REGION Network 6: LECTURA ESCANER SIDE LH
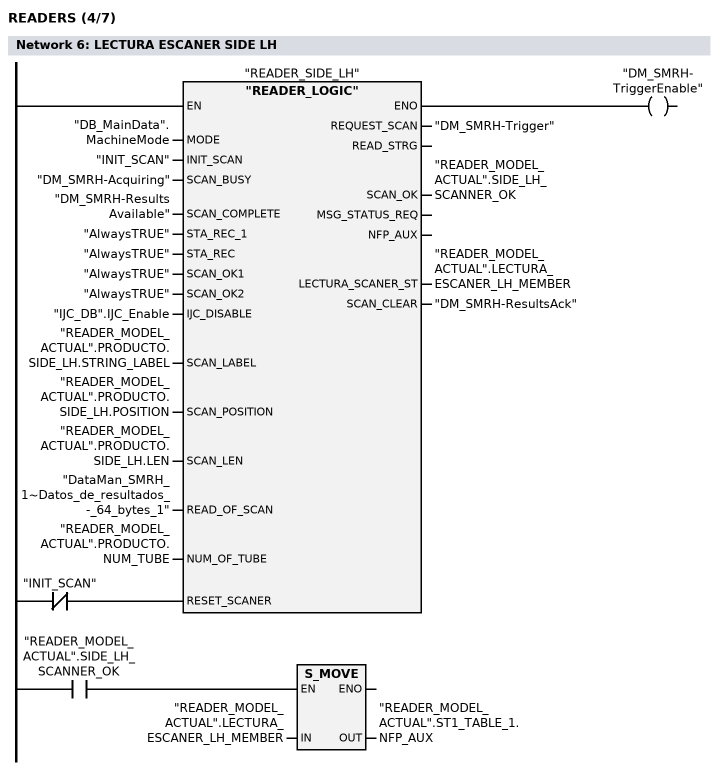
   RUNG wire#powerrail
      "READER_SIDE_LH"(RESET_SCANER := wire#w1, MODE := "DB_MainData".MachineMode, INIT_SCAN := "INIT_SCAN", SCAN_BUSY := "DM_SMRH-Acquiring", SCAN_COMPLETE := "DM_SMRH-Results Available", STA_REC_1 := "AlwaysTRUE", STA_REC := "AlwaysTRUE", SCAN_OK1 := "AlwaysTRUE", SCAN_OK2 := "AlwaysTRUE", IJC_DISABLE := "IJC_DB".IJC_Enable, SCAN_LABEL := "READER_MODEL_ACTUAL".PRODUCTO.SIDE_LH.STRING_LABEL, SCAN_POSITION := "READER_MODEL_ACTUAL".PRODUCTO.SIDE_LH.POSITION, SCAN_LEN := "READER_MODEL_ACTUAL".PRODUCTO.SIDE_LH.LEN, READ_OF_SCAN := "DataMan_SMRH_1~Datos_de_resultados_-_64_bytes_1", NUM_OF_TUBE := "READER_MODEL_ACTUAL".PRODUCTO.NUM_TUBE, REQUEST_SCAN => "DM_SMRH-Trigger", READ_STRG =>, SCAN_OK => "READER_MODEL_ACTUAL".SIDE_LH_SCANNER_OK, MSG_STATUS_REQ =>, NFP_AUX =>, LECTURA_SCANER_ST => "READER_MODEL_ACTUAL".LECTURA_ESCANER_LH_MEMBER, SCAN_CLEAR => "DM_SMRH-ResultsAck")
      Coil( "DM_SMRH-TriggerEnable" )
   END_RUNG
   RUNG wire#powerrail
      I_Contact( "INIT_SCAN" )
   END_RUNG wire#w1
   RUNG wire#powerrail
      Contact( "READER_MODEL_ACTUAL".SIDE_LH_SCANNER_OK )
      S_Move(in := "READER_MODEL_ACTUAL".LECTURA_ESCANER_LH_MEMBER, out => "READER_MODEL_ACTUAL".ST1_TABLE_1.NFP_AUX)
   END_RUNG
   // the same network as SCL:
   "READER_SIDE_LH"(MODE := "DB_MainData".MachineMode,   // "READER_LOGIC"
                    INIT_SCAN := "INIT_SCAN",
                    SCAN_BUSY := "DM_SMRH-Acquiring",
                    SCAN_COMPLETE := "DM_SMRH-Results Available",
                    STA_REC_1 := "AlwaysTRUE",
                    STA_REC := "AlwaysTRUE",
                    SCAN_OK1 := "AlwaysTRUE",
                    SCAN_OK2 := "AlwaysTRUE",
                    IJC_DISABLE := "IJC_DB".IJC_Enable,
                    SCAN_LABEL := "READER_MODEL_ACTUAL".PRODUCTO.SIDE_LH.STRING_LABEL,
                    SCAN_POSITION := "READER_MODEL_ACTUAL".PRODUCTO.SIDE_LH.POSITION,
                    SCAN_LEN := "READER_MODEL_ACTUAL".PRODUCTO.SIDE_LH.LEN,
                    READ_OF_SCAN := "DataMan_SMRH_1~Datos_de_resultados_-_64_bytes_1",
                    NUM_OF_TUBE := "READER_MODEL_ACTUAL".PRODUCTO.NUM_TUBE,
                    RESET_SCANER := NOT "INIT_SCAN",
                    REQUEST_SCAN => "DM_SMRH-Trigger",
                    SCAN_OK => "READER_MODEL_ACTUAL".SIDE_LH_SCANNER_OK,
                    LECTURA_SCANER_ST => "READER_MODEL_ACTUAL".LECTURA_ESCANER_LH_MEMBER,
                    SCAN_CLEAR => "DM_SMRH-ResultsAck",
                    ENO => #_w1);
   "DM_SMRH-TriggerEnable" := #_w1;
   IF "READER_MODEL_ACTUAL".SIDE_LH_SCANNER_OK THEN
       "READER_MODEL_ACTUAL".ST1_TABLE_1.NFP_AUX := "READER_MODEL_ACTUAL".LECTURA_ESCANER_LH_MEMBER;
   END_IF;
END_REGION

REGION Network 7: LECTURA ESCANER SIDE RH
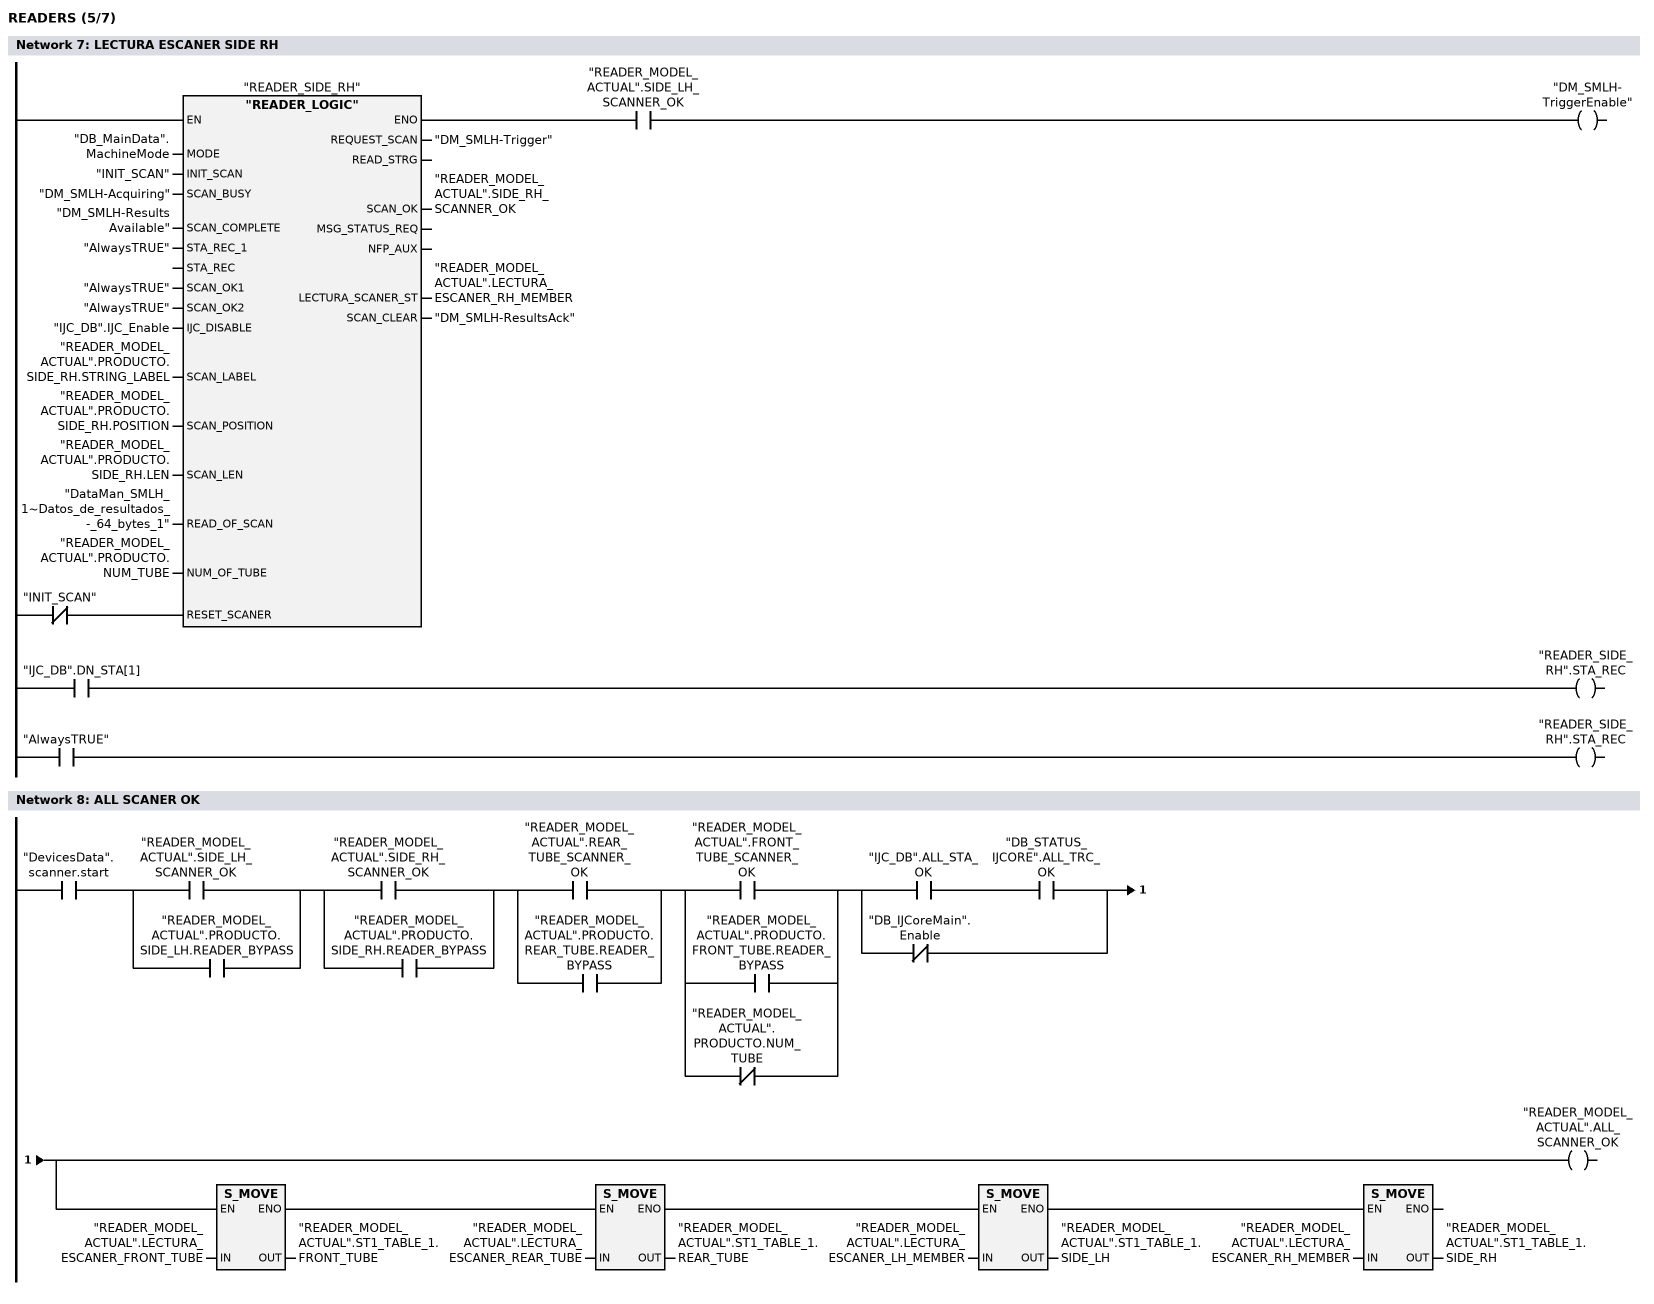
   RUNG wire#powerrail
      "READER_SIDE_RH"(RESET_SCANER := wire#w1, MODE := "DB_MainData".MachineMode, INIT_SCAN := "INIT_SCAN", SCAN_BUSY := "DM_SMLH-Acquiring", SCAN_COMPLETE := "DM_SMLH-Results Available", STA_REC_1 := "AlwaysTRUE", STA_REC :=, SCAN_OK1 := "AlwaysTRUE", SCAN_OK2 := "AlwaysTRUE", IJC_DISABLE := "IJC_DB".IJC_Enable, SCAN_LABEL := "READER_MODEL_ACTUAL".PRODUCTO.SIDE_RH.STRING_LABEL, SCAN_POSITION := "READER_MODEL_ACTUAL".PRODUCTO.SIDE_RH.POSITION, SCAN_LEN := "READER_MODEL_ACTUAL".PRODUCTO.SIDE_RH.LEN, READ_OF_SCAN := "DataMan_SMLH_1~Datos_de_resultados_-_64_bytes_1", NUM_OF_TUBE := "READER_MODEL_ACTUAL".PRODUCTO.NUM_TUBE, REQUEST_SCAN => "DM_SMLH-Trigger", READ_STRG =>, SCAN_OK => "READER_MODEL_ACTUAL".SIDE_RH_SCANNER_OK, MSG_STATUS_REQ =>, NFP_AUX =>, LECTURA_SCANER_ST => "READER_MODEL_ACTUAL".LECTURA_ESCANER_RH_MEMBER, SCAN_CLEAR => "DM_SMLH-ResultsAck")
      Contact( "READER_MODEL_ACTUAL".SIDE_LH_SCANNER_OK )
      Coil( "DM_SMLH-TriggerEnable" )
   END_RUNG
   RUNG wire#powerrail
      I_Contact( "INIT_SCAN" )
   END_RUNG wire#w1
   RUNG wire#powerrail
      Contact( "IJC_DB".DN_STA[1] )
      Coil( "READER_SIDE_RH".STA_REC )
   END_RUNG
   RUNG wire#powerrail
      Contact( "AlwaysTRUE" )
      Coil( "READER_SIDE_RH".STA_REC )
   END_RUNG
   // the same network as SCL:
   "READER_SIDE_RH"(MODE := "DB_MainData".MachineMode,   // "READER_LOGIC"
                    INIT_SCAN := "INIT_SCAN",
                    SCAN_BUSY := "DM_SMLH-Acquiring",
                    SCAN_COMPLETE := "DM_SMLH-Results Available",
                    STA_REC_1 := "AlwaysTRUE",
                    SCAN_OK1 := "AlwaysTRUE",
                    SCAN_OK2 := "AlwaysTRUE",
                    IJC_DISABLE := "IJC_DB".IJC_Enable,
                    SCAN_LABEL := "READER_MODEL_ACTUAL".PRODUCTO.SIDE_RH.STRING_LABEL,
                    SCAN_POSITION := "READER_MODEL_ACTUAL".PRODUCTO.SIDE_RH.POSITION,
                    SCAN_LEN := "READER_MODEL_ACTUAL".PRODUCTO.SIDE_RH.LEN,
                    READ_OF_SCAN := "DataMan_SMLH_1~Datos_de_resultados_-_64_bytes_1",
                    NUM_OF_TUBE := "READER_MODEL_ACTUAL".PRODUCTO.NUM_TUBE,
                    RESET_SCANER := NOT "INIT_SCAN",
                    REQUEST_SCAN => "DM_SMLH-Trigger",
                    SCAN_OK => "READER_MODEL_ACTUAL".SIDE_RH_SCANNER_OK,
                    LECTURA_SCANER_ST => "READER_MODEL_ACTUAL".LECTURA_ESCANER_RH_MEMBER,
                    SCAN_CLEAR => "DM_SMLH-ResultsAck",
                    ENO => #_w1);
   "DM_SMLH-TriggerEnable" := #_w1 AND "READER_MODEL_ACTUAL".SIDE_LH_SCANNER_OK;
   "READER_SIDE_RH".STA_REC := "IJC_DB".DN_STA[1];
   "READER_SIDE_RH".STA_REC := "AlwaysTRUE";
END_REGION

REGION Network 8: ALL SCANER OK
   RUNG wire#powerrail
      Contact( "DevicesData".scanner.start )
      wire#w1
      Contact( "READER_MODEL_ACTUAL".SIDE_LH_SCANNER_OK )
      wire#w2
      Contact( "READER_MODEL_ACTUAL".SIDE_RH_SCANNER_OK )
      wire#w3
      Contact( "READER_MODEL_ACTUAL".REAR_TUBE_SCANNER_OK )
      wire#w4
      Contact( "READER_MODEL_ACTUAL".FRONT_TUBE_SCANNER_OK )
      wire#w5
      Contact( "IJC_DB".ALL_STA_OK )
      Contact( "DB_STATUS_IJCORE".ALL_TRC_OK )
      wire#w6
      Coil( "READER_MODEL_ACTUAL".ALL_SCANNER_OK )
   END_RUNG
   RUNG wire#w1
      Contact( "READER_MODEL_ACTUAL".PRODUCTO.SIDE_LH.READER_BYPASS )
   END_RUNG wire#w2
   RUNG wire#w2
      Contact( "READER_MODEL_ACTUAL".PRODUCTO.SIDE_RH.READER_BYPASS )
   END_RUNG wire#w3
   RUNG wire#w3
      Contact( "READER_MODEL_ACTUAL".PRODUCTO.REAR_TUBE.READER_BYPASS )
   END_RUNG wire#w4
   RUNG wire#w4
      Contact( "READER_MODEL_ACTUAL".PRODUCTO.FRONT_TUBE.READER_BYPASS )
   END_RUNG wire#w5
   RUNG wire#w4
      I_Contact( "READER_MODEL_ACTUAL".PRODUCTO.NUM_TUBE )
   END_RUNG wire#w5
   RUNG wire#w5
      I_Contact( "DB_IJCoreMain".Enable )
   END_RUNG wire#w6
   RUNG wire#w6
      S_Move(in := "READER_MODEL_ACTUAL".LECTURA_ESCANER_FRONT_TUBE, out => "READER_MODEL_ACTUAL".ST1_TABLE_1.FRONT_TUBE)
      S_Move(in := "READER_MODEL_ACTUAL".LECTURA_ESCANER_REAR_TUBE, out => "READER_MODEL_ACTUAL".ST1_TABLE_1.REAR_TUBE)
      S_Move(in := "READER_MODEL_ACTUAL".LECTURA_ESCANER_LH_MEMBER, out => "READER_MODEL_ACTUAL".ST1_TABLE_1.SIDE_LH)
      S_Move(in := "READER_MODEL_ACTUAL".LECTURA_ESCANER_RH_MEMBER, out => "READER_MODEL_ACTUAL".ST1_TABLE_1.SIDE_RH)
   END_RUNG
   // the same network as SCL:
   "READER_MODEL_ACTUAL".ALL_SCANNER_OK := "DevicesData".scanner.start AND ("READER_MODEL_ACTUAL".SIDE_LH_SCANNER_OK OR "READER_MODEL_ACTUAL".PRODUCTO.SIDE_LH.READER_BYPASS) AND ("READER_MODEL_ACTUAL".SIDE_RH_SCANNER_OK OR "READER_MODEL_ACTUAL".PRODUCTO.SIDE_RH.READER_BYPASS) AND ("READER_MODEL_ACTUAL".REAR_TUBE_SCANNER_OK OR "READER_MODEL_ACTUAL".PRODUCTO.REAR_TUBE.READER_BYPASS) AND ("READER_MODEL_ACTUAL".FRONT_TUBE_SCANNER_OK OR "READER_MODEL_ACTUAL".PRODUCTO.FRONT_TUBE.READER_BYPASS OR NOT "READER_MODEL_ACTUAL".PRODUCTO.NUM_TUBE) AND (("IJC_DB".ALL_STA_OK AND "DB_STATUS_IJCORE".ALL_TRC_OK) OR NOT "DB_IJCoreMain".Enable);
   IF "READER_MODEL_ACTUAL".ALL_SCANNER_OK THEN
       "READER_MODEL_ACTUAL".ST1_TABLE_1.FRONT_TUBE := "READER_MODEL_ACTUAL".LECTURA_ESCANER_FRONT_TUBE;
       "READER_MODEL_ACTUAL".ST1_TABLE_1.REAR_TUBE := "READER_MODEL_ACTUAL".LECTURA_ESCANER_REAR_TUBE;
       "READER_MODEL_ACTUAL".ST1_TABLE_1.SIDE_LH := "READER_MODEL_ACTUAL".LECTURA_ESCANER_LH_MEMBER;
       "READER_MODEL_ACTUAL".ST1_TABLE_1.SIDE_RH := "READER_MODEL_ACTUAL".LECTURA_ESCANER_RH_MEMBER;
   END_IF;
END_REGION

REGION Network 9
   // "DB_ProductionProgramActual".Program.MechanicalType:
   // 0 - LH
   // 1 - RH
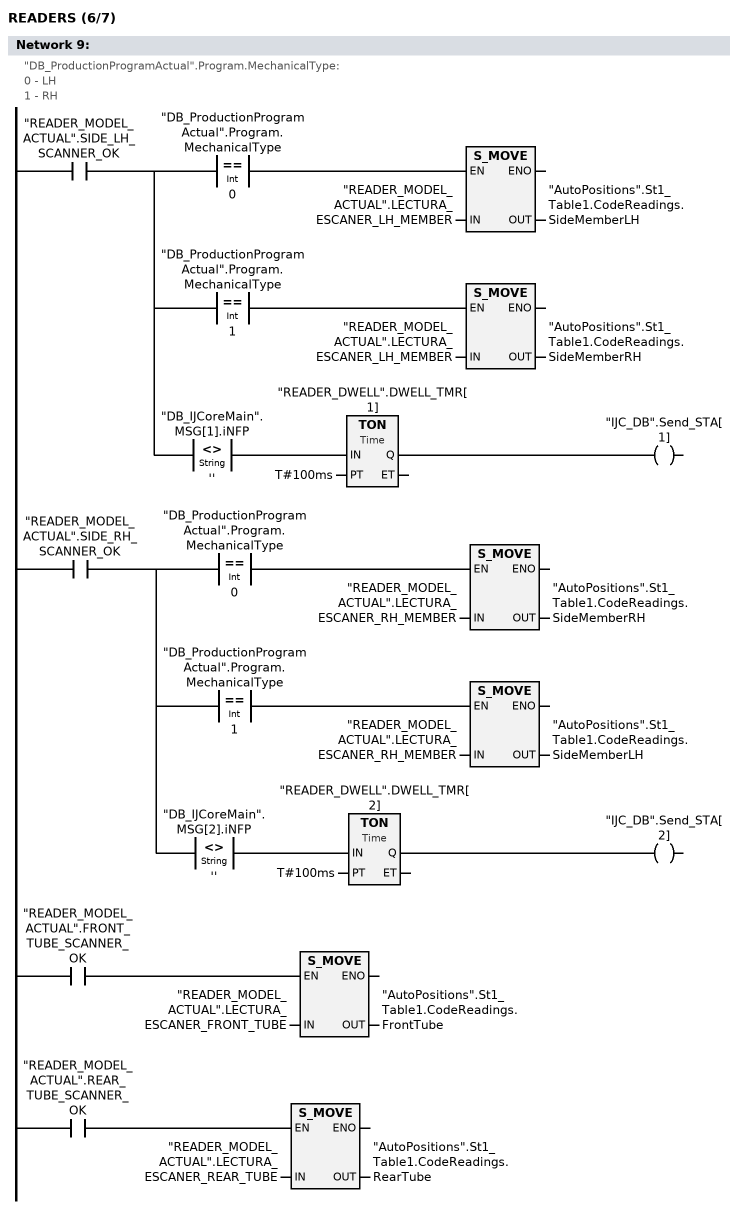
   RUNG wire#powerrail
      Contact( "READER_MODEL_ACTUAL".SIDE_LH_SCANNER_OK )
      wire#w1
      { S7_Templates := "SrcType := Int" } EQ_Contact(in1 := "DB_ProductionProgramActual".Program.MechanicalType, in2 := 0)
      S_Move(in := "READER_MODEL_ACTUAL".LECTURA_ESCANER_LH_MEMBER, out => "AutoPositions".St1_Table1.CodeReadings.SideMemberLH)
   END_RUNG
   RUNG wire#w1
      { S7_Templates := "SrcType := Int" } EQ_Contact(in1 := "DB_ProductionProgramActual".Program.MechanicalType, in2 := 1)
      S_Move(in := "READER_MODEL_ACTUAL".LECTURA_ESCANER_LH_MEMBER, out => "AutoPositions".St1_Table1.CodeReadings.SideMemberRH)
   END_RUNG
   RUNG wire#w1
      { S7_Templates := "SrcType := String" } NE_Contact(in1 := "DB_IJCoreMain".MSG[1].iNFP, in2 := '')
      { S7_Templates := "time_type := Time" } "READER_DWELL".DWELL_TMR[1].TON(pt := T#100ms, et =>)
      Coil( "IJC_DB".Send_STA[1] )
   END_RUNG
   RUNG wire#powerrail
      Contact( "READER_MODEL_ACTUAL".SIDE_RH_SCANNER_OK )
      wire#w2
      { S7_Templates := "SrcType := Int" } EQ_Contact(in1 := "DB_ProductionProgramActual".Program.MechanicalType, in2 := 0)
      S_Move(in := "READER_MODEL_ACTUAL".LECTURA_ESCANER_RH_MEMBER, out => "AutoPositions".St1_Table1.CodeReadings.SideMemberRH)
   END_RUNG
   RUNG wire#w2
      { S7_Templates := "SrcType := Int" } EQ_Contact(in1 := "DB_ProductionProgramActual".Program.MechanicalType, in2 := 1)
      S_Move(in := "READER_MODEL_ACTUAL".LECTURA_ESCANER_RH_MEMBER, out => "AutoPositions".St1_Table1.CodeReadings.SideMemberLH)
   END_RUNG
   RUNG wire#w2
      { S7_Templates := "SrcType := String" } NE_Contact(in1 := "DB_IJCoreMain".MSG[2].iNFP, in2 := '')
      { S7_Templates := "time_type := Time" } "READER_DWELL".DWELL_TMR[2].TON(pt := T#100ms, et =>)
      Coil( "IJC_DB".Send_STA[2] )
   END_RUNG
   RUNG wire#powerrail
      Contact( "READER_MODEL_ACTUAL".FRONT_TUBE_SCANNER_OK )
      S_Move(in := "READER_MODEL_ACTUAL".LECTURA_ESCANER_FRONT_TUBE, out => "AutoPositions".St1_Table1.CodeReadings.FrontTube)
   END_RUNG
   RUNG wire#powerrail
      Contact( "READER_MODEL_ACTUAL".REAR_TUBE_SCANNER_OK )
      S_Move(in := "READER_MODEL_ACTUAL".LECTURA_ESCANER_REAR_TUBE, out => "AutoPositions".St1_Table1.CodeReadings.RearTube)
   END_RUNG
   // the same network as SCL:
   IF "READER_MODEL_ACTUAL".SIDE_LH_SCANNER_OK AND ("DB_ProductionProgramActual".Program.MechanicalType = 0) THEN
       "AutoPositions".St1_Table1.CodeReadings.SideMemberLH := "READER_MODEL_ACTUAL".LECTURA_ESCANER_LH_MEMBER;
   END_IF;
   IF "READER_MODEL_ACTUAL".SIDE_LH_SCANNER_OK AND ("DB_ProductionProgramActual".Program.MechanicalType = 1) THEN
       "AutoPositions".St1_Table1.CodeReadings.SideMemberRH := "READER_MODEL_ACTUAL".LECTURA_ESCANER_LH_MEMBER;
   END_IF;
   "READER_DWELL".DWELL_TMR[1].TON(IN := "READER_MODEL_ACTUAL".SIDE_LH_SCANNER_OK AND ("DB_IJCoreMain".MSG[1].iNFP <> ''),
                           PT := T#100ms);
   "IJC_DB".Send_STA[1] := "READER_DWELL".DWELL_TMR[1].Q;
   IF "READER_MODEL_ACTUAL".SIDE_RH_SCANNER_OK AND ("DB_ProductionProgramActual".Program.MechanicalType = 0) THEN
       "AutoPositions".St1_Table1.CodeReadings.SideMemberRH := "READER_MODEL_ACTUAL".LECTURA_ESCANER_RH_MEMBER;
   END_IF;
   IF "READER_MODEL_ACTUAL".SIDE_RH_SCANNER_OK AND ("DB_ProductionProgramActual".Program.MechanicalType = 1) THEN
       "AutoPositions".St1_Table1.CodeReadings.SideMemberLH := "READER_MODEL_ACTUAL".LECTURA_ESCANER_RH_MEMBER;
   END_IF;
   "READER_DWELL".DWELL_TMR[2].TON(IN := "READER_MODEL_ACTUAL".SIDE_RH_SCANNER_OK AND ("DB_IJCoreMain".MSG[2].iNFP <> ''),
                           PT := T#100ms);
   "IJC_DB".Send_STA[2] := "READER_DWELL".DWELL_TMR[2].Q;
   IF "READER_MODEL_ACTUAL".FRONT_TUBE_SCANNER_OK THEN
       "AutoPositions".St1_Table1.CodeReadings.FrontTube := "READER_MODEL_ACTUAL".LECTURA_ESCANER_FRONT_TUBE;
   END_IF;
   IF "READER_MODEL_ACTUAL".REAR_TUBE_SCANNER_OK THEN
       "AutoPositions".St1_Table1.CodeReadings.RearTube := "READER_MODEL_ACTUAL".LECTURA_ESCANER_REAR_TUBE;
   END_IF;
END_REGION

REGION Network 10: SENSORES LASER
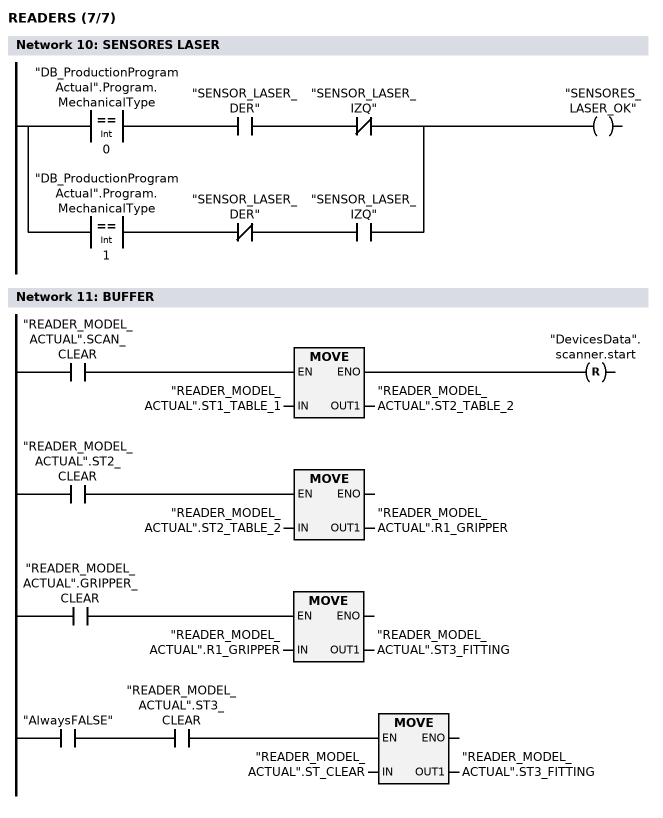
   RUNG wire#powerrail
      { S7_Templates := "SrcType := Int" } EQ_Contact(in1 := "DB_ProductionProgramActual".Program.MechanicalType, in2 := 0)
      Contact( "SENSOR_LASER_DER" )
      I_Contact( "SENSOR_LASER_IZQ" )
      wire#w1
      Coil( "SENSORES_LASER_OK" )
   END_RUNG
   RUNG wire#powerrail
      { S7_Templates := "SrcType := Int" } EQ_Contact(in1 := "DB_ProductionProgramActual".Program.MechanicalType, in2 := 1)
      I_Contact( "SENSOR_LASER_DER" )
      Contact( "SENSOR_LASER_IZQ" )
   END_RUNG wire#w1
   // the same network as SCL:
   "SENSORES_LASER_OK" := (("DB_ProductionProgramActual".Program.MechanicalType = 0) AND "SENSOR_LASER_DER" AND NOT "SENSOR_LASER_IZQ") OR (("DB_ProductionProgramActual".Program.MechanicalType = 1) AND NOT "SENSOR_LASER_DER" AND "SENSOR_LASER_IZQ");
END_REGION

REGION Network 11: BUFFER
   RUNG wire#powerrail
      Contact( "READER_MODEL_ACTUAL".SCAN_CLEAR )
      Move(in := "READER_MODEL_ACTUAL".ST1_TABLE_1, out1 => "READER_MODEL_ACTUAL".ST2_TABLE_2)
      R_Coil( "DevicesData".scanner.start )
   END_RUNG
   RUNG wire#powerrail
      Contact( "READER_MODEL_ACTUAL".ST2_CLEAR )
      Move(in := "READER_MODEL_ACTUAL".ST2_TABLE_2, out1 => "READER_MODEL_ACTUAL".R1_GRIPPER)
   END_RUNG
   RUNG wire#powerrail
      Contact( "READER_MODEL_ACTUAL".GRIPPER_CLEAR )
      Move(in := "READER_MODEL_ACTUAL".R1_GRIPPER, out1 => "READER_MODEL_ACTUAL".ST3_FITTING)
   END_RUNG
   RUNG wire#powerrail
      Contact( "AlwaysFALSE" )
      Contact( "READER_MODEL_ACTUAL".ST3_CLEAR )
      Move(in := "READER_MODEL_ACTUAL".ST_CLEAR, out1 => "READER_MODEL_ACTUAL".ST3_FITTING)
   END_RUNG
   // the same network as SCL:
   IF "READER_MODEL_ACTUAL".SCAN_CLEAR THEN
       "READER_MODEL_ACTUAL".ST2_TABLE_2 := "READER_MODEL_ACTUAL".ST1_TABLE_1;
       "DevicesData".scanner.start := FALSE;
   END_IF;
   IF "READER_MODEL_ACTUAL".ST2_CLEAR THEN
       "READER_MODEL_ACTUAL".R1_GRIPPER := "READER_MODEL_ACTUAL".ST2_TABLE_2;
   END_IF;
   IF "READER_MODEL_ACTUAL".GRIPPER_CLEAR THEN
       "READER_MODEL_ACTUAL".ST3_FITTING := "READER_MODEL_ACTUAL".R1_GRIPPER;
   END_IF;
   IF "AlwaysFALSE" AND "READER_MODEL_ACTUAL".ST3_CLEAR THEN
       "READER_MODEL_ACTUAL".ST3_FITTING := "READER_MODEL_ACTUAL".ST_CLEAR;
   END_IF;
END_REGION
END_FUNCTION

FUNCTION_BLOCK "READER_LOGIC"   // FB24, LAD
{ S7_Optimized_Access := 'TRUE' }
VERSION : 0.1
// stored: AutoNumber true, IsIECCheckEnabled false, IsRetainMemResEnabled false, MemoryReserve 100, SetENOAutomatically false, UDAEnableTagReadback false
   VAR_INPUT
      MODE : UInt;
      INIT_SCAN : Bool;
      SCAN_BUSY : Bool;
      SCAN_COMPLETE : Bool;
      STA_REC_1 : Bool;
      STA_REC : Bool;
      SCAN_OK1 : Bool;
      SCAN_OK2 : Bool;
      IJC_DISABLE : Bool;
      SCAN_LABEL : String;
      SCAN_POSITION : Int;
      SCAN_LEN : Int;
      READ_OF_SCAN : HW_SUBMODULE;
      NUM_OF_TUBE : Bool;
      RESET_SCANER : Bool;
   END_VAR
   VAR_OUTPUT
      REQUEST_SCAN : Bool;
      READ_STRG : String;
      SCAN_OK : Bool;
      MSG_STATUS_REQ : Bool;
      NFP_AUX : String;
      LECTURA_SCANER_ST : String;
      SCAN_CLEAR : Bool;
   END_VAR
   VAR
      RET_TRIG : IEC_TIMER;
   END_VAR
   VAR_TEMP
      ERROR_RECIBIDO_ESCANER : Int;
      RECIBIDO_SCANER : Array[0..254] of Char;
      RECIBIDO_SCANER_STRG : String;
      LECTURA_SCANER : String;
      done : Bool;
   END_VAR
   VAR_TEMP   // added for the SCL form of the ladder/FBD networks
      _w1 : Bool;
      _w2 : Bool;
      _w3 : Bool;
      _w4 : Bool;
      _w5 : Bool;
   END_VAR
BEGIN

REGION Network 1
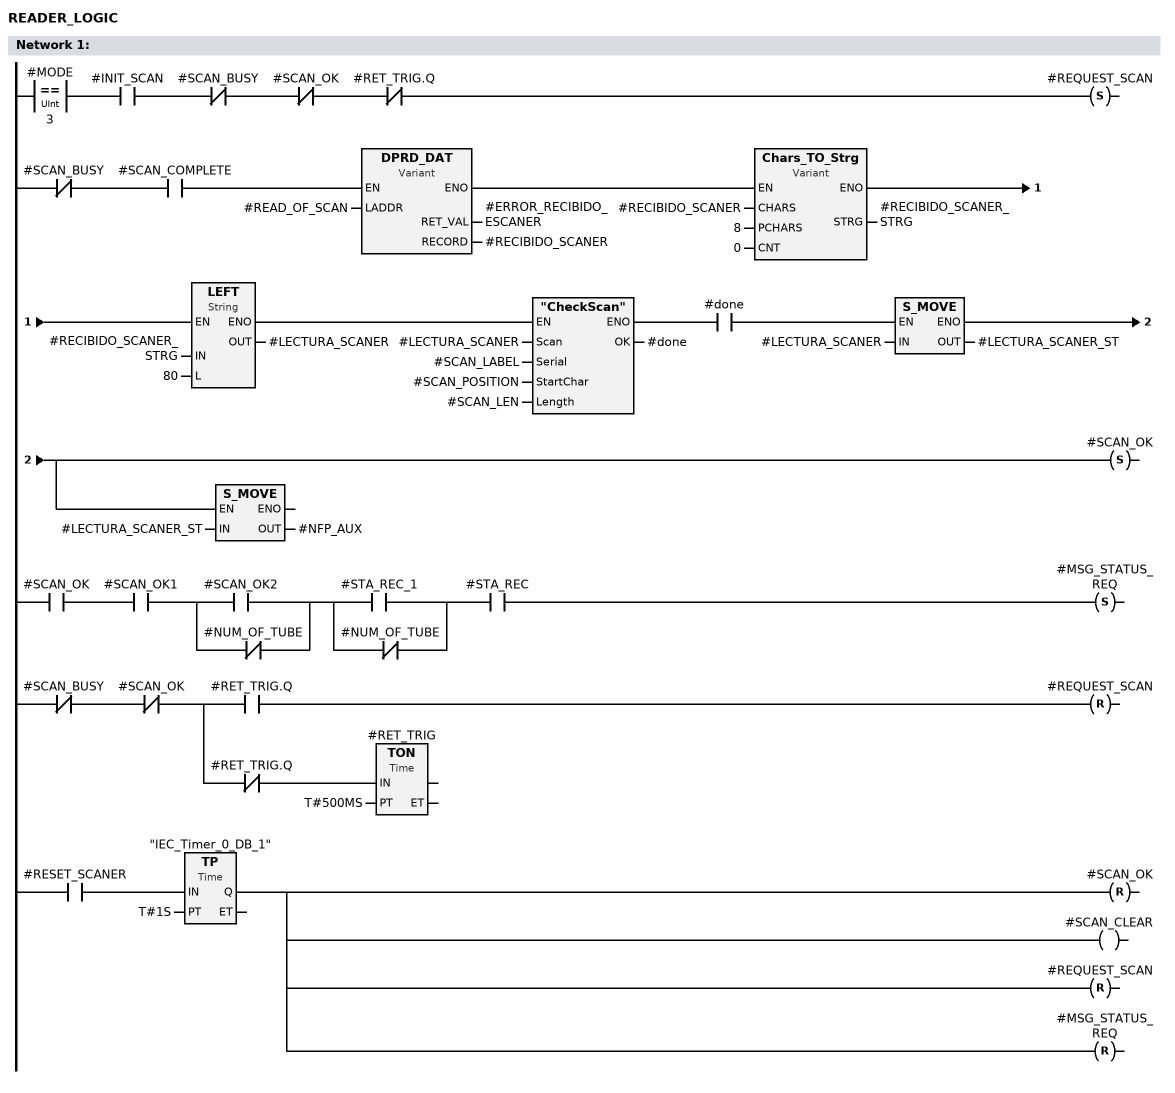
   RUNG wire#powerrail
      { S7_Templates := "SrcType := UInt" } EQ_Contact(in1 := #MODE, in2 := 3)
      Contact( #INIT_SCAN )
      I_Contact( #SCAN_BUSY )
      I_Contact( #SCAN_OK )
      I_Contact( #RET_TRIG.Q )
      S_Coil( #REQUEST_SCAN )
   END_RUNG
   RUNG wire#powerrail
      I_Contact( #SCAN_BUSY )
      Contact( #SCAN_COMPLETE )
      { S7_Templates := "[ptr_type := Variant, laddr_type := HW_IO]" } DPRD_DAT(LADDR := #READ_OF_SCAN, RET_VAL => #ERROR_RECIBIDO_ESCANER, RECORD => #RECIBIDO_SCANER)
      { S7_Templates := "[ptr_type := Variant, str_type := String]" } Chars_TO_Strg(Chars := #RECIBIDO_SCANER, pChars := 8, Cnt := 0, Strg => #RECIBIDO_SCANER_STRG)
      { S7_Templates := "str_type := String" } LEFT(IN := #RECIBIDO_SCANER_STRG, L := 80, OUT => #LECTURA_SCANER)
      "CheckScan"(Scan := #LECTURA_SCANER, Serial := #SCAN_LABEL, StartChar := #SCAN_POSITION, Length := #SCAN_LEN, OK => #done)
      Contact( #done )
      S_Move(in := #LECTURA_SCANER, out => #LECTURA_SCANER_ST)
      wire#w1
      S_Coil( #SCAN_OK )
   END_RUNG
   RUNG wire#w1
      S_Move(in := #LECTURA_SCANER_ST, out => #NFP_AUX)
   END_RUNG
   RUNG wire#powerrail
      Contact( #SCAN_OK )
      Contact( #SCAN_OK1 )
      wire#w2
      Contact( #SCAN_OK2 )
      wire#w3
      Contact( #STA_REC_1 )
      wire#w4
      Contact( #STA_REC )
      S_Coil( #MSG_STATUS_REQ )
   END_RUNG
   RUNG wire#w2
      I_Contact( #NUM_OF_TUBE )
   END_RUNG wire#w3
   RUNG wire#w3
      I_Contact( #NUM_OF_TUBE )
   END_RUNG wire#w4
   RUNG wire#powerrail
      I_Contact( #SCAN_BUSY )
      I_Contact( #SCAN_OK )
      wire#w5
      Contact( #RET_TRIG.Q )
      R_Coil( #REQUEST_SCAN )
   END_RUNG
   RUNG wire#w5
      I_Contact( #RET_TRIG.Q )
      { S7_Templates := "time_type := Time" } #RET_TRIG.TON(pt := T#500MS, et =>)
   END_RUNG
   RUNG wire#powerrail
      Contact( #RESET_SCANER )
      { S7_Templates := "time_type := Time" } "IEC_Timer_0_DB_1".TP(pt := T#1S, et =>)
      wire#w6
      R_Coil( #SCAN_OK )
   END_RUNG
   RUNG wire#w6
      Coil( #SCAN_CLEAR )
   END_RUNG
   RUNG wire#w6
      R_Coil( #REQUEST_SCAN )
   END_RUNG
   RUNG wire#w6
      R_Coil( #MSG_STATUS_REQ )
   END_RUNG
   // the same network as SCL:
   IF (#MODE = 3) AND #INIT_SCAN AND NOT #SCAN_BUSY AND NOT #SCAN_OK AND NOT #RET_TRIG.Q THEN
       #REQUEST_SCAN := TRUE;
   END_IF;
   #ERROR_RECIBIDO_ESCANER := DPRD_DAT(EN := NOT #SCAN_BUSY AND #SCAN_COMPLETE,
                           LADDR := #READ_OF_SCAN,
                           RECORD => #RECIBIDO_SCANER,
                           ENO => #_w1);
   Chars_TO_Strg(EN := #_w1,
                 Chars := #RECIBIDO_SCANER,
                 pChars := 8,
                 Cnt := 0,
                 Strg => #RECIBIDO_SCANER_STRG,
                 ENO => #_w2);
   LEFT(EN := #_w2, IN := #RECIBIDO_SCANER_STRG, L := 80, OUT => #LECTURA_SCANER, ENO => #_w3);
   "CheckScan"(EN := #_w3,
               Scan := #LECTURA_SCANER,
               Serial := #SCAN_LABEL,
               StartChar := #SCAN_POSITION,
               Length := #SCAN_LEN,
               OK => #done,
               ENO => #_w4);
   IF #_w4 AND #done THEN
       #LECTURA_SCANER_ST := #LECTURA_SCANER;
       #SCAN_OK := TRUE;
       #NFP_AUX := #LECTURA_SCANER_ST;
   END_IF;
   IF #SCAN_OK AND #SCAN_OK1 AND (#SCAN_OK2 OR NOT #NUM_OF_TUBE) AND (#STA_REC_1 OR NOT #NUM_OF_TUBE) AND #STA_REC THEN
       #MSG_STATUS_REQ := TRUE;
   END_IF;
   #_w5 := NOT #SCAN_BUSY AND NOT #SCAN_OK;
   IF #_w5 AND #RET_TRIG.Q THEN #REQUEST_SCAN := FALSE; END_IF;
   #RET_TRIG.TON(IN := #_w5 AND NOT #RET_TRIG.Q, PT := T#500MS);
   "IEC_Timer_0_DB_1".TP(IN := #RESET_SCANER, PT := T#1S);
   IF "IEC_Timer_0_DB_1".Q THEN #SCAN_OK := FALSE; END_IF;
   #SCAN_CLEAR := "IEC_Timer_0_DB_1".Q;
   IF "IEC_Timer_0_DB_1".Q THEN
       #REQUEST_SCAN := FALSE;
       #MSG_STATUS_REQ := FALSE;
   END_IF;
END_REGION
END_FUNCTION_BLOCK

FUNCTION_BLOCK "FB_IJC"   // FB800, LAD
{ S7_Optimized_Access := 'TRUE' }
VERSION : 0.1
// stored: AutoNumber false, IsIECCheckEnabled false, IsRetainMemResEnabled false, MemoryReserve 100, SetENOAutomatically false, UDAEnableTagReadback false
   VAR
      MSG { S7_SetPoint := 'True'} : Array[0..30] of "IJC PROTOCOL";
      NFP_1 { S7_SetPoint := 'True'} : String[8];
      Component_1 : String[30];
      NFP_2 : String[8];
      Component_2 : String[30];
      Send_STA : Array[0..5] of Bool;
      Send_TRC : Array[0..5] of Bool;
      Send_TRR : Array[0..5] of Bool;
      Send_CNF : Array[0..5] of Bool;
      IJC_STA_1_Ans_OK : Bool;
      IJC_STA_1_Ans_NOK : Bool;
      IJC_TRC_1_Ans_OK : Bool;
      IJC_TRC_1_Ans_NOK : Bool;
      IJC_STA_2_Ans_NOK : Bool;
      IJC_STA_2_Ans_OK : Bool;
      IJC_TRC_2_Ans_OK : Bool;
      IJC_TRC_2_Ans_NOK : Bool;
      FP1 : Bool;
      FP2 : Bool;
      FP3 : Bool;
      FP4 : Bool;
      FP5 : Bool;
      FP6 : Bool;
      Reset : Bool;
      IJC_Enable : Bool;
      DN_STA : Array[0..5] of Bool;
      DN_TRC : Array[0..5] of Bool;
      DN_TRR : Array[0..5] of Bool;
      DN_CNF : Array[0..5] of Bool;
      INDEX : Int;
      ALL_STA_OK : Bool;
      AWAKE_SIGNAL_INSTANCE : "AWAKE_SIGNAL";
   END_VAR
   VAR_TEMP
      i : USInt;
      res : SInt;
      INDEX_NFP : Int;
   END_VAR
BEGIN

REGION Network 1
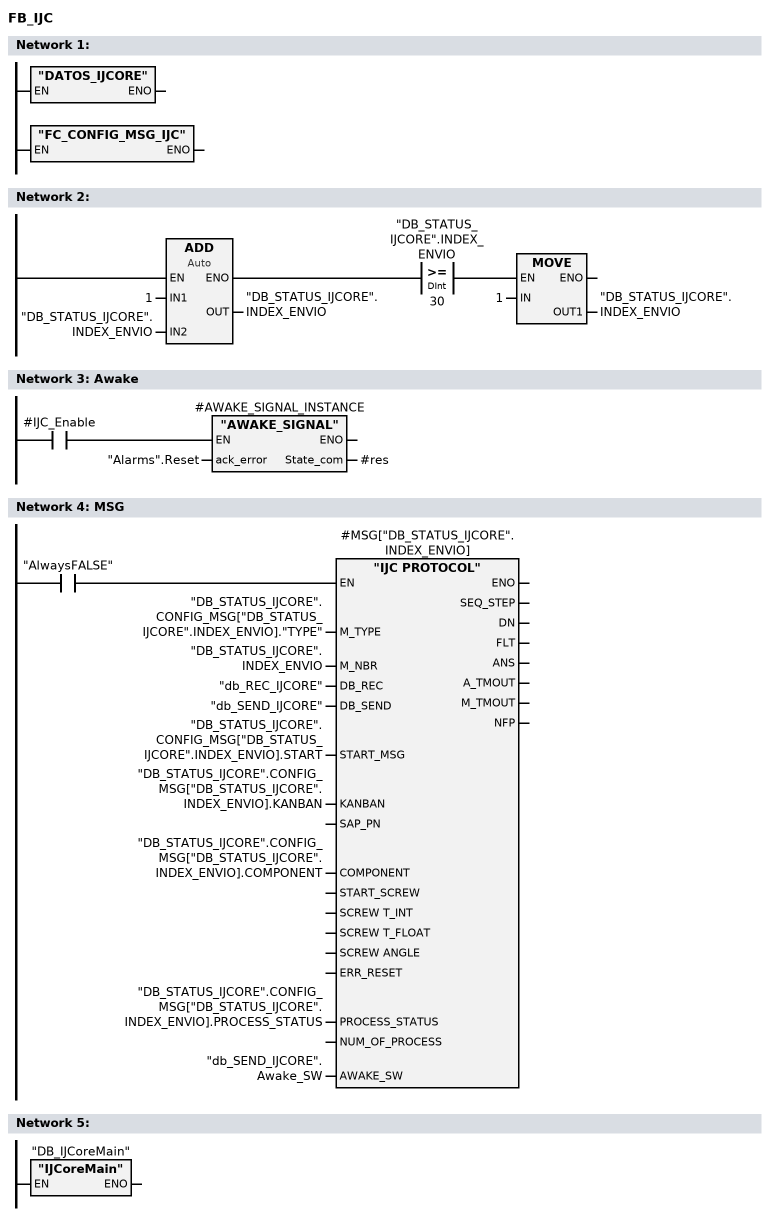
   RUNG wire#powerrail
      "DATOS_IJCORE"()
   END_RUNG
   RUNG wire#powerrail
      "FC_CONFIG_MSG_IJC"()
   END_RUNG
   // the same network as SCL:
   "DATOS_IJCORE"();
   "FC_CONFIG_MSG_IJC"();
END_REGION

REGION Network 2
   RUNG wire#powerrail
      Add(in1 := 1, in2 := "DB_STATUS_IJCORE".INDEX_ENVIO, out => "DB_STATUS_IJCORE".INDEX_ENVIO)
      { S7_Templates := "SrcType := DInt" } GE_Contact(in1 := "DB_STATUS_IJCORE".INDEX_ENVIO, in2 := 30)
      Move(in := 1, out1 => "DB_STATUS_IJCORE".INDEX_ENVIO)
   END_RUNG
   // the same network as SCL:
   "DB_STATUS_IJCORE".INDEX_ENVIO := 1 + "DB_STATUS_IJCORE".INDEX_ENVIO;
   IF "DB_STATUS_IJCORE".INDEX_ENVIO >= 30 THEN "DB_STATUS_IJCORE".INDEX_ENVIO := 1; END_IF;
END_REGION

REGION Network 3: Awake
   RUNG wire#powerrail
      Contact( #IJC_Enable )
      #AWAKE_SIGNAL_INSTANCE(ack_error := "Alarms".Reset, State_com => #res)
   END_RUNG
   // the same network as SCL:
   IF #IJC_Enable THEN
       #AWAKE_SIGNAL_INSTANCE(ack_error := "Alarms".Reset, State_com => #res);   // "AWAKE_SIGNAL"
   END_IF;
END_REGION

REGION Network 4: MSG
   RUNG wire#powerrail
      Contact( "AlwaysFALSE" )
      #MSG["DB_STATUS_IJCORE".INDEX_ENVIO](M_TYPE := "DB_STATUS_IJCORE".CONFIG_MSG["DB_STATUS_IJCORE".INDEX_ENVIO]."TYPE", M_NBR := "DB_STATUS_IJCORE".INDEX_ENVIO, DB_REC := "db_REC_IJCORE", DB_SEND := "db_SEND_IJCORE", START_MSG := "DB_STATUS_IJCORE".CONFIG_MSG["DB_STATUS_IJCORE".INDEX_ENVIO].START, KANBAN := "DB_STATUS_IJCORE".CONFIG_MSG["DB_STATUS_IJCORE".INDEX_ENVIO].KANBAN, SAP_PN :=, COMPONENT := "DB_STATUS_IJCORE".CONFIG_MSG["DB_STATUS_IJCORE".INDEX_ENVIO].COMPONENT, START_SCREW :=, "SCREW T_INT" :=, "SCREW T_FLOAT" :=, "SCREW ANGLE" :=, ERR_RESET :=, PROCESS_STATUS := "DB_STATUS_IJCORE".CONFIG_MSG["DB_STATUS_IJCORE".INDEX_ENVIO].PROCESS_STATUS, NUM_OF_PROCESS :=, AWAKE_SW := "db_SEND_IJCORE".Awake_SW, SEQ_STEP =>, DN =>, FLT =>, ANS =>, A_TMOUT =>, M_TMOUT =>, NFP =>)
   END_RUNG
   // the same network as SCL:
   IF "AlwaysFALSE" THEN
       #MSG["DB_STATUS_IJCORE".INDEX_ENVIO](M_TYPE := "DB_STATUS_IJCORE".CONFIG_MSG["DB_STATUS_IJCORE".INDEX_ENVIO]."TYPE",   // "IJC PROTOCOL"
                               M_NBR := "DB_STATUS_IJCORE".INDEX_ENVIO,
                               DB_REC := "db_REC_IJCORE",
                               DB_SEND := "db_SEND_IJCORE",
                               START_MSG := "DB_STATUS_IJCORE".CONFIG_MSG["DB_STATUS_IJCORE".INDEX_ENVIO].START,
                               KANBAN := "DB_STATUS_IJCORE".CONFIG_MSG["DB_STATUS_IJCORE".INDEX_ENVIO].KANBAN,
                               COMPONENT := "DB_STATUS_IJCORE".CONFIG_MSG["DB_STATUS_IJCORE".INDEX_ENVIO].COMPONENT,
                               PROCESS_STATUS := "DB_STATUS_IJCORE".CONFIG_MSG["DB_STATUS_IJCORE".INDEX_ENVIO].PROCESS_STATUS,
                               AWAKE_SW := "db_SEND_IJCORE".Awake_SW);
   END_IF;
END_REGION

REGION Network 5
   RUNG wire#powerrail
      "DB_IJCoreMain"()
   END_RUNG
   // the same network as SCL:
   "DB_IJCoreMain"();   // "IJCoreMain"
END_REGION
END_FUNCTION_BLOCK

FUNCTION "DATOS_IJCORE" : Void   // FC1, LAD
{ S7_Optimized_Access := 'TRUE' }
VERSION : 0.1
// stored: AutoNumber true, IsIECCheckEnabled false, SetENOAutomatically false, UDAEnableTagReadback false
   VAR_TEMP
      ijc_off : Bool;
      PV_HMI : Int;
      INDEX_HMI2 : Int;
      INDEX_HMI3 : Int;
   END_VAR
   VAR_TEMP   // added for the SCL form of the ladder/FBD networks
      _w1 : Bool;
   END_VAR
BEGIN

REGION Network 2: ALARMA ACTIVA
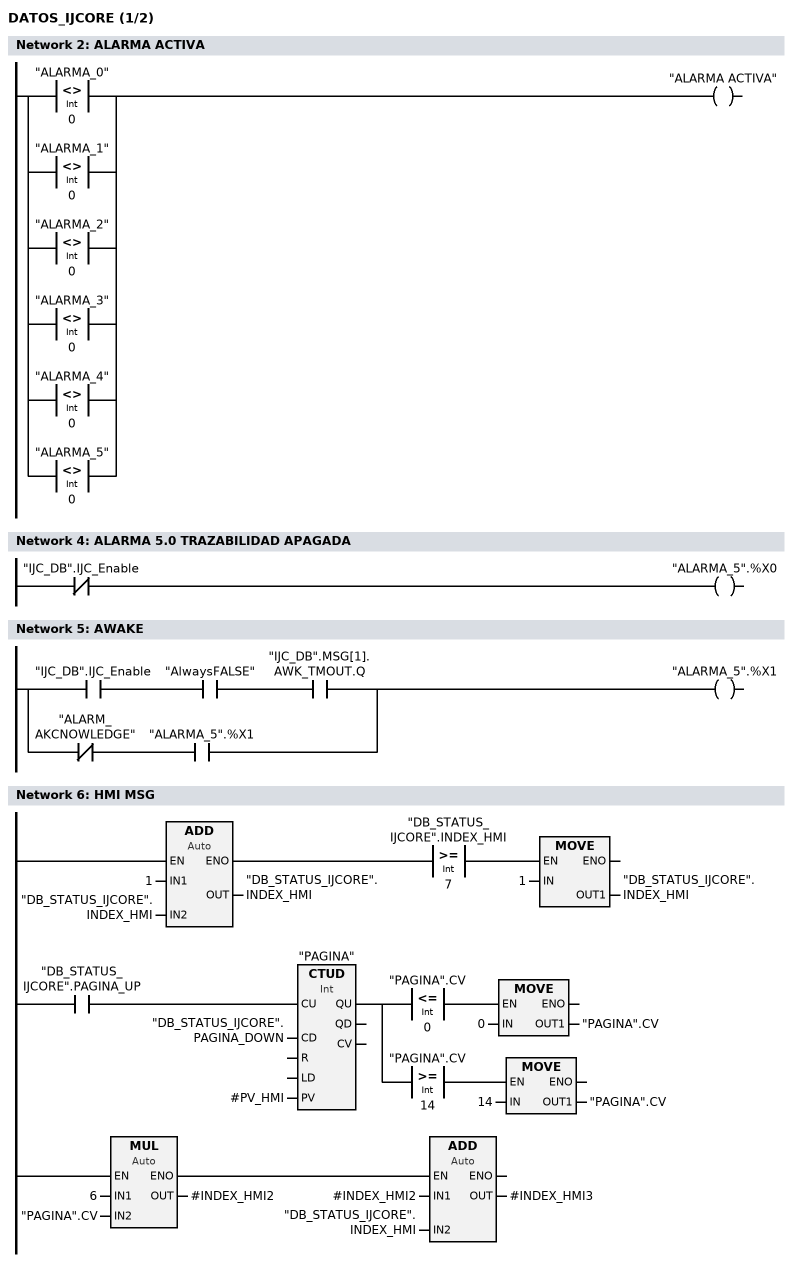
   RUNG wire#powerrail
      { S7_Templates := "SrcType := Int" } NE_Contact(in1 := "ALARMA_0", in2 := 0)
      wire#w1
      Coil( "ALARMA ACTIVA" )
   END_RUNG
   RUNG wire#powerrail
      { S7_Templates := "SrcType := Int" } NE_Contact(in1 := "ALARMA_1", in2 := 0)
   END_RUNG wire#w1
   RUNG wire#powerrail
      { S7_Templates := "SrcType := Int" } NE_Contact(in1 := "ALARMA_2", in2 := 0)
   END_RUNG wire#w1
   RUNG wire#powerrail
      { S7_Templates := "SrcType := Int" } NE_Contact(in1 := "ALARMA_3", in2 := 0)
   END_RUNG wire#w1
   RUNG wire#powerrail
      { S7_Templates := "SrcType := Int" } NE_Contact(in1 := "ALARMA_4", in2 := 0)
   END_RUNG wire#w1
   RUNG wire#powerrail
      { S7_Templates := "SrcType := Int" } NE_Contact(in1 := "ALARMA_5", in2 := 0)
   END_RUNG wire#w1
   // the same network as SCL:
   "ALARMA ACTIVA" := ("ALARMA_0" <> 0) OR ("ALARMA_1" <> 0) OR ("ALARMA_2" <> 0) OR ("ALARMA_3" <> 0) OR ("ALARMA_4" <> 0) OR ("ALARMA_5" <> 0);
END_REGION

REGION Network 3 (SCL): ALARMAS IJCORE

   //////// MESAGE ALARMS /////////
   //
   //Alarm AWAKE  error
   //
   IF "IJC_DB".AWAKE_SIGNAL_INSTANCE.AwSignalTimeOutFault AND"IJC_DB".IJC_Enable THEN
       "Alarms".Alarm[127] := true;
   ELSE
       "Alarms".Alarm[127] := FALSE;
   END_IF;

   CASE "DB_ProductionProgramActual".Program.MechanicalType OF
       1:

           //Alarm IJC STA SIDE MEMBER LH  error
           //
           IF "IJC_DB".MSG[1].DN AND "DB_STATUS_IJCORE".ANSWER_STA[1] = -2
               AND "IJC_DB".IJC_Enable AND "DB_ProductionProgramActual".Program.MechanicalType = 1 THEN
               "Alarms".Alarm[130] := true;
           ELSE
               "Alarms".Alarm[130] := FALSE;
           END_IF;

           IF "IJC_DB".MSG[1].DN AND "DB_STATUS_IJCORE".ANSWER_STA[1] = -10
               AND "IJC_DB".IJC_Enable AND "DB_ProductionProgramActual".Program.MechanicalType = 1 THEN
               "Alarms".Alarm[150] := true;
           ELSE
               "Alarms".Alarm[150] := FALSE;
           END_IF;

           IF "IJC_DB".MSG[1].DN AND "DB_STATUS_IJCORE".ANSWER_STA[1] = -16
               AND "IJC_DB".IJC_Enable AND "DB_ProductionProgramActual".Program.MechanicalType = 1 THEN
               "Alarms".Alarm[151] := true;
           ELSE
               "Alarms".Alarm[151] := FALSE;
           END_IF;

           IF "IJC_DB".MSG[1].DN AND "DB_STATUS_IJCORE".ANSWER_STA[1] = 8224
               AND "IJC_DB".IJC_Enable AND "DB_ProductionProgramActual".Program.MechanicalType = 1 THEN
               "Alarms".Alarm[152] := true;
           ELSE
               "Alarms".Alarm[152] := FALSE;
           END_IF;

           //Alarm IJC STA SIDE MEMBER RH  error
           //
           IF "IJC_DB".MSG[2].DN AND "DB_STATUS_IJCORE".ANSWER_STA[2] = -2
               AND "IJC_DB".IJC_Enable THEN
               "Alarms".Alarm[131] := true;
           ELSE
               "Alarms".Alarm[131] := FALSE;
           END_IF;

           IF "IJC_DB".MSG[2].DN AND "DB_STATUS_IJCORE".ANSWER_STA[2] = -10
               AND "IJC_DB".IJC_Enable THEN
               "Alarms".Alarm[153] := true;
           ELSE
               "Alarms".Alarm[153] := FALSE;
           END_IF;

           IF "IJC_DB".MSG[2].DN AND "DB_STATUS_IJCORE".ANSWER_STA[2] = -16
               AND "IJC_DB".IJC_Enable THEN
               "Alarms".Alarm[154] := true;
           ELSE
               "Alarms".Alarm[154] := FALSE;
           END_IF;

           IF "IJC_DB".MSG[2].DN AND "DB_STATUS_IJCORE".ANSWER_STA[2] = 8224
               AND "IJC_DB".IJC_Enable THEN
               "Alarms".Alarm[155] := true;
           ELSE
               "Alarms".Alarm[155] := FALSE;
           END_IF;
       0:

           //Alarm IJC STA SIDE MEMBER LH  error
           //
           IF "IJC_DB".MSG[1].DN AND "DB_STATUS_IJCORE".ANSWER_STA[1] = -2
               AND "IJC_DB".IJC_Enable AND "DB_ProductionProgramActual".Program.MechanicalType = 1 THEN
               "Alarms".Alarm[131] := true;
           ELSE
               "Alarms".Alarm[131] := FALSE;
           END_IF;

           IF "IJC_DB".MSG[1].DN AND "DB_STATUS_IJCORE".ANSWER_STA[1] = -10
               AND "IJC_DB".IJC_Enable AND "DB_ProductionProgramActual".Program.MechanicalType = 1 THEN
               "Alarms".Alarm[153] := true;
           ELSE
               "Alarms".Alarm[153] := FALSE;
           END_IF;

           IF "IJC_DB".MSG[1].DN AND "DB_STATUS_IJCORE".ANSWER_STA[1] = -16
               AND "IJC_DB".IJC_Enable AND "DB_ProductionProgramActual".Program.MechanicalType = 1 THEN
               "Alarms".Alarm[154] := true;
           ELSE
               "Alarms".Alarm[154] := FALSE;
           END_IF;

           IF "IJC_DB".MSG[1].DN AND "DB_STATUS_IJCORE".ANSWER_STA[1] = 8224
               AND "IJC_DB".IJC_Enable AND "DB_ProductionProgramActual".Program.MechanicalType = 1 THEN
               "Alarms".Alarm[155] := true;
           ELSE
               "Alarms".Alarm[155] := FALSE;
           END_IF;

           //Alarm IJC STA SIDE MEMBER RH  error
           //
           IF "IJC_DB".MSG[2].DN AND "DB_STATUS_IJCORE".ANSWER_STA[2] = -2
               AND "IJC_DB".IJC_Enable THEN
               "Alarms".Alarm[130] := true;
           ELSE
               "Alarms".Alarm[130] := FALSE;
           END_IF;

           IF "IJC_DB".MSG[2].DN AND "DB_STATUS_IJCORE".ANSWER_STA[2] = -10
               AND "IJC_DB".IJC_Enable THEN
               "Alarms".Alarm[150] := true;
           ELSE
               "Alarms".Alarm[150] := FALSE;
           END_IF;

           IF "IJC_DB".MSG[2].DN AND "DB_STATUS_IJCORE".ANSWER_STA[2] = -16
               AND "IJC_DB".IJC_Enable THEN
               "Alarms".Alarm[151] := true;
           ELSE
               "Alarms".Alarm[151] := FALSE;
           END_IF;

           IF "IJC_DB".MSG[2].DN AND "DB_STATUS_IJCORE".ANSWER_STA[2] = 8224
               AND "IJC_DB".IJC_Enable THEN
               "Alarms".Alarm[152] := true;
           ELSE
               "Alarms".Alarm[152] := FALSE;
           END_IF;
   END_CASE;

   //Alarm IJC STA FRONT TUBE  error
   //
   IF "IJC_DB".MSG[3].DN AND "DB_STATUS_IJCORE".ANSWER_STA[3] = -2
       AND "IJC_DB".IJC_Enable THEN
       "Alarms".Alarm[132] := true;
   ELSE
       "Alarms".Alarm[132] := FALSE;
   END_IF;

   IF "IJC_DB".MSG[3].DN AND "DB_STATUS_IJCORE".ANSWER_STA[3] = -10
       AND "IJC_DB".IJC_Enable THEN
       "Alarms".Alarm[156] := true;
   ELSE
       "Alarms".Alarm[156] := FALSE;
   END_IF;

   IF "IJC_DB".MSG[3].DN AND "DB_STATUS_IJCORE".ANSWER_STA[3] = -16
       AND "IJC_DB".IJC_Enable THEN
       "Alarms".Alarm[157] := true;
   ELSE
       "Alarms".Alarm[157] := FALSE;
   END_IF;

   IF "IJC_DB".MSG[3].DN AND "DB_STATUS_IJCORE".ANSWER_STA[3] = 8224
       AND "IJC_DB".IJC_Enable THEN
       "Alarms".Alarm[158] := true;
   ELSE
       "Alarms".Alarm[158] := FALSE;
   END_IF;
   //Alarm IJC STA REAR TUBE  error
   //
   IF "IJC_DB".MSG[4].DN AND "DB_STATUS_IJCORE".ANSWER_STA[4] = -2
       AND "IJC_DB".IJC_Enable THEN
       "Alarms".Alarm[133] := true;
   ELSE
       "Alarms".Alarm[133] := FALSE;
   END_IF;

   IF "IJC_DB".MSG[4].DN AND "DB_STATUS_IJCORE".ANSWER_STA[4] = -10
       AND "IJC_DB".IJC_Enable THEN
       "Alarms".Alarm[159] := true;
   ELSE
       "Alarms".Alarm[159] := FALSE;
   END_IF;

   IF "IJC_DB".MSG[4].DN AND "DB_STATUS_IJCORE".ANSWER_STA[4] = -16
       AND "IJC_DB".IJC_Enable THEN
       "Alarms".Alarm[160] := true;
   ELSE
       "Alarms".Alarm[160] := FALSE;
   END_IF;

   IF "IJC_DB".MSG[4].DN AND "DB_STATUS_IJCORE".ANSWER_STA[4] = 8224
       AND "IJC_DB".IJC_Enable THEN
       "Alarms".Alarm[161] := true;
   ELSE
       "Alarms".Alarm[161] := FALSE;
   END_IF;

   //Alarm IJC TRC SIDE MEMBER LH  error
   //
   IF "IJC_DB".MSG[5].DN AND "DB_STATUS_IJCORE".ANSWER_TRC[1] = -2
       AND "IJC_DB".IJC_Enable AND NOT "M_TRC1_OK" THEN
       "Alarms".Alarm[134] := true;
   ELSE
       "Alarms".Alarm[134] := FALSE;
   END_IF;

   IF "IJC_DB".MSG[5].DN AND "DB_STATUS_IJCORE".ANSWER_TRC[1] = -4
       AND "IJC_DB".IJC_Enable AND NOT "M_TRC1_OK" THEN
       "Alarms".Alarm[162] := true;
   ELSE
       "Alarms".Alarm[162] := FALSE;
   END_IF;

   IF "IJC_DB".MSG[5].DN AND "DB_STATUS_IJCORE".ANSWER_TRC[1] = -16
       AND "IJC_DB".IJC_Enable AND NOT "M_TRC1_OK" THEN
       "Alarms".Alarm[163] := true;
   ELSE
       "Alarms".Alarm[163] := FALSE;
   END_IF;

   IF "IJC_DB".MSG[5].DN AND "DB_STATUS_IJCORE".ANSWER_TRC[1] = 8224
       AND "IJC_DB".IJC_Enable AND NOT "M_TRC1_OK" THEN
       "Alarms".Alarm[146] := true;
   ELSE
       "Alarms".Alarm[146] := FALSE;
   END_IF;

   //Alarm IJC TRC SIDE MEMBER RH  error
   //
   IF "IJC_DB".MSG[6].DN AND "DB_STATUS_IJCORE".ANSWER_TRC[2] = -2
       AND "IJC_DB".IJC_Enable AND NOT "M_TRC2_OK" THEN
       "Alarms".Alarm[135] := true;
   ELSE
       "Alarms".Alarm[135] := FALSE;
   END_IF;

   IF "IJC_DB".MSG[6].DN AND "DB_STATUS_IJCORE".ANSWER_TRC[2] = -4
       AND "IJC_DB".IJC_Enable AND NOT "M_TRC2_OK" THEN
       "Alarms".Alarm[164] := true;
   ELSE
       "Alarms".Alarm[164] := FALSE;
   END_IF;

   IF "IJC_DB".MSG[6].DN AND "DB_STATUS_IJCORE".ANSWER_TRC[2] = -16
       AND "IJC_DB".IJC_Enable AND NOT "M_TRC2_OK" THEN
       "Alarms".Alarm[165] := true;
   ELSE
       "Alarms".Alarm[165] := FALSE;
   END_IF;

   IF "IJC_DB".MSG[6].DN AND "DB_STATUS_IJCORE".ANSWER_TRC[2] = 8224
       AND "IJC_DB".IJC_Enable AND NOT "M_TRC2_OK" THEN
       "Alarms".Alarm[147] := true;
   ELSE
       "Alarms".Alarm[147] := FALSE;
   END_IF;

   //Alarm IJC TRC FRONT TUBE  error
   //
   IF "IJC_DB".MSG[7].DN AND "DB_STATUS_IJCORE".ANSWER_TRC[3] = -2
       AND "IJC_DB".IJC_Enable AND NOT "M_TRC3_OK" THEN
       "Alarms".Alarm[136] := true;
   ELSE
       "Alarms".Alarm[136] := FALSE;
   END_IF;

   IF "IJC_DB".MSG[7].DN AND "DB_STATUS_IJCORE".ANSWER_TRC[3] = -4
       AND "IJC_DB".IJC_Enable AND NOT "M_TRC3_OK" THEN
       "Alarms".Alarm[166] := true;
   ELSE
       "Alarms".Alarm[166] := FALSE;
   END_IF;

   IF "IJC_DB".MSG[7].DN AND "DB_STATUS_IJCORE".ANSWER_TRC[3] = -16
       AND "IJC_DB".IJC_Enable AND NOT "M_TRC3_OK" THEN
       "Alarms".Alarm[167] := true;
   ELSE
       "Alarms".Alarm[167] := FALSE;
   END_IF;

   IF "IJC_DB".MSG[7].DN AND "DB_STATUS_IJCORE".ANSWER_TRC[3] = 8224
       AND "IJC_DB".IJC_Enable AND NOT "M_TRC3_OK" THEN
       "Alarms".Alarm[148] := true;
   ELSE
       "Alarms".Alarm[148] := FALSE;
   END_IF;
   //Alarm IJC TRC REAR TUBE  error
   //
   IF "IJC_DB".MSG[8].DN AND "DB_STATUS_IJCORE".ANSWER_TRC[4] = -2
       AND "IJC_DB".IJC_Enable AND NOT "M_TRC4_OK" THEN
       "Alarms".Alarm[137] := true;
   ELSE
       "Alarms".Alarm[137] := FALSE;
   END_IF;

   IF "IJC_DB".MSG[8].DN AND "DB_STATUS_IJCORE".ANSWER_TRC[4] = -4
       AND "IJC_DB".IJC_Enable AND NOT "M_TRC4_OK" THEN
       "Alarms".Alarm[168] := true;
   ELSE
       "Alarms".Alarm[168] := FALSE;
   END_IF;

   IF "IJC_DB".MSG[8].DN AND "DB_STATUS_IJCORE".ANSWER_TRC[4] = -16
       AND "IJC_DB".IJC_Enable AND NOT "M_TRC4_OK" THEN
       "Alarms".Alarm[169] := true;
   ELSE
       "Alarms".Alarm[169] := FALSE;
   END_IF;

   IF "IJC_DB".MSG[8].DN AND "DB_STATUS_IJCORE".ANSWER_TRC[4] <> 8224
       AND "IJC_DB".IJC_Enable AND NOT "M_TRC4_OK" THEN
       "Alarms".Alarm[149] := true;
   ELSE
       "Alarms".Alarm[149] := FALSE;
   END_IF;
   //Alarm IJC TRR 1 CUPFORMIG error
   //
   //IF "IJC_DB".MSG[9].DN AND "DB_STATUS_IJCORE".ANSWER_RECIB[9] = -2
      // AND "IJC_DB".IJC_Enable THEN
       //"Alarms".Alarm[122] := true;
   //ELSE
     //  "Alarms".Alarm[122] := FALSE;
   //END_IF;
   //
   ////IF "IJC_DB".MSG[9].DN AND "DB_STATUS_IJCORE".ANSWER_RECIB[9] = -16
   // AND "IJC_DB".IJC_Enable THEN
   //"Alarms".Alarm[122] := true;
   //ELSE
   //  "Alarms".Alarm[122] := FALSE;
   //END_IF;
   //
   //IF "IJC_DB".MSG[9].DN AND "DB_STATUS_IJCORE".ANSWER_RECIB[9] = 8224
   // AND "IJC_DB".IJC_Enable THEN
   //"Alarms".Alarm[122] := true;
   //ELSE
   //  "Alarms".Alarm[122] := FALSE;
   //END_IF;

   //Alarm IJC TRR 2 RIVETS error
   //
   //IF "IJC_DB".MSG[10].DN AND "DB_STATUS_IJCORE".ANSWER_RECIB[10] = -2
       //AND "IJC_DB".IJC_Enable THEN
       //"Alarms".Alarm[123] := true;
   //ELSE
     //  "Alarms".Alarm[123] := FALSE;
   //END_IF;
   //
   //IF "IJC_DB".MSG[10].DN AND "DB_STATUS_IJCORE".ANSWER_RECIB[10] = -16
   //AND "IJC_DB".IJC_Enable THEN
   //"Alarms".Alarm[123] := true;
   //ELSE
   //  "Alarms".Alarm[123] := FALSE;
   //END_IF;
   //
   //IF "IJC_DB".MSG[10].DN AND "DB_STATUS_IJCORE".ANSWER_RECIB[10] = 8224
   //AND "IJC_DB".IJC_Enable THEN
   //"Alarms".Alarm[123] := true;
   //ELSE
   //  "Alarms".Alarm[123] := FALSE;
   //END_IF;

   //Alarm IJC CNF SIDE MEMBER LH  error
   //
   //IF "IJC_DB".MSG[11].DN AND "DB_STATUS_IJCORE".ANSWER_RECIB[11] <> 1
     //  AND "IJC_DB".IJC_Enable THEN
     //  "Alarms".Alarm[124] := true;
   //END_IF;
   //

   //
   //IF "IJC_DB".MSG[11].DN AND "DB_STATUS_IJCORE".ANSWER_RECIB[11] = 8224
   //  AND "IJC_DB".IJC_Enable THEN
   //  "Alarms".Alarm[124] := true;
   //END_IF;

   //Alarm IJC CNF SIDE MEMBER RH  error
   //
   //IF "IJC_DB".MSG[12].DN AND "DB_STATUS_IJCORE".ANSWER_RECIB[12] <> 1
     //  AND "IJC_DB".IJC_Enable THEN
       //"Alarms".Alarm[124] := true;
   //END_IF;

   //Alarm IJC CNF REAR TUBE  error
   //
   //IF "IJC_DB".MSG[13].DN AND "DB_STATUS_IJCORE".ANSWER_RECIB[13] <> 1
     //  AND "IJC_DB".IJC_Enable THEN
       //"Alarms".Alarm[125] := true;
   //ELSE
     //  "Alarms".Alarm[125] := FALSE;
   //END_IF;

   //Alarm IJC CNF SIDE MEMBER LH  error
   //
   //IF "IJC_DB".MSG[15].DN AND "DB_STATUS_IJCORE".ANSWER_RECIB[15] <> 1
     //  AND "IJC_DB".IJC_Enable THEN
       //"Alarms".Alarm[126] := true;
   //ELSE
     //  "Alarms".Alarm[126] := FALSE;
   //END_IF;
   //
   //Alarm IJC PFC SIDE MEMBER LH  error
   //
   IF "IJC_DB".MSG[14].DN AND "DB_STATUS_IJCORE".ANSWER_RECIB[14] = -2
       AND "IJC_DB".IJC_Enable AND NOT "M_PFC_OK" THEN
       "Alarms".Alarm[170] := true;
   ELSE
       "Alarms".Alarm[170] := FALSE;
   END_IF;

   IF "IJC_DB".MSG[14].DN AND "DB_STATUS_IJCORE".ANSWER_RECIB[14] = -4
       AND "IJC_DB".IJC_Enable AND NOT "M_PFC_OK" THEN
       "Alarms".Alarm[143] := true;
   ELSE
       "Alarms".Alarm[143] := FALSE;
   END_IF;

   IF "IJC_DB".MSG[14].DN AND "DB_STATUS_IJCORE".ANSWER_RECIB[14] = -10
       AND "IJC_DB".IJC_Enable AND NOT "M_PFC_OK" THEN
      "Alarms".Alarm[171] := true;
   ELSE
     "Alarms".Alarm[171] := FALSE;
   END_IF;


   IF "IJC_DB".MSG[14].DN AND "DB_STATUS_IJCORE".ANSWER_RECIB[14] = -16
       AND "IJC_DB".IJC_Enable AND NOT "M_PFC_OK" THEN
     "Alarms".Alarm[172] := true;
   ELSE
       "Alarms".Alarm[172] := FALSE;
   END_IF;

   IF "IJC_DB".MSG[14].DN AND "DB_STATUS_IJCORE".ANSWER_RECIB[14] = 8224
       AND "IJC_DB".IJC_Enable AND NOT "M_PFC_OK" THEN
       "Alarms".Alarm[145] := true;
   ELSE
       "Alarms".Alarm[145] := FALSE;
   END_IF;
END_REGION

REGION Network 4: ALARMA 5.0 TRAZABILIDAD APAGADA
   RUNG wire#powerrail
      I_Contact( "IJC_DB".IJC_Enable )
      Coil( "ALARMA_5".%X0 )
   END_RUNG
   // the same network as SCL:
   "ALARMA_5".%X0 := NOT "IJC_DB".IJC_Enable;
END_REGION

REGION Network 5: AWAKE
   RUNG wire#powerrail
      Contact( "IJC_DB".IJC_Enable )
      Contact( "AlwaysFALSE" )
      Contact( "IJC_DB".MSG[1].AWK_TMOUT.Q )
      wire#w1
      Coil( "ALARMA_5".%X1 )
   END_RUNG
   RUNG wire#powerrail
      I_Contact( "ALARM_AKCNOWLEDGE" )
      Contact( "ALARMA_5".%X1 )
   END_RUNG wire#w1
   // the same network as SCL:
   "ALARMA_5".%X1 := ("IJC_DB".IJC_Enable AND "AlwaysFALSE" AND "IJC_DB".MSG[1].AWK_TMOUT.Q) OR (NOT "ALARM_AKCNOWLEDGE" AND "ALARMA_5".%X1);
END_REGION

REGION Network 6: HMI MSG
   RUNG wire#powerrail
      Add(in1 := 1, in2 := "DB_STATUS_IJCORE".INDEX_HMI, out => "DB_STATUS_IJCORE".INDEX_HMI)
      { S7_Templates := "SrcType := Int" } GE_Contact(in1 := "DB_STATUS_IJCORE".INDEX_HMI, in2 := 7)
      Move(in := 1, out1 => "DB_STATUS_IJCORE".INDEX_HMI)
   END_RUNG
   RUNG wire#powerrail
      Contact( "DB_STATUS_IJCORE".PAGINA_UP )
      { S7_Templates := "value_type := Int" } "PAGINA".CTUD(cd := "DB_STATUS_IJCORE".PAGINA_DOWN, r :=, ld :=, pv := #PV_HMI, qd =>, cv =>)
      wire#w1
      { S7_Templates := "SrcType := Int" } LE_Contact(in1 := "PAGINA".CV, in2 := 0)
      Move(in := 0, out1 => "PAGINA".CV)
   END_RUNG
   RUNG wire#w1
      { S7_Templates := "SrcType := Int" } GE_Contact(in1 := "PAGINA".CV, in2 := 14)
      Move(in := 14, out1 => "PAGINA".CV)
   END_RUNG
   RUNG wire#powerrail
      Mul(in1 := 6, in2 := "PAGINA".CV, out => #INDEX_HMI2)
      Add(in1 := #INDEX_HMI2, in2 := "DB_STATUS_IJCORE".INDEX_HMI, out => #INDEX_HMI3)
   END_RUNG
   // the same network as SCL:
   "DB_STATUS_IJCORE".INDEX_HMI := 1 + "DB_STATUS_IJCORE".INDEX_HMI;
   IF "DB_STATUS_IJCORE".INDEX_HMI >= 7 THEN "DB_STATUS_IJCORE".INDEX_HMI := 1; END_IF;
   "PAGINA".CTUD(CU := "DB_STATUS_IJCORE".PAGINA_UP, CD := "DB_STATUS_IJCORE".PAGINA_DOWN, PV := #PV_HMI);
   #_w1 := "PAGINA".QU;
   IF "PAGINA".QU AND ("PAGINA".CV <= 0) THEN "PAGINA".CV := 0; END_IF;
   IF #_w1 AND ("PAGINA".CV >= 14) THEN "PAGINA".CV := 14; END_IF;
   #INDEX_HMI2 := 6 * "PAGINA".CV;
   #INDEX_HMI3 := #INDEX_HMI2 + "DB_STATUS_IJCORE".INDEX_HMI;
END_REGION

REGION Network 7: VARIABLES HMI
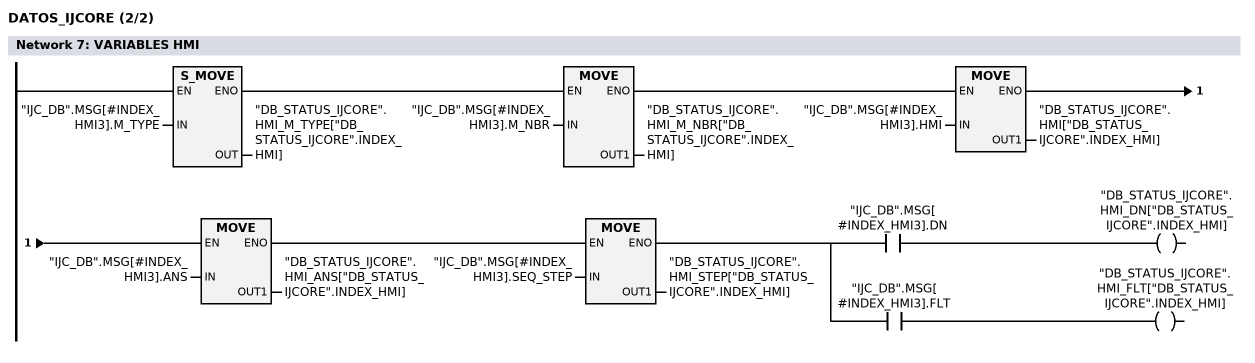
   RUNG wire#powerrail
      S_Move(in := "IJC_DB".MSG[#INDEX_HMI3].M_TYPE, out => "DB_STATUS_IJCORE".HMI_M_TYPE["DB_STATUS_IJCORE".INDEX_HMI])
      Move(in := "IJC_DB".MSG[#INDEX_HMI3].M_NBR, out1 => "DB_STATUS_IJCORE".HMI_M_NBR["DB_STATUS_IJCORE".INDEX_HMI])
      Move(in := "IJC_DB".MSG[#INDEX_HMI3].HMI, out1 => "DB_STATUS_IJCORE".HMI["DB_STATUS_IJCORE".INDEX_HMI])
      Move(in := "IJC_DB".MSG[#INDEX_HMI3].ANS, out1 => "DB_STATUS_IJCORE".HMI_ANS["DB_STATUS_IJCORE".INDEX_HMI])
      Move(in := "IJC_DB".MSG[#INDEX_HMI3].SEQ_STEP, out1 => "DB_STATUS_IJCORE".HMI_STEP["DB_STATUS_IJCORE".INDEX_HMI])
      wire#w1
      Contact( "IJC_DB".MSG[#INDEX_HMI3].DN )
      Coil( "DB_STATUS_IJCORE".HMI_DN["DB_STATUS_IJCORE".INDEX_HMI] )
   END_RUNG
   RUNG wire#w1
      Contact( "IJC_DB".MSG[#INDEX_HMI3].FLT )
      Coil( "DB_STATUS_IJCORE".HMI_FLT["DB_STATUS_IJCORE".INDEX_HMI] )
   END_RUNG
   // the same network as SCL:
   "DB_STATUS_IJCORE".HMI_M_TYPE["DB_STATUS_IJCORE".INDEX_HMI] := "IJC_DB".MSG[#INDEX_HMI3].M_TYPE;
   "DB_STATUS_IJCORE".HMI_M_NBR["DB_STATUS_IJCORE".INDEX_HMI] := "IJC_DB".MSG[#INDEX_HMI3].M_NBR;
   "DB_STATUS_IJCORE".HMI["DB_STATUS_IJCORE".INDEX_HMI] := "IJC_DB".MSG[#INDEX_HMI3].HMI;
   "DB_STATUS_IJCORE".HMI_ANS["DB_STATUS_IJCORE".INDEX_HMI] := "IJC_DB".MSG[#INDEX_HMI3].ANS;
   "DB_STATUS_IJCORE".HMI_STEP["DB_STATUS_IJCORE".INDEX_HMI] := "IJC_DB".MSG[#INDEX_HMI3].SEQ_STEP;
   "DB_STATUS_IJCORE".HMI_DN["DB_STATUS_IJCORE".INDEX_HMI] := "IJC_DB".MSG[#INDEX_HMI3].DN;
   "DB_STATUS_IJCORE".HMI_FLT["DB_STATUS_IJCORE".INDEX_HMI] := "IJC_DB".MSG[#INDEX_HMI3].FLT;
END_REGION
END_FUNCTION

FUNCTION "FC_CONFIG_MSG_IJC" : Void   // FC2, LAD
{ S7_Optimized_Access := 'TRUE' }
VERSION : 0.1
// stored: AutoNumber true, IsIECCheckEnabled false, SetENOAutomatically false, UDAEnableTagReadback false
   VAR_TEMP
      STRING_USER1 : String;
      STRING_USER2 : String;
      STRING_CORDON_1 : String;
      INDEX_IJC_CORDON : Int;
      STRING_CORDONES : Array[0..13] of String;
   END_VAR
   VAR_TEMP   // added for the SCL form of the ladder/FBD networks
      _w1 : Bool;
      _w2 : Bool;
   END_VAR
BEGIN

REGION Network 1: INDEX MSG CONFIG
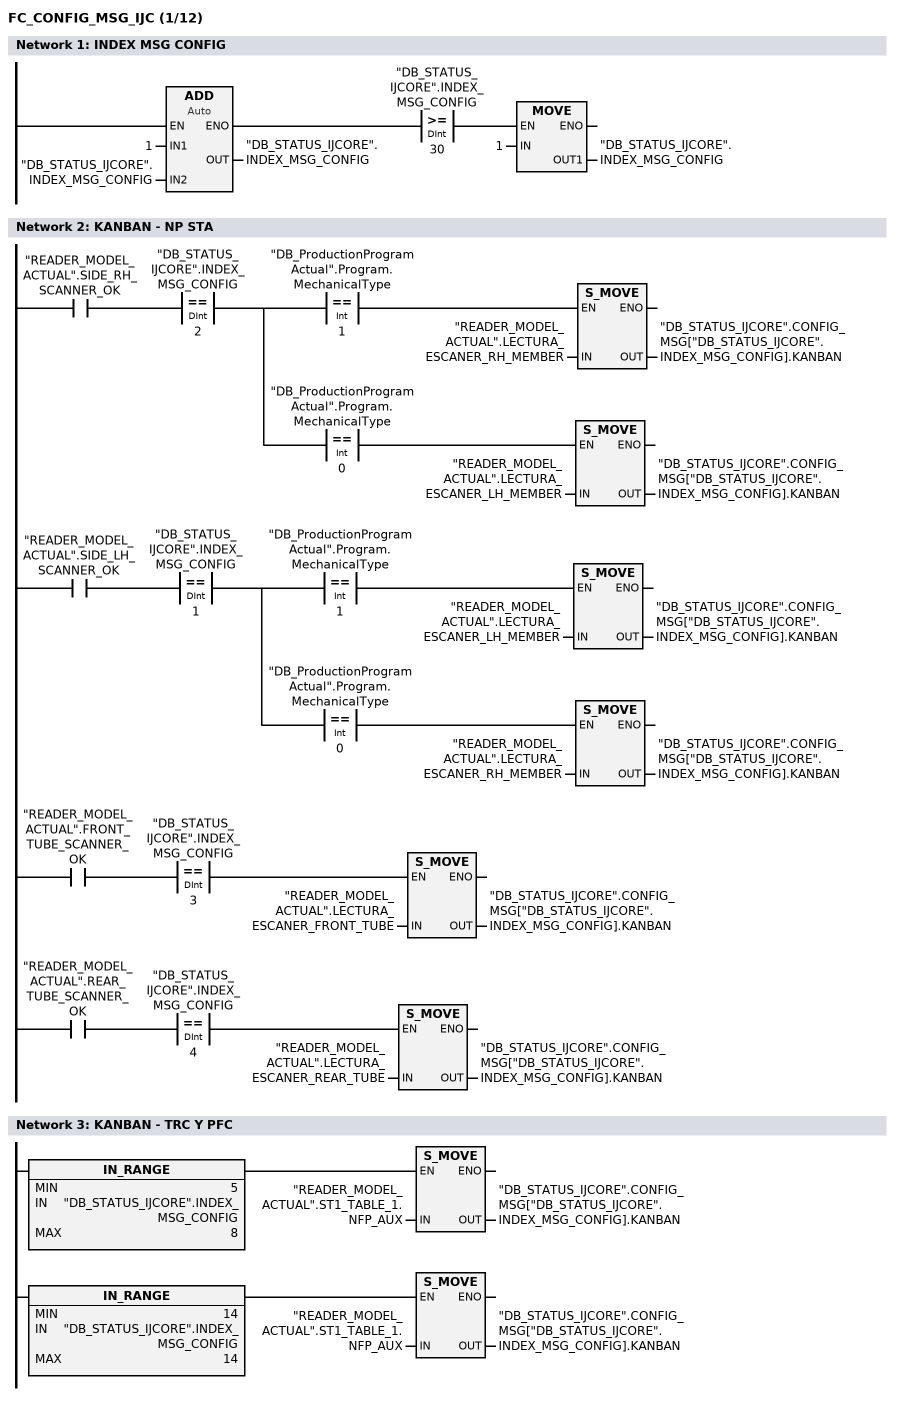
   RUNG wire#powerrail
      Add(in1 := 1, in2 := "DB_STATUS_IJCORE".INDEX_MSG_CONFIG, out => "DB_STATUS_IJCORE".INDEX_MSG_CONFIG)
      { S7_Templates := "SrcType := DInt" } GE_Contact(in1 := "DB_STATUS_IJCORE".INDEX_MSG_CONFIG, in2 := 30)
      Move(in := 1, out1 => "DB_STATUS_IJCORE".INDEX_MSG_CONFIG)
   END_RUNG
   // the same network as SCL:
   "DB_STATUS_IJCORE".INDEX_MSG_CONFIG := 1 + "DB_STATUS_IJCORE".INDEX_MSG_CONFIG;
   IF "DB_STATUS_IJCORE".INDEX_MSG_CONFIG >= 30 THEN "DB_STATUS_IJCORE".INDEX_MSG_CONFIG := 1; END_IF;
END_REGION

REGION Network 2: KANBAN - NP STA
   RUNG wire#powerrail
      Contact( "READER_MODEL_ACTUAL".SIDE_RH_SCANNER_OK )
      { S7_Templates := "SrcType := DInt" } EQ_Contact(in1 := "DB_STATUS_IJCORE".INDEX_MSG_CONFIG, in2 := 2)
      wire#w1
      { S7_Templates := "SrcType := Int" } EQ_Contact(in1 := "DB_ProductionProgramActual".Program.MechanicalType, in2 := 1)
      S_Move(in := "READER_MODEL_ACTUAL".LECTURA_ESCANER_RH_MEMBER, out => "DB_STATUS_IJCORE".CONFIG_MSG["DB_STATUS_IJCORE".INDEX_MSG_CONFIG].KANBAN)
   END_RUNG
   RUNG wire#w1
      { S7_Templates := "SrcType := Int" } EQ_Contact(in1 := "DB_ProductionProgramActual".Program.MechanicalType, in2 := 0)
      S_Move(in := "READER_MODEL_ACTUAL".LECTURA_ESCANER_LH_MEMBER, out => "DB_STATUS_IJCORE".CONFIG_MSG["DB_STATUS_IJCORE".INDEX_MSG_CONFIG].KANBAN)
   END_RUNG
   RUNG wire#powerrail
      Contact( "READER_MODEL_ACTUAL".SIDE_LH_SCANNER_OK )
      { S7_Templates := "SrcType := DInt" } EQ_Contact(in1 := "DB_STATUS_IJCORE".INDEX_MSG_CONFIG, in2 := 1)
      wire#w2
      { S7_Templates := "SrcType := Int" } EQ_Contact(in1 := "DB_ProductionProgramActual".Program.MechanicalType, in2 := 1)
      S_Move(in := "READER_MODEL_ACTUAL".LECTURA_ESCANER_LH_MEMBER, out => "DB_STATUS_IJCORE".CONFIG_MSG["DB_STATUS_IJCORE".INDEX_MSG_CONFIG].KANBAN)
   END_RUNG
   RUNG wire#w2
      { S7_Templates := "SrcType := Int" } EQ_Contact(in1 := "DB_ProductionProgramActual".Program.MechanicalType, in2 := 0)
      S_Move(in := "READER_MODEL_ACTUAL".LECTURA_ESCANER_RH_MEMBER, out => "DB_STATUS_IJCORE".CONFIG_MSG["DB_STATUS_IJCORE".INDEX_MSG_CONFIG].KANBAN)
   END_RUNG
   RUNG wire#powerrail
      Contact( "READER_MODEL_ACTUAL".FRONT_TUBE_SCANNER_OK )
      { S7_Templates := "SrcType := DInt" } EQ_Contact(in1 := "DB_STATUS_IJCORE".INDEX_MSG_CONFIG, in2 := 3)
      S_Move(in := "READER_MODEL_ACTUAL".LECTURA_ESCANER_FRONT_TUBE, out => "DB_STATUS_IJCORE".CONFIG_MSG["DB_STATUS_IJCORE".INDEX_MSG_CONFIG].KANBAN)
   END_RUNG
   RUNG wire#powerrail
      Contact( "READER_MODEL_ACTUAL".REAR_TUBE_SCANNER_OK )
      { S7_Templates := "SrcType := DInt" } EQ_Contact(in1 := "DB_STATUS_IJCORE".INDEX_MSG_CONFIG, in2 := 4)
      S_Move(in := "READER_MODEL_ACTUAL".LECTURA_ESCANER_REAR_TUBE, out => "DB_STATUS_IJCORE".CONFIG_MSG["DB_STATUS_IJCORE".INDEX_MSG_CONFIG].KANBAN)
   END_RUNG
   // the same network as SCL:
   #_w1 := "READER_MODEL_ACTUAL".SIDE_RH_SCANNER_OK AND ("DB_STATUS_IJCORE".INDEX_MSG_CONFIG = 2);
   IF #_w1 AND ("DB_ProductionProgramActual".Program.MechanicalType = 1) THEN
       "DB_STATUS_IJCORE".CONFIG_MSG["DB_STATUS_IJCORE".INDEX_MSG_CONFIG].KANBAN := "READER_MODEL_ACTUAL".LECTURA_ESCANER_RH_MEMBER;
   END_IF;
   IF #_w1 AND ("DB_ProductionProgramActual".Program.MechanicalType = 0) THEN
       "DB_STATUS_IJCORE".CONFIG_MSG["DB_STATUS_IJCORE".INDEX_MSG_CONFIG].KANBAN := "READER_MODEL_ACTUAL".LECTURA_ESCANER_LH_MEMBER;
   END_IF;
   #_w2 := "READER_MODEL_ACTUAL".SIDE_LH_SCANNER_OK AND ("DB_STATUS_IJCORE".INDEX_MSG_CONFIG = 1);
   IF #_w2 AND ("DB_ProductionProgramActual".Program.MechanicalType = 1) THEN
       "DB_STATUS_IJCORE".CONFIG_MSG["DB_STATUS_IJCORE".INDEX_MSG_CONFIG].KANBAN := "READER_MODEL_ACTUAL".LECTURA_ESCANER_LH_MEMBER;
   END_IF;
   IF #_w2 AND ("DB_ProductionProgramActual".Program.MechanicalType = 0) THEN
       "DB_STATUS_IJCORE".CONFIG_MSG["DB_STATUS_IJCORE".INDEX_MSG_CONFIG].KANBAN := "READER_MODEL_ACTUAL".LECTURA_ESCANER_RH_MEMBER;
   END_IF;
   IF "READER_MODEL_ACTUAL".FRONT_TUBE_SCANNER_OK AND ("DB_STATUS_IJCORE".INDEX_MSG_CONFIG = 3) THEN
       "DB_STATUS_IJCORE".CONFIG_MSG["DB_STATUS_IJCORE".INDEX_MSG_CONFIG].KANBAN := "READER_MODEL_ACTUAL".LECTURA_ESCANER_FRONT_TUBE;
   END_IF;
   IF "READER_MODEL_ACTUAL".REAR_TUBE_SCANNER_OK AND ("DB_STATUS_IJCORE".INDEX_MSG_CONFIG = 4) THEN
       "DB_STATUS_IJCORE".CONFIG_MSG["DB_STATUS_IJCORE".INDEX_MSG_CONFIG].KANBAN := "READER_MODEL_ACTUAL".LECTURA_ESCANER_REAR_TUBE;
   END_IF;
END_REGION

REGION Network 3: KANBAN - TRC Y PFC
   RUNG wire#powerrail
      { S7_Templates := "SrcType := DInt" } InRange(min := 5, in := "DB_STATUS_IJCORE".INDEX_MSG_CONFIG, max := 8)
      S_Move(in := "READER_MODEL_ACTUAL".ST1_TABLE_1.NFP_AUX, out => "DB_STATUS_IJCORE".CONFIG_MSG["DB_STATUS_IJCORE".INDEX_MSG_CONFIG].KANBAN)
   END_RUNG
   RUNG wire#powerrail
      { S7_Templates := "SrcType := DInt" } InRange(min := 14, in := "DB_STATUS_IJCORE".INDEX_MSG_CONFIG, max := 14)
      S_Move(in := "READER_MODEL_ACTUAL".ST1_TABLE_1.NFP_AUX, out => "DB_STATUS_IJCORE".CONFIG_MSG["DB_STATUS_IJCORE".INDEX_MSG_CONFIG].KANBAN)
   END_RUNG
   // the same network as SCL:
   IF (5 <= "DB_STATUS_IJCORE".INDEX_MSG_CONFIG) AND ("DB_STATUS_IJCORE".INDEX_MSG_CONFIG <= 8) THEN
       "DB_STATUS_IJCORE".CONFIG_MSG["DB_STATUS_IJCORE".INDEX_MSG_CONFIG].KANBAN := "READER_MODEL_ACTUAL".ST1_TABLE_1.NFP_AUX;
   END_IF;
   IF (14 <= "DB_STATUS_IJCORE".INDEX_MSG_CONFIG) AND ("DB_STATUS_IJCORE".INDEX_MSG_CONFIG <= 14) THEN
       "DB_STATUS_IJCORE".CONFIG_MSG["DB_STATUS_IJCORE".INDEX_MSG_CONFIG].KANBAN := "READER_MODEL_ACTUAL".ST1_TABLE_1.NFP_AUX;
   END_IF;
END_REGION

REGION Network 4: KANBAN - TRR Y CNF
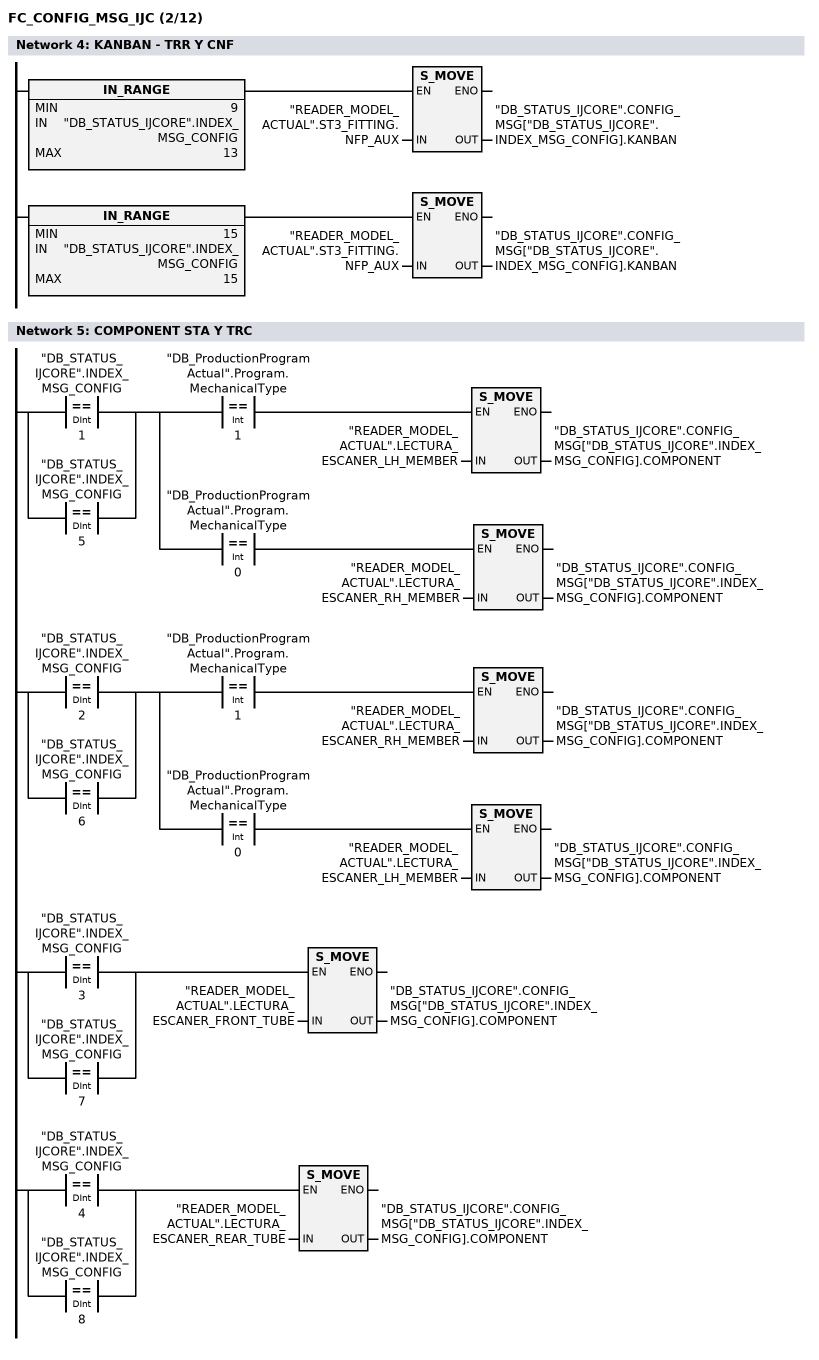
   RUNG wire#powerrail
      { S7_Templates := "SrcType := DInt" } InRange(min := 9, in := "DB_STATUS_IJCORE".INDEX_MSG_CONFIG, max := 13)
      S_Move(in := "READER_MODEL_ACTUAL".ST3_FITTING.NFP_AUX, out => "DB_STATUS_IJCORE".CONFIG_MSG["DB_STATUS_IJCORE".INDEX_MSG_CONFIG].KANBAN)
   END_RUNG
   RUNG wire#powerrail
      { S7_Templates := "SrcType := DInt" } InRange(min := 15, in := "DB_STATUS_IJCORE".INDEX_MSG_CONFIG, max := 15)
      S_Move(in := "READER_MODEL_ACTUAL".ST3_FITTING.NFP_AUX, out => "DB_STATUS_IJCORE".CONFIG_MSG["DB_STATUS_IJCORE".INDEX_MSG_CONFIG].KANBAN)
   END_RUNG
   // the same network as SCL:
   IF (9 <= "DB_STATUS_IJCORE".INDEX_MSG_CONFIG) AND ("DB_STATUS_IJCORE".INDEX_MSG_CONFIG <= 13) THEN
       "DB_STATUS_IJCORE".CONFIG_MSG["DB_STATUS_IJCORE".INDEX_MSG_CONFIG].KANBAN := "READER_MODEL_ACTUAL".ST3_FITTING.NFP_AUX;
   END_IF;
   IF (15 <= "DB_STATUS_IJCORE".INDEX_MSG_CONFIG) AND ("DB_STATUS_IJCORE".INDEX_MSG_CONFIG <= 15) THEN
       "DB_STATUS_IJCORE".CONFIG_MSG["DB_STATUS_IJCORE".INDEX_MSG_CONFIG].KANBAN := "READER_MODEL_ACTUAL".ST3_FITTING.NFP_AUX;
   END_IF;
END_REGION

REGION Network 5: COMPONENT STA Y TRC
   RUNG wire#powerrail
      { S7_Templates := "SrcType := DInt" } EQ_Contact(in1 := "DB_STATUS_IJCORE".INDEX_MSG_CONFIG, in2 := 1)
      wire#w1
      { S7_Templates := "SrcType := Int" } EQ_Contact(in1 := "DB_ProductionProgramActual".Program.MechanicalType, in2 := 1)
      S_Move(in := "READER_MODEL_ACTUAL".LECTURA_ESCANER_LH_MEMBER, out => "DB_STATUS_IJCORE".CONFIG_MSG["DB_STATUS_IJCORE".INDEX_MSG_CONFIG].COMPONENT)
   END_RUNG
   RUNG wire#powerrail
      { S7_Templates := "SrcType := DInt" } EQ_Contact(in1 := "DB_STATUS_IJCORE".INDEX_MSG_CONFIG, in2 := 5)
   END_RUNG wire#w1
   RUNG wire#w1
      { S7_Templates := "SrcType := Int" } EQ_Contact(in1 := "DB_ProductionProgramActual".Program.MechanicalType, in2 := 0)
      S_Move(in := "READER_MODEL_ACTUAL".LECTURA_ESCANER_RH_MEMBER, out => "DB_STATUS_IJCORE".CONFIG_MSG["DB_STATUS_IJCORE".INDEX_MSG_CONFIG].COMPONENT)
   END_RUNG
   RUNG wire#powerrail
      { S7_Templates := "SrcType := DInt" } EQ_Contact(in1 := "DB_STATUS_IJCORE".INDEX_MSG_CONFIG, in2 := 2)
      wire#w2
      { S7_Templates := "SrcType := Int" } EQ_Contact(in1 := "DB_ProductionProgramActual".Program.MechanicalType, in2 := 1)
      S_Move(in := "READER_MODEL_ACTUAL".LECTURA_ESCANER_RH_MEMBER, out => "DB_STATUS_IJCORE".CONFIG_MSG["DB_STATUS_IJCORE".INDEX_MSG_CONFIG].COMPONENT)
   END_RUNG
   RUNG wire#powerrail
      { S7_Templates := "SrcType := DInt" } EQ_Contact(in1 := "DB_STATUS_IJCORE".INDEX_MSG_CONFIG, in2 := 6)
   END_RUNG wire#w2
   RUNG wire#w2
      { S7_Templates := "SrcType := Int" } EQ_Contact(in1 := "DB_ProductionProgramActual".Program.MechanicalType, in2 := 0)
      S_Move(in := "READER_MODEL_ACTUAL".LECTURA_ESCANER_LH_MEMBER, out => "DB_STATUS_IJCORE".CONFIG_MSG["DB_STATUS_IJCORE".INDEX_MSG_CONFIG].COMPONENT)
   END_RUNG
   RUNG wire#powerrail
      { S7_Templates := "SrcType := DInt" } EQ_Contact(in1 := "DB_STATUS_IJCORE".INDEX_MSG_CONFIG, in2 := 3)
      wire#w3
      S_Move(in := "READER_MODEL_ACTUAL".LECTURA_ESCANER_FRONT_TUBE, out => "DB_STATUS_IJCORE".CONFIG_MSG["DB_STATUS_IJCORE".INDEX_MSG_CONFIG].COMPONENT)
   END_RUNG
   RUNG wire#powerrail
      { S7_Templates := "SrcType := DInt" } EQ_Contact(in1 := "DB_STATUS_IJCORE".INDEX_MSG_CONFIG, in2 := 7)
   END_RUNG wire#w3
   RUNG wire#powerrail
      { S7_Templates := "SrcType := DInt" } EQ_Contact(in1 := "DB_STATUS_IJCORE".INDEX_MSG_CONFIG, in2 := 4)
      wire#w4
      S_Move(in := "READER_MODEL_ACTUAL".LECTURA_ESCANER_REAR_TUBE, out => "DB_STATUS_IJCORE".CONFIG_MSG["DB_STATUS_IJCORE".INDEX_MSG_CONFIG].COMPONENT)
   END_RUNG
   RUNG wire#powerrail
      { S7_Templates := "SrcType := DInt" } EQ_Contact(in1 := "DB_STATUS_IJCORE".INDEX_MSG_CONFIG, in2 := 8)
   END_RUNG wire#w4
   // the same network as SCL:
   #_w1 := ("DB_STATUS_IJCORE".INDEX_MSG_CONFIG = 1) OR ("DB_STATUS_IJCORE".INDEX_MSG_CONFIG = 5);
   IF #_w1 AND ("DB_ProductionProgramActual".Program.MechanicalType = 1) THEN
       "DB_STATUS_IJCORE".CONFIG_MSG["DB_STATUS_IJCORE".INDEX_MSG_CONFIG].COMPONENT := "READER_MODEL_ACTUAL".LECTURA_ESCANER_LH_MEMBER;
   END_IF;
   IF #_w1 AND ("DB_ProductionProgramActual".Program.MechanicalType = 0) THEN
       "DB_STATUS_IJCORE".CONFIG_MSG["DB_STATUS_IJCORE".INDEX_MSG_CONFIG].COMPONENT := "READER_MODEL_ACTUAL".LECTURA_ESCANER_RH_MEMBER;
   END_IF;
   #_w2 := ("DB_STATUS_IJCORE".INDEX_MSG_CONFIG = 2) OR ("DB_STATUS_IJCORE".INDEX_MSG_CONFIG = 6);
   IF #_w2 AND ("DB_ProductionProgramActual".Program.MechanicalType = 1) THEN
       "DB_STATUS_IJCORE".CONFIG_MSG["DB_STATUS_IJCORE".INDEX_MSG_CONFIG].COMPONENT := "READER_MODEL_ACTUAL".LECTURA_ESCANER_RH_MEMBER;
   END_IF;
   IF #_w2 AND ("DB_ProductionProgramActual".Program.MechanicalType = 0) THEN
       "DB_STATUS_IJCORE".CONFIG_MSG["DB_STATUS_IJCORE".INDEX_MSG_CONFIG].COMPONENT := "READER_MODEL_ACTUAL".LECTURA_ESCANER_LH_MEMBER;
   END_IF;
   IF ("DB_STATUS_IJCORE".INDEX_MSG_CONFIG = 3) OR ("DB_STATUS_IJCORE".INDEX_MSG_CONFIG = 7) THEN
       "DB_STATUS_IJCORE".CONFIG_MSG["DB_STATUS_IJCORE".INDEX_MSG_CONFIG].COMPONENT := "READER_MODEL_ACTUAL".LECTURA_ESCANER_FRONT_TUBE;
   END_IF;
   IF ("DB_STATUS_IJCORE".INDEX_MSG_CONFIG = 4) OR ("DB_STATUS_IJCORE".INDEX_MSG_CONFIG = 8) THEN
       "DB_STATUS_IJCORE".CONFIG_MSG["DB_STATUS_IJCORE".INDEX_MSG_CONFIG].COMPONENT := "READER_MODEL_ACTUAL".LECTURA_ESCANER_REAR_TUBE;
   END_IF;
END_REGION

REGION Network 6: COMPONENT PFC
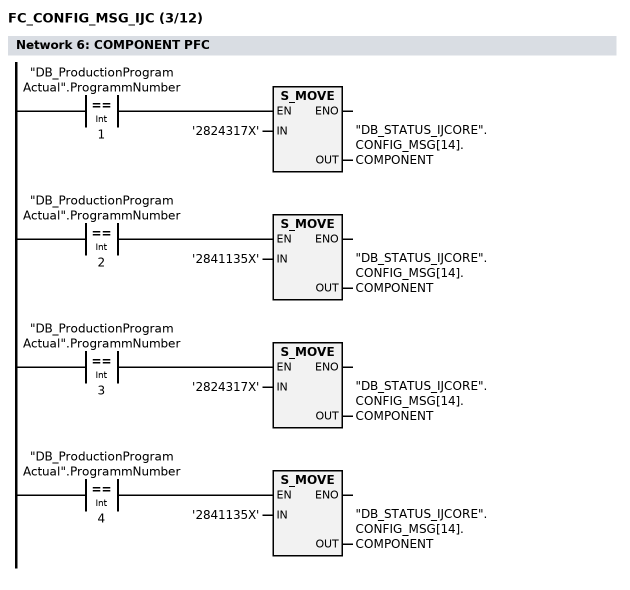
   RUNG wire#powerrail
      { S7_Templates := "SrcType := Int" } EQ_Contact(in1 := "DB_ProductionProgramActual".ProgrammNumber, in2 := 1)
      S_Move(in := '2824317X', out => "DB_STATUS_IJCORE".CONFIG_MSG[14].COMPONENT)
   END_RUNG
   RUNG wire#powerrail
      { S7_Templates := "SrcType := Int" } EQ_Contact(in1 := "DB_ProductionProgramActual".ProgrammNumber, in2 := 2)
      S_Move(in := '2841135X', out => "DB_STATUS_IJCORE".CONFIG_MSG[14].COMPONENT)
   END_RUNG
   RUNG wire#powerrail
      { S7_Templates := "SrcType := Int" } EQ_Contact(in1 := "DB_ProductionProgramActual".ProgrammNumber, in2 := 3)
      S_Move(in := '2824317X', out => "DB_STATUS_IJCORE".CONFIG_MSG[14].COMPONENT)
   END_RUNG
   RUNG wire#powerrail
      { S7_Templates := "SrcType := Int" } EQ_Contact(in1 := "DB_ProductionProgramActual".ProgrammNumber, in2 := 4)
      S_Move(in := '2841135X', out => "DB_STATUS_IJCORE".CONFIG_MSG[14].COMPONENT)
   END_RUNG
   // the same network as SCL:
   IF "DB_ProductionProgramActual".ProgrammNumber = 1 THEN
       "DB_STATUS_IJCORE".CONFIG_MSG[14].COMPONENT := '2824317X';
   END_IF;
   IF "DB_ProductionProgramActual".ProgrammNumber = 2 THEN
       "DB_STATUS_IJCORE".CONFIG_MSG[14].COMPONENT := '2841135X';
   END_IF;
   IF "DB_ProductionProgramActual".ProgrammNumber = 3 THEN
       "DB_STATUS_IJCORE".CONFIG_MSG[14].COMPONENT := '2824317X';
   END_IF;
   IF "DB_ProductionProgramActual".ProgrammNumber = 4 THEN
       "DB_STATUS_IJCORE".CONFIG_MSG[14].COMPONENT := '2841135X';
   END_IF;
END_REGION

REGION Network 7: COMPONENT CNF
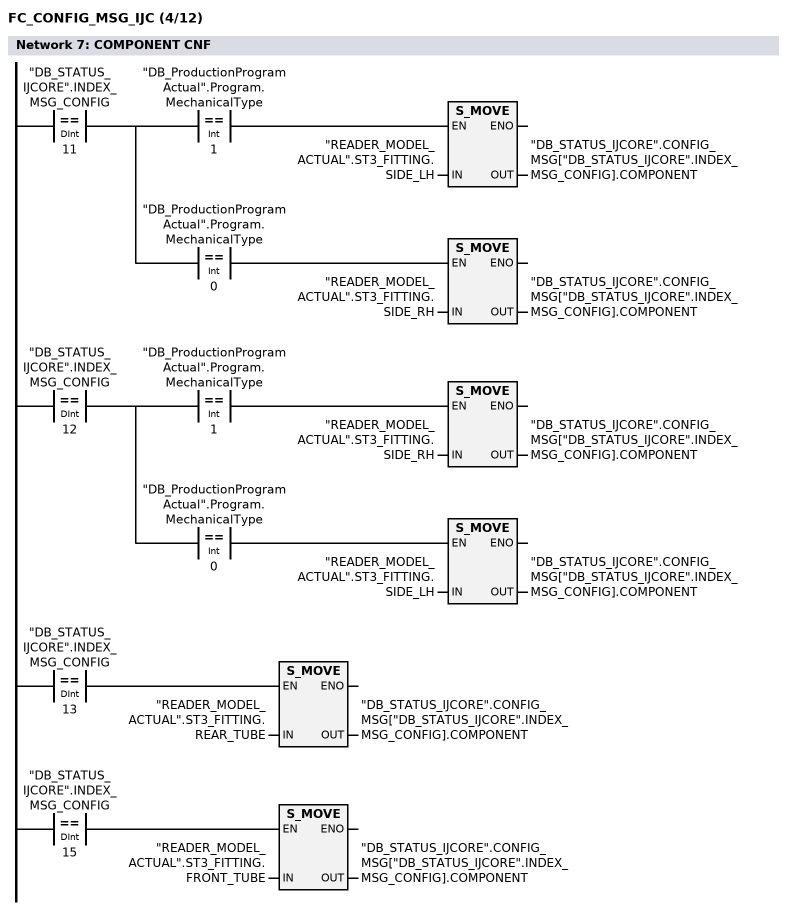
   RUNG wire#powerrail
      { S7_Templates := "SrcType := DInt" } EQ_Contact(in1 := "DB_STATUS_IJCORE".INDEX_MSG_CONFIG, in2 := 11)
      wire#w1
      { S7_Templates := "SrcType := Int" } EQ_Contact(in1 := "DB_ProductionProgramActual".Program.MechanicalType, in2 := 1)
      S_Move(in := "READER_MODEL_ACTUAL".ST3_FITTING.SIDE_LH, out => "DB_STATUS_IJCORE".CONFIG_MSG["DB_STATUS_IJCORE".INDEX_MSG_CONFIG].COMPONENT)
   END_RUNG
   RUNG wire#w1
      { S7_Templates := "SrcType := Int" } EQ_Contact(in1 := "DB_ProductionProgramActual".Program.MechanicalType, in2 := 0)
      S_Move(in := "READER_MODEL_ACTUAL".ST3_FITTING.SIDE_RH, out => "DB_STATUS_IJCORE".CONFIG_MSG["DB_STATUS_IJCORE".INDEX_MSG_CONFIG].COMPONENT)
   END_RUNG
   RUNG wire#powerrail
      { S7_Templates := "SrcType := DInt" } EQ_Contact(in1 := "DB_STATUS_IJCORE".INDEX_MSG_CONFIG, in2 := 12)
      wire#w2
      { S7_Templates := "SrcType := Int" } EQ_Contact(in1 := "DB_ProductionProgramActual".Program.MechanicalType, in2 := 1)
      S_Move(in := "READER_MODEL_ACTUAL".ST3_FITTING.SIDE_RH, out => "DB_STATUS_IJCORE".CONFIG_MSG["DB_STATUS_IJCORE".INDEX_MSG_CONFIG].COMPONENT)
   END_RUNG
   RUNG wire#w2
      { S7_Templates := "SrcType := Int" } EQ_Contact(in1 := "DB_ProductionProgramActual".Program.MechanicalType, in2 := 0)
      S_Move(in := "READER_MODEL_ACTUAL".ST3_FITTING.SIDE_LH, out => "DB_STATUS_IJCORE".CONFIG_MSG["DB_STATUS_IJCORE".INDEX_MSG_CONFIG].COMPONENT)
   END_RUNG
   RUNG wire#powerrail
      { S7_Templates := "SrcType := DInt" } EQ_Contact(in1 := "DB_STATUS_IJCORE".INDEX_MSG_CONFIG, in2 := 13)
      S_Move(in := "READER_MODEL_ACTUAL".ST3_FITTING.REAR_TUBE, out => "DB_STATUS_IJCORE".CONFIG_MSG["DB_STATUS_IJCORE".INDEX_MSG_CONFIG].COMPONENT)
   END_RUNG
   RUNG wire#powerrail
      { S7_Templates := "SrcType := DInt" } EQ_Contact(in1 := "DB_STATUS_IJCORE".INDEX_MSG_CONFIG, in2 := 15)
      S_Move(in := "READER_MODEL_ACTUAL".ST3_FITTING.FRONT_TUBE, out => "DB_STATUS_IJCORE".CONFIG_MSG["DB_STATUS_IJCORE".INDEX_MSG_CONFIG].COMPONENT)
   END_RUNG
   // the same network as SCL:
   #_w1 := "DB_STATUS_IJCORE".INDEX_MSG_CONFIG = 11;
   IF #_w1 AND ("DB_ProductionProgramActual".Program.MechanicalType = 1) THEN
       "DB_STATUS_IJCORE".CONFIG_MSG["DB_STATUS_IJCORE".INDEX_MSG_CONFIG].COMPONENT := "READER_MODEL_ACTUAL".ST3_FITTING.SIDE_LH;
   END_IF;
   IF #_w1 AND ("DB_ProductionProgramActual".Program.MechanicalType = 0) THEN
       "DB_STATUS_IJCORE".CONFIG_MSG["DB_STATUS_IJCORE".INDEX_MSG_CONFIG].COMPONENT := "READER_MODEL_ACTUAL".ST3_FITTING.SIDE_RH;
   END_IF;
   #_w2 := "DB_STATUS_IJCORE".INDEX_MSG_CONFIG = 12;
   IF #_w2 AND ("DB_ProductionProgramActual".Program.MechanicalType = 1) THEN
       "DB_STATUS_IJCORE".CONFIG_MSG["DB_STATUS_IJCORE".INDEX_MSG_CONFIG].COMPONENT := "READER_MODEL_ACTUAL".ST3_FITTING.SIDE_RH;
   END_IF;
   IF #_w2 AND ("DB_ProductionProgramActual".Program.MechanicalType = 0) THEN
       "DB_STATUS_IJCORE".CONFIG_MSG["DB_STATUS_IJCORE".INDEX_MSG_CONFIG].COMPONENT := "READER_MODEL_ACTUAL".ST3_FITTING.SIDE_LH;
   END_IF;
   IF "DB_STATUS_IJCORE".INDEX_MSG_CONFIG = 13 THEN
       "DB_STATUS_IJCORE".CONFIG_MSG["DB_STATUS_IJCORE".INDEX_MSG_CONFIG].COMPONENT := "READER_MODEL_ACTUAL".ST3_FITTING.REAR_TUBE;
   END_IF;
   IF "DB_STATUS_IJCORE".INDEX_MSG_CONFIG = 15 THEN
       "DB_STATUS_IJCORE".CONFIG_MSG["DB_STATUS_IJCORE".INDEX_MSG_CONFIG].COMPONENT := "READER_MODEL_ACTUAL".ST3_FITTING.FRONT_TUBE;
   END_IF;
END_REGION

REGION Network 8: STATUS TRR
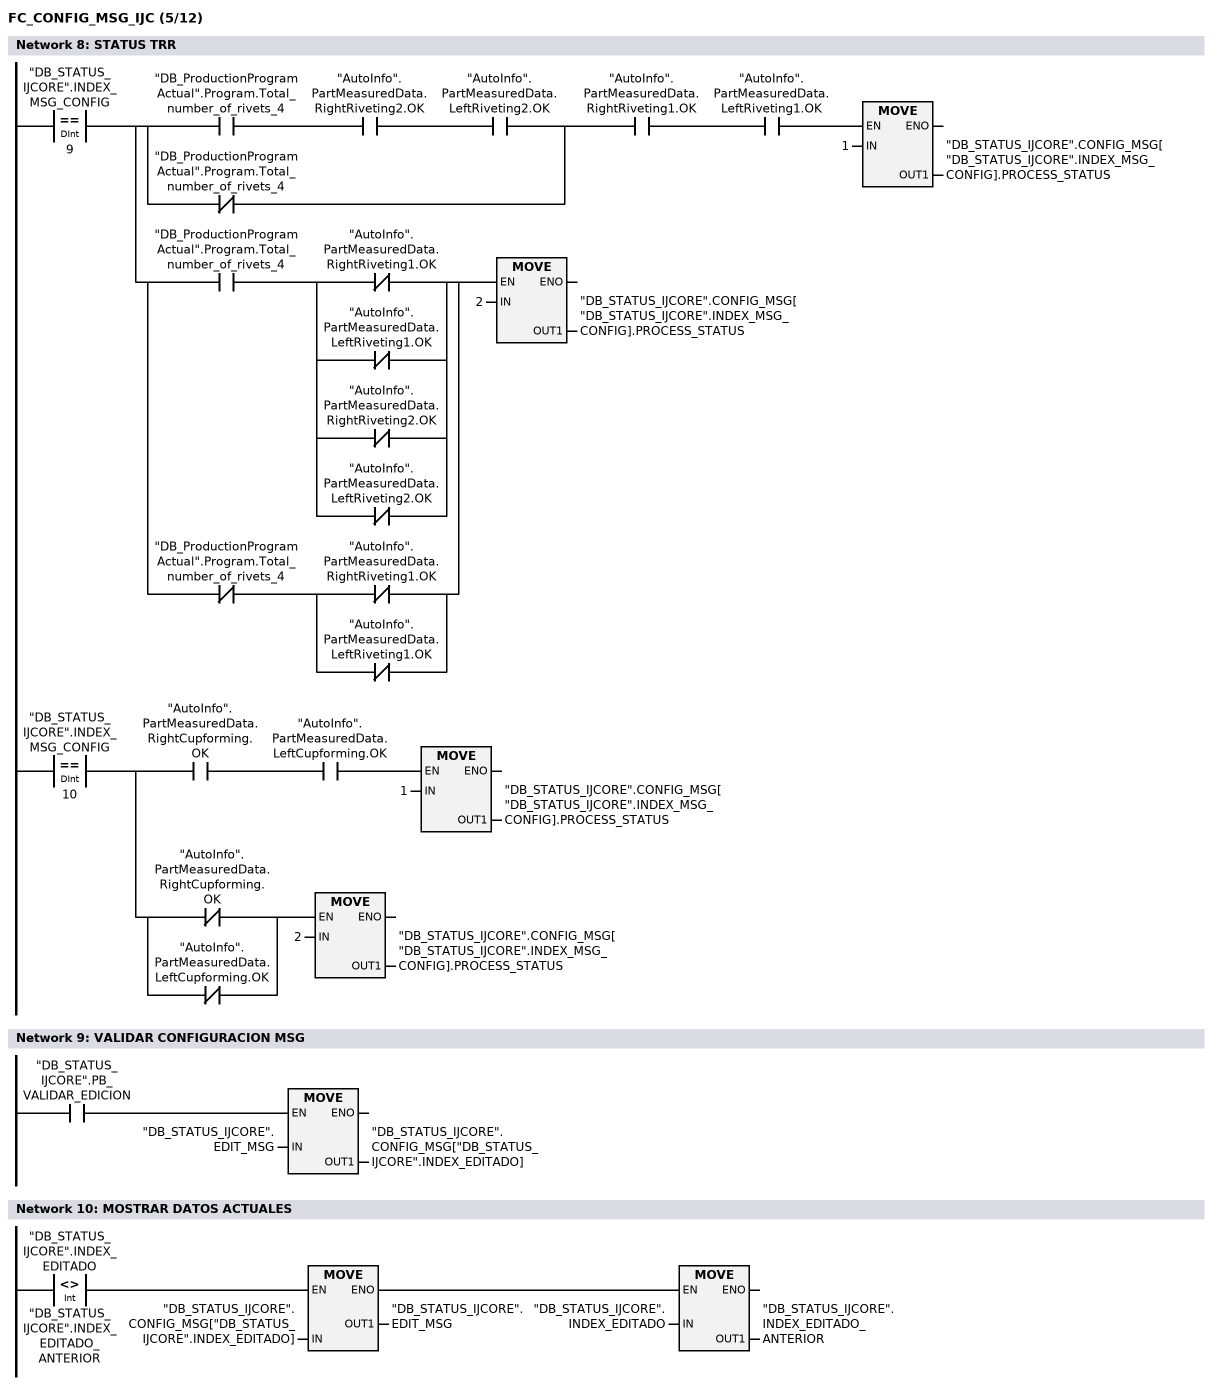
   RUNG wire#powerrail
      { S7_Templates := "SrcType := DInt" } EQ_Contact(in1 := "DB_STATUS_IJCORE".INDEX_MSG_CONFIG, in2 := 9)
      wire#w1
      Contact( "DB_ProductionProgramActual".Program.Total_number_of_rivets_4 )
      Contact( "AutoInfo".PartMeasuredData.RightRiveting2.OK )
      Contact( "AutoInfo".PartMeasuredData.LeftRiveting2.OK )
      wire#w2
      Contact( "AutoInfo".PartMeasuredData.RightRiveting1.OK )
      Contact( "AutoInfo".PartMeasuredData.LeftRiveting1.OK )
      Move(in := 1, out1 => "DB_STATUS_IJCORE".CONFIG_MSG["DB_STATUS_IJCORE".INDEX_MSG_CONFIG].PROCESS_STATUS)
   END_RUNG
   RUNG wire#w1
      I_Contact( "DB_ProductionProgramActual".Program.Total_number_of_rivets_4 )
   END_RUNG wire#w2
   RUNG wire#w1
      Contact( "DB_ProductionProgramActual".Program.Total_number_of_rivets_4 )
      wire#w3
      I_Contact( "AutoInfo".PartMeasuredData.RightRiveting1.OK )
      wire#w4
      Move(in := 2, out1 => "DB_STATUS_IJCORE".CONFIG_MSG["DB_STATUS_IJCORE".INDEX_MSG_CONFIG].PROCESS_STATUS)
   END_RUNG
   RUNG wire#w3
      I_Contact( "AutoInfo".PartMeasuredData.LeftRiveting1.OK )
   END_RUNG wire#w4
   RUNG wire#w3
      I_Contact( "AutoInfo".PartMeasuredData.RightRiveting2.OK )
   END_RUNG wire#w4
   RUNG wire#w3
      I_Contact( "AutoInfo".PartMeasuredData.LeftRiveting2.OK )
   END_RUNG wire#w4
   RUNG wire#w1
      I_Contact( "DB_ProductionProgramActual".Program.Total_number_of_rivets_4 )
      wire#w5
      I_Contact( "AutoInfo".PartMeasuredData.RightRiveting1.OK )
   END_RUNG wire#w4
   RUNG wire#w5
      I_Contact( "AutoInfo".PartMeasuredData.LeftRiveting1.OK )
   END_RUNG wire#w4
   RUNG wire#powerrail
      { S7_Templates := "SrcType := DInt" } EQ_Contact(in1 := "DB_STATUS_IJCORE".INDEX_MSG_CONFIG, in2 := 10)
      wire#w6
      Contact( "AutoInfo".PartMeasuredData.RightCupforming.OK )
      Contact( "AutoInfo".PartMeasuredData.LeftCupforming.OK )
      Move(in := 1, out1 => "DB_STATUS_IJCORE".CONFIG_MSG["DB_STATUS_IJCORE".INDEX_MSG_CONFIG].PROCESS_STATUS)
   END_RUNG
   RUNG wire#w6
      I_Contact( "AutoInfo".PartMeasuredData.RightCupforming.OK )
      wire#w7
      Move(in := 2, out1 => "DB_STATUS_IJCORE".CONFIG_MSG["DB_STATUS_IJCORE".INDEX_MSG_CONFIG].PROCESS_STATUS)
   END_RUNG
   RUNG wire#w6
      I_Contact( "AutoInfo".PartMeasuredData.LeftCupforming.OK )
   END_RUNG wire#w7
   // the same network as SCL:
   #_w1 := "DB_STATUS_IJCORE".INDEX_MSG_CONFIG = 9;
   IF #_w1 AND (("DB_ProductionProgramActual".Program.Total_number_of_rivets_4 AND "AutoInfo".PartMeasuredData.RightRiveting2.OK AND "AutoInfo".PartMeasuredData.LeftRiveting2.OK) OR NOT "DB_ProductionProgramActual".Program.Total_number_of_rivets_4) AND "AutoInfo".PartMeasuredData.RightRiveting1.OK AND "AutoInfo".PartMeasuredData.LeftRiveting1.OK THEN
       "DB_STATUS_IJCORE".CONFIG_MSG["DB_STATUS_IJCORE".INDEX_MSG_CONFIG].PROCESS_STATUS := 1;
   END_IF;
   IF #_w1 AND (("DB_ProductionProgramActual".Program.Total_number_of_rivets_4 AND (NOT "AutoInfo".PartMeasuredData.RightRiveting1.OK OR NOT "AutoInfo".PartMeasuredData.LeftRiveting1.OK OR NOT "AutoInfo".PartMeasuredData.RightRiveting2.OK OR NOT "AutoInfo".PartMeasuredData.LeftRiveting2.OK)) OR (NOT "DB_ProductionProgramActual".Program.Total_number_of_rivets_4 AND (NOT "AutoInfo".PartMeasuredData.RightRiveting1.OK OR NOT "AutoInfo".PartMeasuredData.LeftRiveting1.OK))) THEN
       "DB_STATUS_IJCORE".CONFIG_MSG["DB_STATUS_IJCORE".INDEX_MSG_CONFIG].PROCESS_STATUS := 2;
   END_IF;
   #_w2 := "DB_STATUS_IJCORE".INDEX_MSG_CONFIG = 10;
   IF #_w2 AND "AutoInfo".PartMeasuredData.RightCupforming.OK AND "AutoInfo".PartMeasuredData.LeftCupforming.OK THEN
       "DB_STATUS_IJCORE".CONFIG_MSG["DB_STATUS_IJCORE".INDEX_MSG_CONFIG].PROCESS_STATUS := 1;
   END_IF;
   IF #_w2 AND (NOT "AutoInfo".PartMeasuredData.RightCupforming.OK OR NOT "AutoInfo".PartMeasuredData.LeftCupforming.OK) THEN
       "DB_STATUS_IJCORE".CONFIG_MSG["DB_STATUS_IJCORE".INDEX_MSG_CONFIG].PROCESS_STATUS := 2;
   END_IF;
END_REGION

REGION Network 9: VALIDAR CONFIGURACION MSG
   RUNG wire#powerrail
      Contact( "DB_STATUS_IJCORE".PB_VALIDAR_EDICION )
      Move(in := "DB_STATUS_IJCORE".EDIT_MSG, out1 => "DB_STATUS_IJCORE".CONFIG_MSG["DB_STATUS_IJCORE".INDEX_EDITADO])
   END_RUNG
   // the same network as SCL:
   IF "DB_STATUS_IJCORE".PB_VALIDAR_EDICION THEN
       "DB_STATUS_IJCORE".CONFIG_MSG["DB_STATUS_IJCORE".INDEX_EDITADO] := "DB_STATUS_IJCORE".EDIT_MSG;
   END_IF;
END_REGION

REGION Network 10: MOSTRAR DATOS ACTUALES
   RUNG wire#powerrail
      { S7_Templates := "SrcType := Int" } NE_Contact(in1 := "DB_STATUS_IJCORE".INDEX_EDITADO, in2 := "DB_STATUS_IJCORE".INDEX_EDITADO_ANTERIOR)
      Move(in := "DB_STATUS_IJCORE".CONFIG_MSG["DB_STATUS_IJCORE".INDEX_EDITADO], out1 => "DB_STATUS_IJCORE".EDIT_MSG)
      Move(in := "DB_STATUS_IJCORE".INDEX_EDITADO, out1 => "DB_STATUS_IJCORE".INDEX_EDITADO_ANTERIOR)
   END_RUNG
   // the same network as SCL:
   IF "DB_STATUS_IJCORE".INDEX_EDITADO <> "DB_STATUS_IJCORE".INDEX_EDITADO_ANTERIOR THEN
       "DB_STATUS_IJCORE".EDIT_MSG := "DB_STATUS_IJCORE".CONFIG_MSG["DB_STATUS_IJCORE".INDEX_EDITADO];
       "DB_STATUS_IJCORE".INDEX_EDITADO_ANTERIOR := "DB_STATUS_IJCORE".INDEX_EDITADO;
   END_IF;
END_REGION

REGION Network 11: SEND STA
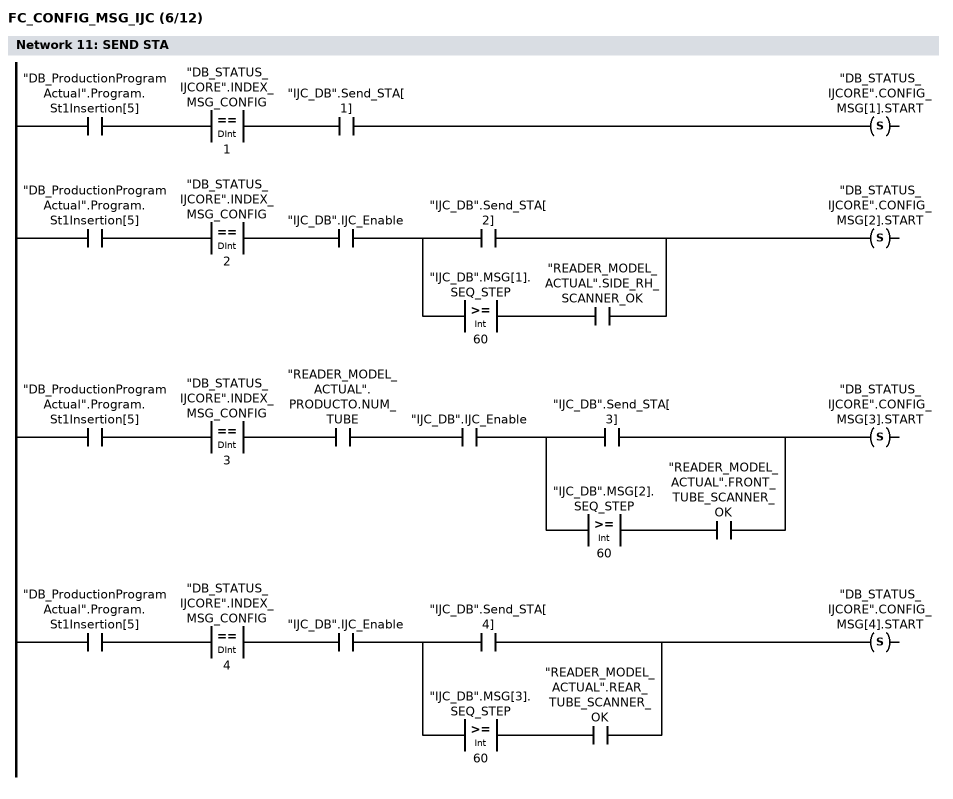
   RUNG wire#powerrail
      Contact( "DB_ProductionProgramActual".Program.St1Insertion[5] )
      { S7_Templates := "SrcType := DInt" } EQ_Contact(in1 := "DB_STATUS_IJCORE".INDEX_MSG_CONFIG, in2 := 1)
      Contact( "IJC_DB".Send_STA[1] )
      S_Coil( "DB_STATUS_IJCORE".CONFIG_MSG[1].START )
   END_RUNG
   RUNG wire#powerrail
      Contact( "DB_ProductionProgramActual".Program.St1Insertion[5] )
      { S7_Templates := "SrcType := DInt" } EQ_Contact(in1 := "DB_STATUS_IJCORE".INDEX_MSG_CONFIG, in2 := 2)
      Contact( "IJC_DB".IJC_Enable )
      wire#w1
      Contact( "IJC_DB".Send_STA[2] )
      wire#w2
      S_Coil( "DB_STATUS_IJCORE".CONFIG_MSG[2].START )
   END_RUNG
   RUNG wire#w1
      { S7_Templates := "SrcType := Int" } GE_Contact(in1 := "IJC_DB".MSG[1].SEQ_STEP, in2 := 60)
      Contact( "READER_MODEL_ACTUAL".SIDE_RH_SCANNER_OK )
   END_RUNG wire#w2
   RUNG wire#powerrail
      Contact( "DB_ProductionProgramActual".Program.St1Insertion[5] )
      { S7_Templates := "SrcType := DInt" } EQ_Contact(in1 := "DB_STATUS_IJCORE".INDEX_MSG_CONFIG, in2 := 3)
      Contact( "READER_MODEL_ACTUAL".PRODUCTO.NUM_TUBE )
      Contact( "IJC_DB".IJC_Enable )
      wire#w3
      Contact( "IJC_DB".Send_STA[3] )
      wire#w4
      S_Coil( "DB_STATUS_IJCORE".CONFIG_MSG[3].START )
   END_RUNG
   RUNG wire#w3
      { S7_Templates := "SrcType := Int" } GE_Contact(in1 := "IJC_DB".MSG[2].SEQ_STEP, in2 := 60)
      Contact( "READER_MODEL_ACTUAL".FRONT_TUBE_SCANNER_OK )
   END_RUNG wire#w4
   RUNG wire#powerrail
      Contact( "DB_ProductionProgramActual".Program.St1Insertion[5] )
      { S7_Templates := "SrcType := DInt" } EQ_Contact(in1 := "DB_STATUS_IJCORE".INDEX_MSG_CONFIG, in2 := 4)
      Contact( "IJC_DB".IJC_Enable )
      wire#w5
      Contact( "IJC_DB".Send_STA[4] )
      wire#w6
      S_Coil( "DB_STATUS_IJCORE".CONFIG_MSG[4].START )
   END_RUNG
   RUNG wire#w5
      { S7_Templates := "SrcType := Int" } GE_Contact(in1 := "IJC_DB".MSG[3].SEQ_STEP, in2 := 60)
      Contact( "READER_MODEL_ACTUAL".REAR_TUBE_SCANNER_OK )
   END_RUNG wire#w6
   // the same network as SCL:
   IF "DB_ProductionProgramActual".Program.St1Insertion[5] AND ("DB_STATUS_IJCORE".INDEX_MSG_CONFIG = 1) AND "IJC_DB".Send_STA[1] THEN
       "DB_STATUS_IJCORE".CONFIG_MSG[1].START := TRUE;
   END_IF;
   IF "DB_ProductionProgramActual".Program.St1Insertion[5] AND ("DB_STATUS_IJCORE".INDEX_MSG_CONFIG = 2) AND "IJC_DB".IJC_Enable AND ("IJC_DB".Send_STA[2] OR (("IJC_DB".MSG[1].SEQ_STEP >= 60) AND "READER_MODEL_ACTUAL".SIDE_RH_SCANNER_OK)) THEN
       "DB_STATUS_IJCORE".CONFIG_MSG[2].START := TRUE;
   END_IF;
   IF "DB_ProductionProgramActual".Program.St1Insertion[5] AND ("DB_STATUS_IJCORE".INDEX_MSG_CONFIG = 3) AND "READER_MODEL_ACTUAL".PRODUCTO.NUM_TUBE AND "IJC_DB".IJC_Enable AND ("IJC_DB".Send_STA[3] OR (("IJC_DB".MSG[2].SEQ_STEP >= 60) AND "READER_MODEL_ACTUAL".FRONT_TUBE_SCANNER_OK)) THEN
       "DB_STATUS_IJCORE".CONFIG_MSG[3].START := TRUE;
   END_IF;
   IF "DB_ProductionProgramActual".Program.St1Insertion[5] AND ("DB_STATUS_IJCORE".INDEX_MSG_CONFIG = 4) AND "IJC_DB".IJC_Enable AND ("IJC_DB".Send_STA[4] OR (("IJC_DB".MSG[3].SEQ_STEP >= 60) AND "READER_MODEL_ACTUAL".REAR_TUBE_SCANNER_OK)) THEN
       "DB_STATUS_IJCORE".CONFIG_MSG[4].START := TRUE;
   END_IF;
END_REGION

REGION Network 12: SEND TRC SCAN LABEL
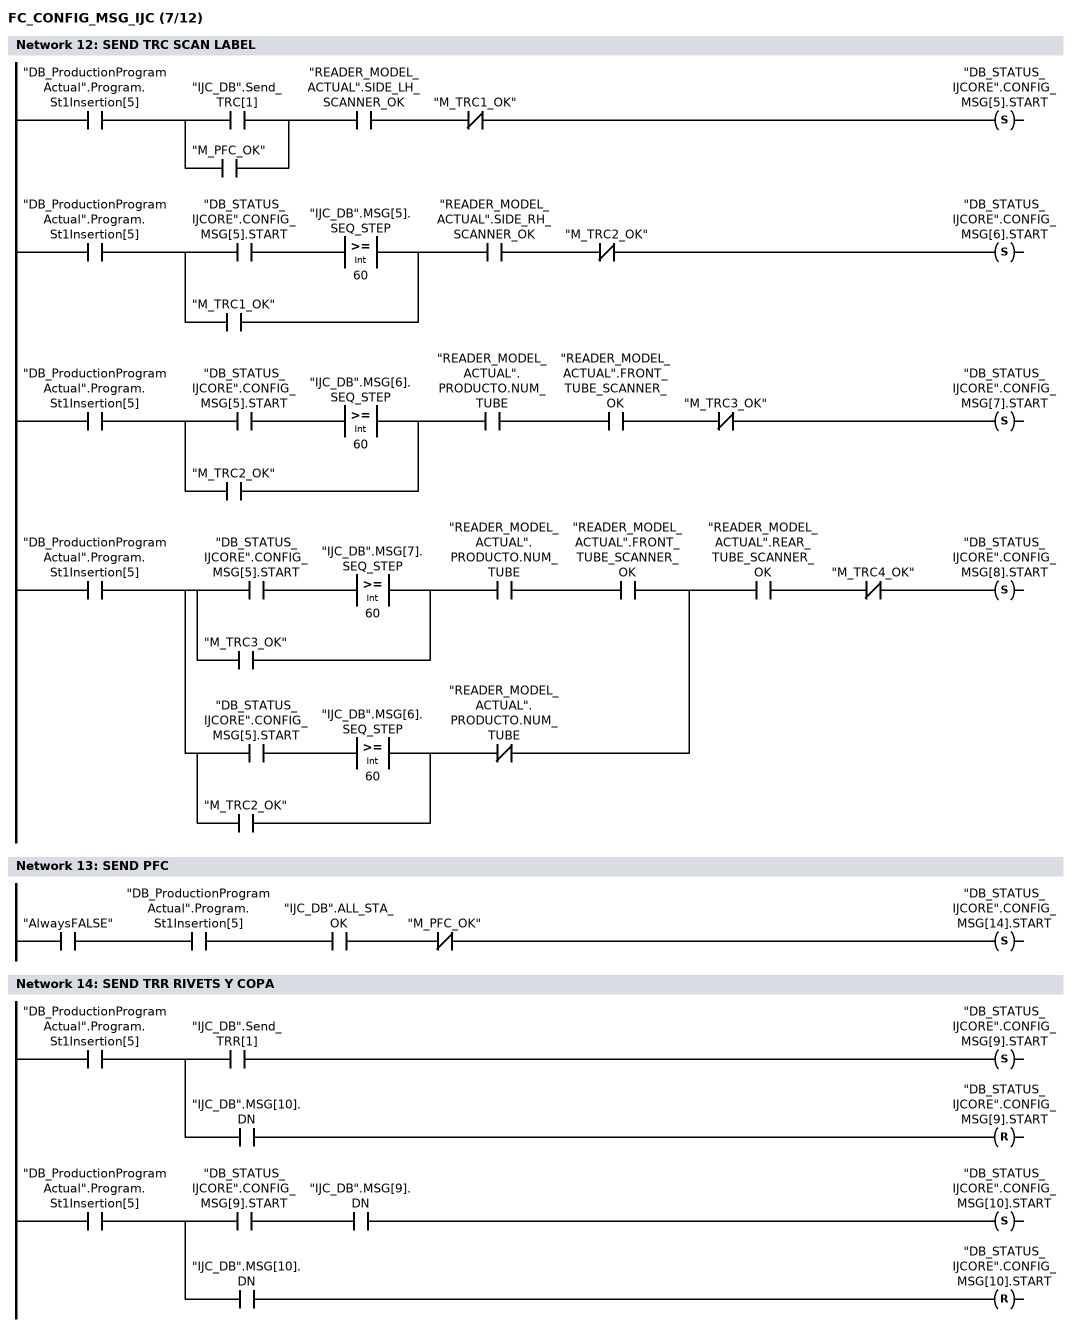
   RUNG wire#powerrail
      Contact( "DB_ProductionProgramActual".Program.St1Insertion[5] )
      wire#w1
      Contact( "IJC_DB".Send_TRC[1] )
      wire#w2
      Contact( "READER_MODEL_ACTUAL".SIDE_LH_SCANNER_OK )
      I_Contact( "M_TRC1_OK" )
      S_Coil( "DB_STATUS_IJCORE".CONFIG_MSG[5].START )
   END_RUNG
   RUNG wire#w1
      Contact( "M_PFC_OK" )
   END_RUNG wire#w2
   RUNG wire#powerrail
      Contact( "DB_ProductionProgramActual".Program.St1Insertion[5] )
      wire#w3
      Contact( "DB_STATUS_IJCORE".CONFIG_MSG[5].START )
      { S7_Templates := "SrcType := Int" } GE_Contact(in1 := "IJC_DB".MSG[5].SEQ_STEP, in2 := 60)
      wire#w4
      Contact( "READER_MODEL_ACTUAL".SIDE_RH_SCANNER_OK )
      I_Contact( "M_TRC2_OK" )
      S_Coil( "DB_STATUS_IJCORE".CONFIG_MSG[6].START )
   END_RUNG
   RUNG wire#w3
      Contact( "M_TRC1_OK" )
   END_RUNG wire#w4
   RUNG wire#powerrail
      Contact( "DB_ProductionProgramActual".Program.St1Insertion[5] )
      wire#w5
      Contact( "DB_STATUS_IJCORE".CONFIG_MSG[5].START )
      { S7_Templates := "SrcType := Int" } GE_Contact(in1 := "IJC_DB".MSG[6].SEQ_STEP, in2 := 60)
      wire#w6
      Contact( "READER_MODEL_ACTUAL".PRODUCTO.NUM_TUBE )
      Contact( "READER_MODEL_ACTUAL".FRONT_TUBE_SCANNER_OK )
      I_Contact( "M_TRC3_OK" )
      S_Coil( "DB_STATUS_IJCORE".CONFIG_MSG[7].START )
   END_RUNG
   RUNG wire#w5
      Contact( "M_TRC2_OK" )
   END_RUNG wire#w6
   RUNG wire#powerrail
      Contact( "DB_ProductionProgramActual".Program.St1Insertion[5] )
      wire#w7
      Contact( "DB_STATUS_IJCORE".CONFIG_MSG[5].START )
      { S7_Templates := "SrcType := Int" } GE_Contact(in1 := "IJC_DB".MSG[7].SEQ_STEP, in2 := 60)
      wire#w8
      Contact( "READER_MODEL_ACTUAL".PRODUCTO.NUM_TUBE )
      Contact( "READER_MODEL_ACTUAL".FRONT_TUBE_SCANNER_OK )
      wire#w9
      Contact( "READER_MODEL_ACTUAL".REAR_TUBE_SCANNER_OK )
      I_Contact( "M_TRC4_OK" )
      S_Coil( "DB_STATUS_IJCORE".CONFIG_MSG[8].START )
   END_RUNG
   RUNG wire#w7
      Contact( "M_TRC3_OK" )
   END_RUNG wire#w8
   RUNG wire#w7
      Contact( "DB_STATUS_IJCORE".CONFIG_MSG[5].START )
      { S7_Templates := "SrcType := Int" } GE_Contact(in1 := "IJC_DB".MSG[6].SEQ_STEP, in2 := 60)
      wire#w10
      I_Contact( "READER_MODEL_ACTUAL".PRODUCTO.NUM_TUBE )
   END_RUNG wire#w9
   RUNG wire#w7
      Contact( "M_TRC2_OK" )
   END_RUNG wire#w10
   // the same network as SCL:
   IF "DB_ProductionProgramActual".Program.St1Insertion[5] AND ("IJC_DB".Send_TRC[1] OR "M_PFC_OK") AND "READER_MODEL_ACTUAL".SIDE_LH_SCANNER_OK AND NOT "M_TRC1_OK" THEN
       "DB_STATUS_IJCORE".CONFIG_MSG[5].START := TRUE;
   END_IF;
   IF "DB_ProductionProgramActual".Program.St1Insertion[5] AND (("DB_STATUS_IJCORE".CONFIG_MSG[5].START AND ("IJC_DB".MSG[5].SEQ_STEP >= 60)) OR "M_TRC1_OK") AND "READER_MODEL_ACTUAL".SIDE_RH_SCANNER_OK AND NOT "M_TRC2_OK" THEN
       "DB_STATUS_IJCORE".CONFIG_MSG[6].START := TRUE;
   END_IF;
   IF "DB_ProductionProgramActual".Program.St1Insertion[5] AND (("DB_STATUS_IJCORE".CONFIG_MSG[5].START AND ("IJC_DB".MSG[6].SEQ_STEP >= 60)) OR "M_TRC2_OK") AND "READER_MODEL_ACTUAL".PRODUCTO.NUM_TUBE AND "READER_MODEL_ACTUAL".FRONT_TUBE_SCANNER_OK AND NOT "M_TRC3_OK" THEN
       "DB_STATUS_IJCORE".CONFIG_MSG[7].START := TRUE;
   END_IF;
   IF "DB_ProductionProgramActual".Program.St1Insertion[5] AND (((("DB_STATUS_IJCORE".CONFIG_MSG[5].START AND ("IJC_DB".MSG[7].SEQ_STEP >= 60)) OR "M_TRC3_OK") AND "READER_MODEL_ACTUAL".PRODUCTO.NUM_TUBE AND "READER_MODEL_ACTUAL".FRONT_TUBE_SCANNER_OK) OR ((("DB_STATUS_IJCORE".CONFIG_MSG[5].START AND ("IJC_DB".MSG[6].SEQ_STEP >= 60)) OR "M_TRC2_OK") AND NOT "READER_MODEL_ACTUAL".PRODUCTO.NUM_TUBE)) AND "READER_MODEL_ACTUAL".REAR_TUBE_SCANNER_OK AND NOT "M_TRC4_OK" THEN
       "DB_STATUS_IJCORE".CONFIG_MSG[8].START := TRUE;
   END_IF;
END_REGION

REGION Network 13: SEND PFC
   RUNG wire#powerrail
      Contact( "AlwaysFALSE" )
      Contact( "DB_ProductionProgramActual".Program.St1Insertion[5] )
      Contact( "IJC_DB".ALL_STA_OK )
      I_Contact( "M_PFC_OK" )
      S_Coil( "DB_STATUS_IJCORE".CONFIG_MSG[14].START )
   END_RUNG
   // the same network as SCL:
   IF "AlwaysFALSE" AND "DB_ProductionProgramActual".Program.St1Insertion[5] AND "IJC_DB".ALL_STA_OK AND NOT "M_PFC_OK" THEN
       "DB_STATUS_IJCORE".CONFIG_MSG[14].START := TRUE;
   END_IF;
END_REGION

REGION Network 14: SEND TRR RIVETS Y COPA
   RUNG wire#powerrail
      Contact( "DB_ProductionProgramActual".Program.St1Insertion[5] )
      wire#w1
      Contact( "IJC_DB".Send_TRR[1] )
      S_Coil( "DB_STATUS_IJCORE".CONFIG_MSG[9].START )
   END_RUNG
   RUNG wire#w1
      Contact( "IJC_DB".MSG[10].DN )
      R_Coil( "DB_STATUS_IJCORE".CONFIG_MSG[9].START )
   END_RUNG
   RUNG wire#powerrail
      Contact( "DB_ProductionProgramActual".Program.St1Insertion[5] )
      wire#w2
      Contact( "DB_STATUS_IJCORE".CONFIG_MSG[9].START )
      Contact( "IJC_DB".MSG[9].DN )
      S_Coil( "DB_STATUS_IJCORE".CONFIG_MSG[10].START )
   END_RUNG
   RUNG wire#w2
      Contact( "IJC_DB".MSG[10].DN )
      R_Coil( "DB_STATUS_IJCORE".CONFIG_MSG[10].START )
   END_RUNG
   // the same network as SCL:
   IF "DB_ProductionProgramActual".Program.St1Insertion[5] AND "IJC_DB".Send_TRR[1] THEN
       "DB_STATUS_IJCORE".CONFIG_MSG[9].START := TRUE;
   END_IF;
   IF "DB_ProductionProgramActual".Program.St1Insertion[5] AND "IJC_DB".MSG[10].DN THEN
       "DB_STATUS_IJCORE".CONFIG_MSG[9].START := FALSE;
   END_IF;
   IF "DB_ProductionProgramActual".Program.St1Insertion[5] AND "DB_STATUS_IJCORE".CONFIG_MSG[9].START AND "IJC_DB".MSG[9].DN THEN
       "DB_STATUS_IJCORE".CONFIG_MSG[10].START := TRUE;
   END_IF;
   IF "DB_ProductionProgramActual".Program.St1Insertion[5] AND "IJC_DB".MSG[10].DN THEN
       "DB_STATUS_IJCORE".CONFIG_MSG[10].START := FALSE;
   END_IF;
END_REGION

REGION Network 15: SEND CNF
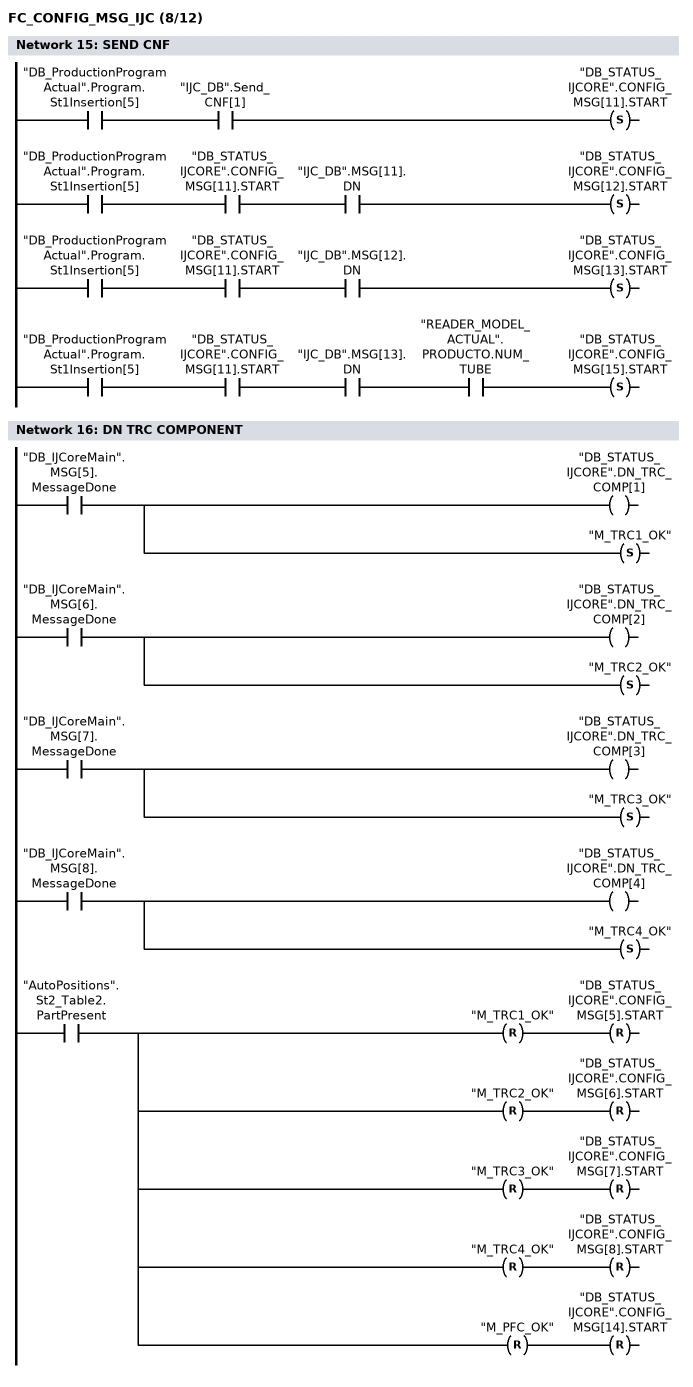
   RUNG wire#powerrail
      Contact( "DB_ProductionProgramActual".Program.St1Insertion[5] )
      Contact( "IJC_DB".Send_CNF[1] )
      S_Coil( "DB_STATUS_IJCORE".CONFIG_MSG[11].START )
   END_RUNG
   RUNG wire#powerrail
      Contact( "DB_ProductionProgramActual".Program.St1Insertion[5] )
      Contact( "DB_STATUS_IJCORE".CONFIG_MSG[11].START )
      Contact( "IJC_DB".MSG[11].DN )
      S_Coil( "DB_STATUS_IJCORE".CONFIG_MSG[12].START )
   END_RUNG
   RUNG wire#powerrail
      Contact( "DB_ProductionProgramActual".Program.St1Insertion[5] )
      Contact( "DB_STATUS_IJCORE".CONFIG_MSG[11].START )
      Contact( "IJC_DB".MSG[12].DN )
      S_Coil( "DB_STATUS_IJCORE".CONFIG_MSG[13].START )
   END_RUNG
   RUNG wire#powerrail
      Contact( "DB_ProductionProgramActual".Program.St1Insertion[5] )
      Contact( "DB_STATUS_IJCORE".CONFIG_MSG[11].START )
      Contact( "IJC_DB".MSG[13].DN )
      Contact( "READER_MODEL_ACTUAL".PRODUCTO.NUM_TUBE )
      S_Coil( "DB_STATUS_IJCORE".CONFIG_MSG[15].START )
   END_RUNG
   // the same network as SCL:
   IF "DB_ProductionProgramActual".Program.St1Insertion[5] AND "IJC_DB".Send_CNF[1] THEN
       "DB_STATUS_IJCORE".CONFIG_MSG[11].START := TRUE;
   END_IF;
   IF "DB_ProductionProgramActual".Program.St1Insertion[5] AND "DB_STATUS_IJCORE".CONFIG_MSG[11].START AND "IJC_DB".MSG[11].DN THEN
       "DB_STATUS_IJCORE".CONFIG_MSG[12].START := TRUE;
   END_IF;
   IF "DB_ProductionProgramActual".Program.St1Insertion[5] AND "DB_STATUS_IJCORE".CONFIG_MSG[11].START AND "IJC_DB".MSG[12].DN THEN
       "DB_STATUS_IJCORE".CONFIG_MSG[13].START := TRUE;
   END_IF;
   IF "DB_ProductionProgramActual".Program.St1Insertion[5] AND "DB_STATUS_IJCORE".CONFIG_MSG[11].START AND "IJC_DB".MSG[13].DN AND "READER_MODEL_ACTUAL".PRODUCTO.NUM_TUBE THEN
       "DB_STATUS_IJCORE".CONFIG_MSG[15].START := TRUE;
   END_IF;
END_REGION

REGION Network 16: DN TRC COMPONENT
   RUNG wire#powerrail
      Contact( "DB_IJCoreMain".MSG[5].MessageDone )
      wire#w1
      Coil( "DB_STATUS_IJCORE".DN_TRC_COMP[1] )
   END_RUNG
   RUNG wire#w1
      S_Coil( "M_TRC1_OK" )
   END_RUNG
   RUNG wire#powerrail
      Contact( "DB_IJCoreMain".MSG[6].MessageDone )
      wire#w2
      Coil( "DB_STATUS_IJCORE".DN_TRC_COMP[2] )
   END_RUNG
   RUNG wire#w2
      S_Coil( "M_TRC2_OK" )
   END_RUNG
   RUNG wire#powerrail
      Contact( "DB_IJCoreMain".MSG[7].MessageDone )
      wire#w3
      Coil( "DB_STATUS_IJCORE".DN_TRC_COMP[3] )
   END_RUNG
   RUNG wire#w3
      S_Coil( "M_TRC3_OK" )
   END_RUNG
   RUNG wire#powerrail
      Contact( "DB_IJCoreMain".MSG[8].MessageDone )
      wire#w4
      Coil( "DB_STATUS_IJCORE".DN_TRC_COMP[4] )
   END_RUNG
   RUNG wire#w4
      S_Coil( "M_TRC4_OK" )
   END_RUNG
   RUNG wire#powerrail
      Contact( "AutoPositions".St2_Table2.PartPresent )
      wire#w5
      R_Coil( "M_TRC1_OK" )
      R_Coil( "DB_STATUS_IJCORE".CONFIG_MSG[5].START )
   END_RUNG
   RUNG wire#w5
      R_Coil( "M_TRC2_OK" )
      R_Coil( "DB_STATUS_IJCORE".CONFIG_MSG[6].START )
   END_RUNG
   RUNG wire#w5
      R_Coil( "M_TRC3_OK" )
      R_Coil( "DB_STATUS_IJCORE".CONFIG_MSG[7].START )
   END_RUNG
   RUNG wire#w5
      R_Coil( "M_TRC4_OK" )
      R_Coil( "DB_STATUS_IJCORE".CONFIG_MSG[8].START )
   END_RUNG
   RUNG wire#w5
      R_Coil( "M_PFC_OK" )
      R_Coil( "DB_STATUS_IJCORE".CONFIG_MSG[14].START )
   END_RUNG
   // the same network as SCL:
   "DB_STATUS_IJCORE".DN_TRC_COMP[1] := "DB_IJCoreMain".MSG[5].MessageDone;
   IF "DB_IJCoreMain".MSG[5].MessageDone THEN "M_TRC1_OK" := TRUE; END_IF;
   "DB_STATUS_IJCORE".DN_TRC_COMP[2] := "DB_IJCoreMain".MSG[6].MessageDone;
   IF "DB_IJCoreMain".MSG[6].MessageDone THEN "M_TRC2_OK" := TRUE; END_IF;
   "DB_STATUS_IJCORE".DN_TRC_COMP[3] := "DB_IJCoreMain".MSG[7].MessageDone;
   IF "DB_IJCoreMain".MSG[7].MessageDone THEN "M_TRC3_OK" := TRUE; END_IF;
   "DB_STATUS_IJCORE".DN_TRC_COMP[4] := "DB_IJCoreMain".MSG[8].MessageDone;
   IF "DB_IJCoreMain".MSG[8].MessageDone THEN "M_TRC4_OK" := TRUE; END_IF;
   IF "AutoPositions".St2_Table2.PartPresent THEN
       "M_TRC1_OK" := FALSE;
       "DB_STATUS_IJCORE".CONFIG_MSG[5].START := FALSE;
       "M_TRC2_OK" := FALSE;
       "DB_STATUS_IJCORE".CONFIG_MSG[6].START := FALSE;
       "M_TRC3_OK" := FALSE;
       "DB_STATUS_IJCORE".CONFIG_MSG[7].START := FALSE;
       "M_TRC4_OK" := FALSE;
       "DB_STATUS_IJCORE".CONFIG_MSG[8].START := FALSE;
       "M_PFC_OK" := FALSE;
       "DB_STATUS_IJCORE".CONFIG_MSG[14].START := FALSE;
   END_IF;
END_REGION

REGION Network 17: DN STA
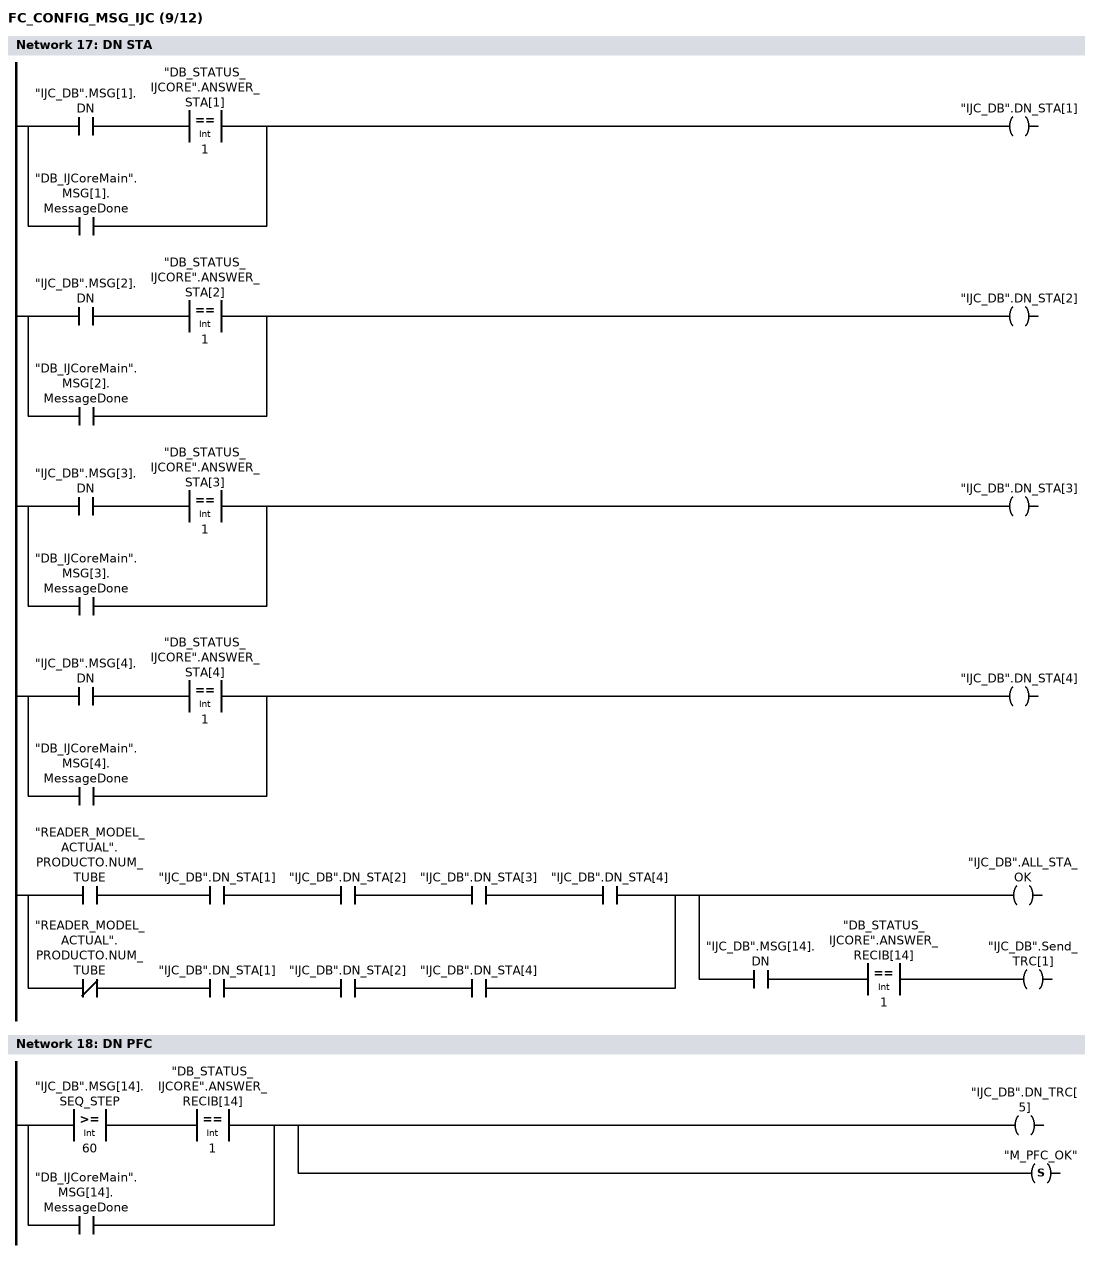
   RUNG wire#powerrail
      Contact( "IJC_DB".MSG[1].DN )
      { S7_Templates := "SrcType := Int" } EQ_Contact(in1 := "DB_STATUS_IJCORE".ANSWER_STA[1], in2 := 1)
      wire#w1
      Coil( "IJC_DB".DN_STA[1] )
   END_RUNG
   RUNG wire#powerrail
      Contact( "DB_IJCoreMain".MSG[1].MessageDone )
   END_RUNG wire#w1
   RUNG wire#powerrail
      Contact( "IJC_DB".MSG[2].DN )
      { S7_Templates := "SrcType := Int" } EQ_Contact(in1 := "DB_STATUS_IJCORE".ANSWER_STA[2], in2 := 1)
      wire#w2
      Coil( "IJC_DB".DN_STA[2] )
   END_RUNG
   RUNG wire#powerrail
      Contact( "DB_IJCoreMain".MSG[2].MessageDone )
   END_RUNG wire#w2
   RUNG wire#powerrail
      Contact( "IJC_DB".MSG[3].DN )
      { S7_Templates := "SrcType := Int" } EQ_Contact(in1 := "DB_STATUS_IJCORE".ANSWER_STA[3], in2 := 1)
      wire#w3
      Coil( "IJC_DB".DN_STA[3] )
   END_RUNG
   RUNG wire#powerrail
      Contact( "DB_IJCoreMain".MSG[3].MessageDone )
   END_RUNG wire#w3
   RUNG wire#powerrail
      Contact( "IJC_DB".MSG[4].DN )
      { S7_Templates := "SrcType := Int" } EQ_Contact(in1 := "DB_STATUS_IJCORE".ANSWER_STA[4], in2 := 1)
      wire#w4
      Coil( "IJC_DB".DN_STA[4] )
   END_RUNG
   RUNG wire#powerrail
      Contact( "DB_IJCoreMain".MSG[4].MessageDone )
   END_RUNG wire#w4
   RUNG wire#powerrail
      Contact( "READER_MODEL_ACTUAL".PRODUCTO.NUM_TUBE )
      Contact( "IJC_DB".DN_STA[1] )
      Contact( "IJC_DB".DN_STA[2] )
      Contact( "IJC_DB".DN_STA[3] )
      Contact( "IJC_DB".DN_STA[4] )
      wire#w5
      Coil( "IJC_DB".ALL_STA_OK )
   END_RUNG
   RUNG wire#powerrail
      I_Contact( "READER_MODEL_ACTUAL".PRODUCTO.NUM_TUBE )
      Contact( "IJC_DB".DN_STA[1] )
      Contact( "IJC_DB".DN_STA[2] )
      Contact( "IJC_DB".DN_STA[4] )
   END_RUNG wire#w5
   RUNG wire#w5
      Contact( "IJC_DB".MSG[14].DN )
      { S7_Templates := "SrcType := Int" } EQ_Contact(in1 := "DB_STATUS_IJCORE".ANSWER_RECIB[14], in2 := 1)
      Coil( "IJC_DB".Send_TRC[1] )
   END_RUNG
   // the same network as SCL:
   "IJC_DB".DN_STA[1] := ("IJC_DB".MSG[1].DN AND ("DB_STATUS_IJCORE".ANSWER_STA[1] = 1)) OR "DB_IJCoreMain".MSG[1].MessageDone;
   "IJC_DB".DN_STA[2] := ("IJC_DB".MSG[2].DN AND ("DB_STATUS_IJCORE".ANSWER_STA[2] = 1)) OR "DB_IJCoreMain".MSG[2].MessageDone;
   "IJC_DB".DN_STA[3] := ("IJC_DB".MSG[3].DN AND ("DB_STATUS_IJCORE".ANSWER_STA[3] = 1)) OR "DB_IJCoreMain".MSG[3].MessageDone;
   "IJC_DB".DN_STA[4] := ("IJC_DB".MSG[4].DN AND ("DB_STATUS_IJCORE".ANSWER_STA[4] = 1)) OR "DB_IJCoreMain".MSG[4].MessageDone;
   "IJC_DB".ALL_STA_OK := ("READER_MODEL_ACTUAL".PRODUCTO.NUM_TUBE AND "IJC_DB".DN_STA[1] AND "IJC_DB".DN_STA[2] AND "IJC_DB".DN_STA[3] AND "IJC_DB".DN_STA[4]) OR (NOT "READER_MODEL_ACTUAL".PRODUCTO.NUM_TUBE AND "IJC_DB".DN_STA[1] AND "IJC_DB".DN_STA[2] AND "IJC_DB".DN_STA[4]);
   "IJC_DB".Send_TRC[1] := "IJC_DB".ALL_STA_OK AND "IJC_DB".MSG[14].DN AND ("DB_STATUS_IJCORE".ANSWER_RECIB[14] = 1);
END_REGION

REGION Network 18: DN PFC
   RUNG wire#powerrail
      { S7_Templates := "SrcType := Int" } GE_Contact(in1 := "IJC_DB".MSG[14].SEQ_STEP, in2 := 60)
      { S7_Templates := "SrcType := Int" } EQ_Contact(in1 := "DB_STATUS_IJCORE".ANSWER_RECIB[14], in2 := 1)
      wire#w1
      Coil( "IJC_DB".DN_TRC[5] )
   END_RUNG
   RUNG wire#powerrail
      Contact( "DB_IJCoreMain".MSG[14].MessageDone )
   END_RUNG wire#w1
   RUNG wire#w1
      S_Coil( "M_PFC_OK" )
   END_RUNG
   // the same network as SCL:
   "IJC_DB".DN_TRC[5] := (("IJC_DB".MSG[14].SEQ_STEP >= 60) AND ("DB_STATUS_IJCORE".ANSWER_RECIB[14] = 1)) OR "DB_IJCoreMain".MSG[14].MessageDone;
   IF (("IJC_DB".MSG[14].SEQ_STEP >= 60) AND ("DB_STATUS_IJCORE".ANSWER_RECIB[14] = 1)) OR "DB_IJCoreMain".MSG[14].MessageDone THEN
       "M_PFC_OK" := TRUE;
   END_IF;
END_REGION

REGION Network 19: DN TRR
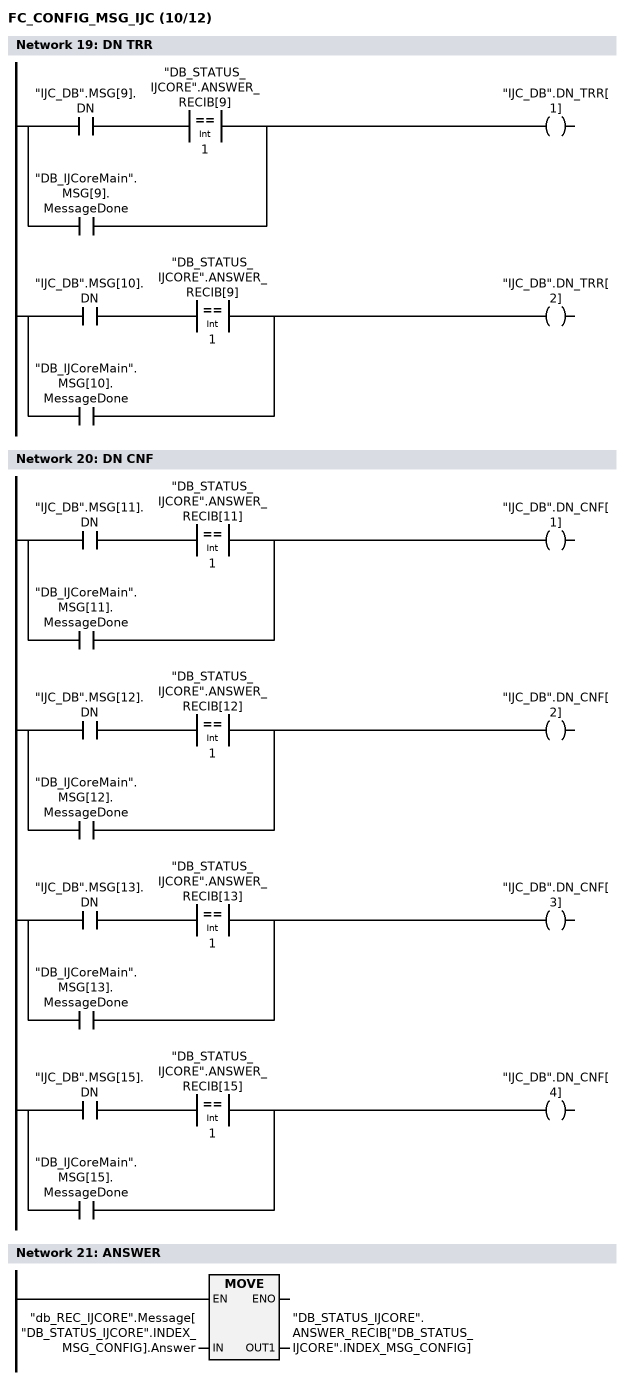
   RUNG wire#powerrail
      Contact( "IJC_DB".MSG[9].DN )
      { S7_Templates := "SrcType := Int" } EQ_Contact(in1 := "DB_STATUS_IJCORE".ANSWER_RECIB[9], in2 := 1)
      wire#w1
      Coil( "IJC_DB".DN_TRR[1] )
   END_RUNG
   RUNG wire#powerrail
      Contact( "DB_IJCoreMain".MSG[9].MessageDone )
   END_RUNG wire#w1
   RUNG wire#powerrail
      Contact( "IJC_DB".MSG[10].DN )
      { S7_Templates := "SrcType := Int" } EQ_Contact(in1 := "DB_STATUS_IJCORE".ANSWER_RECIB[9], in2 := 1)
      wire#w2
      Coil( "IJC_DB".DN_TRR[2] )
   END_RUNG
   RUNG wire#powerrail
      Contact( "DB_IJCoreMain".MSG[10].MessageDone )
   END_RUNG wire#w2
   // the same network as SCL:
   "IJC_DB".DN_TRR[1] := ("IJC_DB".MSG[9].DN AND ("DB_STATUS_IJCORE".ANSWER_RECIB[9] = 1)) OR "DB_IJCoreMain".MSG[9].MessageDone;
   "IJC_DB".DN_TRR[2] := ("IJC_DB".MSG[10].DN AND ("DB_STATUS_IJCORE".ANSWER_RECIB[9] = 1)) OR "DB_IJCoreMain".MSG[10].MessageDone;
END_REGION

REGION Network 20: DN CNF
   RUNG wire#powerrail
      Contact( "IJC_DB".MSG[11].DN )
      { S7_Templates := "SrcType := Int" } EQ_Contact(in1 := "DB_STATUS_IJCORE".ANSWER_RECIB[11], in2 := 1)
      wire#w1
      Coil( "IJC_DB".DN_CNF[1] )
   END_RUNG
   RUNG wire#powerrail
      Contact( "DB_IJCoreMain".MSG[11].MessageDone )
   END_RUNG wire#w1
   RUNG wire#powerrail
      Contact( "IJC_DB".MSG[12].DN )
      { S7_Templates := "SrcType := Int" } EQ_Contact(in1 := "DB_STATUS_IJCORE".ANSWER_RECIB[12], in2 := 1)
      wire#w2
      Coil( "IJC_DB".DN_CNF[2] )
   END_RUNG
   RUNG wire#powerrail
      Contact( "DB_IJCoreMain".MSG[12].MessageDone )
   END_RUNG wire#w2
   RUNG wire#powerrail
      Contact( "IJC_DB".MSG[13].DN )
      { S7_Templates := "SrcType := Int" } EQ_Contact(in1 := "DB_STATUS_IJCORE".ANSWER_RECIB[13], in2 := 1)
      wire#w3
      Coil( "IJC_DB".DN_CNF[3] )
   END_RUNG
   RUNG wire#powerrail
      Contact( "DB_IJCoreMain".MSG[13].MessageDone )
   END_RUNG wire#w3
   RUNG wire#powerrail
      Contact( "IJC_DB".MSG[15].DN )
      { S7_Templates := "SrcType := Int" } EQ_Contact(in1 := "DB_STATUS_IJCORE".ANSWER_RECIB[15], in2 := 1)
      wire#w4
      Coil( "IJC_DB".DN_CNF[4] )
   END_RUNG
   RUNG wire#powerrail
      Contact( "DB_IJCoreMain".MSG[15].MessageDone )
   END_RUNG wire#w4
   // the same network as SCL:
   "IJC_DB".DN_CNF[1] := ("IJC_DB".MSG[11].DN AND ("DB_STATUS_IJCORE".ANSWER_RECIB[11] = 1)) OR "DB_IJCoreMain".MSG[11].MessageDone;
   "IJC_DB".DN_CNF[2] := ("IJC_DB".MSG[12].DN AND ("DB_STATUS_IJCORE".ANSWER_RECIB[12] = 1)) OR "DB_IJCoreMain".MSG[12].MessageDone;
   "IJC_DB".DN_CNF[3] := ("IJC_DB".MSG[13].DN AND ("DB_STATUS_IJCORE".ANSWER_RECIB[13] = 1)) OR "DB_IJCoreMain".MSG[13].MessageDone;
   "IJC_DB".DN_CNF[4] := ("IJC_DB".MSG[15].DN AND ("DB_STATUS_IJCORE".ANSWER_RECIB[15] = 1)) OR "DB_IJCoreMain".MSG[15].MessageDone;
END_REGION

REGION Network 21: ANSWER
   RUNG wire#powerrail
      Move(in := "db_REC_IJCORE".Message["DB_STATUS_IJCORE".INDEX_MSG_CONFIG].Answer, out1 => "DB_STATUS_IJCORE".ANSWER_RECIB["DB_STATUS_IJCORE".INDEX_MSG_CONFIG])
   END_RUNG
   // the same network as SCL:
   "DB_STATUS_IJCORE".ANSWER_RECIB["DB_STATUS_IJCORE".INDEX_MSG_CONFIG] := "db_REC_IJCORE".Message["DB_STATUS_IJCORE".INDEX_MSG_CONFIG].Answer;
END_REGION

REGION Network 22: ANSWER NFP
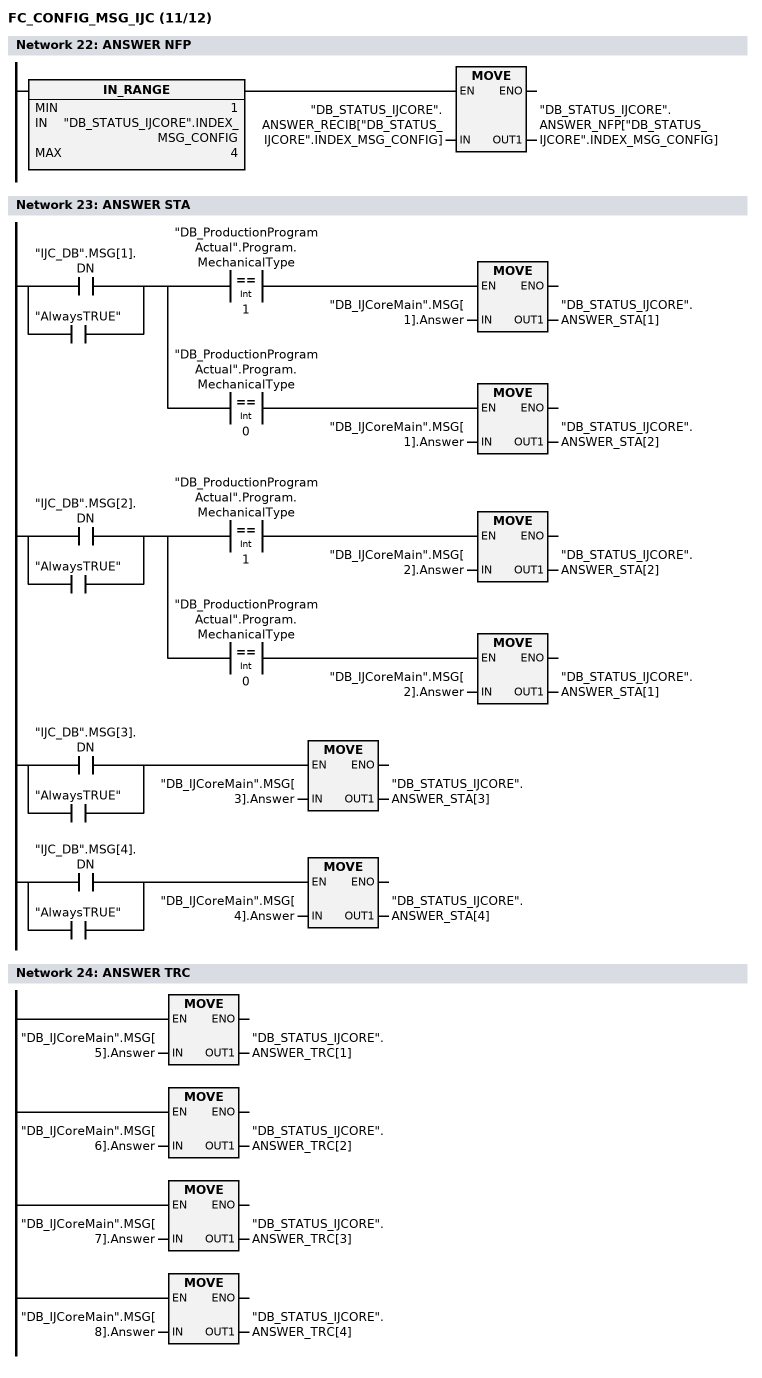
   RUNG wire#powerrail
      { S7_Templates := "SrcType := DInt" } InRange(min := 1, in := "DB_STATUS_IJCORE".INDEX_MSG_CONFIG, max := 4)
      Move(in := "DB_STATUS_IJCORE".ANSWER_RECIB["DB_STATUS_IJCORE".INDEX_MSG_CONFIG], out1 => "DB_STATUS_IJCORE".ANSWER_NFP["DB_STATUS_IJCORE".INDEX_MSG_CONFIG])
   END_RUNG
   // the same network as SCL:
   IF (1 <= "DB_STATUS_IJCORE".INDEX_MSG_CONFIG) AND ("DB_STATUS_IJCORE".INDEX_MSG_CONFIG <= 4) THEN
       "DB_STATUS_IJCORE".ANSWER_NFP["DB_STATUS_IJCORE".INDEX_MSG_CONFIG] := "DB_STATUS_IJCORE".ANSWER_RECIB["DB_STATUS_IJCORE".INDEX_MSG_CONFIG];
   END_IF;
END_REGION

REGION Network 23: ANSWER STA
   RUNG wire#powerrail
      Contact( "IJC_DB".MSG[1].DN )
      wire#w1
      { S7_Templates := "SrcType := Int" } EQ_Contact(in1 := "DB_ProductionProgramActual".Program.MechanicalType, in2 := 1)
      Move(in := "DB_IJCoreMain".MSG[1].Answer, out1 => "DB_STATUS_IJCORE".ANSWER_STA[1])
   END_RUNG
   RUNG wire#powerrail
      Contact( "AlwaysTRUE" )
   END_RUNG wire#w1
   RUNG wire#w1
      { S7_Templates := "SrcType := Int" } EQ_Contact(in1 := "DB_ProductionProgramActual".Program.MechanicalType, in2 := 0)
      Move(in := "DB_IJCoreMain".MSG[1].Answer, out1 => "DB_STATUS_IJCORE".ANSWER_STA[2])
   END_RUNG
   RUNG wire#powerrail
      Contact( "IJC_DB".MSG[2].DN )
      wire#w2
      { S7_Templates := "SrcType := Int" } EQ_Contact(in1 := "DB_ProductionProgramActual".Program.MechanicalType, in2 := 1)
      Move(in := "DB_IJCoreMain".MSG[2].Answer, out1 => "DB_STATUS_IJCORE".ANSWER_STA[2])
   END_RUNG
   RUNG wire#powerrail
      Contact( "AlwaysTRUE" )
   END_RUNG wire#w2
   RUNG wire#w2
      { S7_Templates := "SrcType := Int" } EQ_Contact(in1 := "DB_ProductionProgramActual".Program.MechanicalType, in2 := 0)
      Move(in := "DB_IJCoreMain".MSG[2].Answer, out1 => "DB_STATUS_IJCORE".ANSWER_STA[1])
   END_RUNG
   RUNG wire#powerrail
      Contact( "IJC_DB".MSG[3].DN )
      wire#w3
      Move(in := "DB_IJCoreMain".MSG[3].Answer, out1 => "DB_STATUS_IJCORE".ANSWER_STA[3])
   END_RUNG
   RUNG wire#powerrail
      Contact( "AlwaysTRUE" )
   END_RUNG wire#w3
   RUNG wire#powerrail
      Contact( "IJC_DB".MSG[4].DN )
      wire#w4
      Move(in := "DB_IJCoreMain".MSG[4].Answer, out1 => "DB_STATUS_IJCORE".ANSWER_STA[4])
   END_RUNG
   RUNG wire#powerrail
      Contact( "AlwaysTRUE" )
   END_RUNG wire#w4
   // the same network as SCL:
   #_w1 := "IJC_DB".MSG[1].DN OR "AlwaysTRUE";
   IF #_w1 AND ("DB_ProductionProgramActual".Program.MechanicalType = 1) THEN
       "DB_STATUS_IJCORE".ANSWER_STA[1] := "DB_IJCoreMain".MSG[1].Answer;
   END_IF;
   IF #_w1 AND ("DB_ProductionProgramActual".Program.MechanicalType = 0) THEN
       "DB_STATUS_IJCORE".ANSWER_STA[2] := "DB_IJCoreMain".MSG[1].Answer;
   END_IF;
   #_w2 := "IJC_DB".MSG[2].DN OR "AlwaysTRUE";
   IF #_w2 AND ("DB_ProductionProgramActual".Program.MechanicalType = 1) THEN
       "DB_STATUS_IJCORE".ANSWER_STA[2] := "DB_IJCoreMain".MSG[2].Answer;
   END_IF;
   IF #_w2 AND ("DB_ProductionProgramActual".Program.MechanicalType = 0) THEN
       "DB_STATUS_IJCORE".ANSWER_STA[1] := "DB_IJCoreMain".MSG[2].Answer;
   END_IF;
   IF "IJC_DB".MSG[3].DN OR "AlwaysTRUE" THEN
       "DB_STATUS_IJCORE".ANSWER_STA[3] := "DB_IJCoreMain".MSG[3].Answer;
   END_IF;
   IF "IJC_DB".MSG[4].DN OR "AlwaysTRUE" THEN
       "DB_STATUS_IJCORE".ANSWER_STA[4] := "DB_IJCoreMain".MSG[4].Answer;
   END_IF;
END_REGION

REGION Network 24: ANSWER TRC
   RUNG wire#powerrail
      Move(in := "DB_IJCoreMain".MSG[5].Answer, out1 => "DB_STATUS_IJCORE".ANSWER_TRC[1])
   END_RUNG
   RUNG wire#powerrail
      Move(in := "DB_IJCoreMain".MSG[6].Answer, out1 => "DB_STATUS_IJCORE".ANSWER_TRC[2])
   END_RUNG
   RUNG wire#powerrail
      Move(in := "DB_IJCoreMain".MSG[7].Answer, out1 => "DB_STATUS_IJCORE".ANSWER_TRC[3])
   END_RUNG
   RUNG wire#powerrail
      Move(in := "DB_IJCoreMain".MSG[8].Answer, out1 => "DB_STATUS_IJCORE".ANSWER_TRC[4])
   END_RUNG
   // the same network as SCL:
   "DB_STATUS_IJCORE".ANSWER_TRC[1] := "DB_IJCoreMain".MSG[5].Answer;
   "DB_STATUS_IJCORE".ANSWER_TRC[2] := "DB_IJCoreMain".MSG[6].Answer;
   "DB_STATUS_IJCORE".ANSWER_TRC[3] := "DB_IJCoreMain".MSG[7].Answer;
   "DB_STATUS_IJCORE".ANSWER_TRC[4] := "DB_IJCoreMain".MSG[8].Answer;
END_REGION

REGION Network 25: STATUS MSG TRC
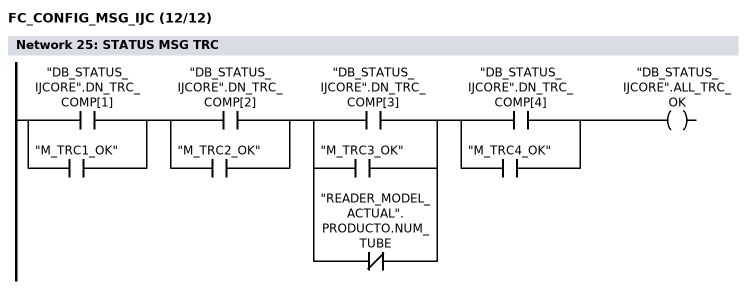
   RUNG wire#powerrail
      Contact( "DB_STATUS_IJCORE".DN_TRC_COMP[1] )
      wire#w1
      Contact( "DB_STATUS_IJCORE".DN_TRC_COMP[2] )
      wire#w2
      Contact( "DB_STATUS_IJCORE".DN_TRC_COMP[3] )
      wire#w3
      Contact( "DB_STATUS_IJCORE".DN_TRC_COMP[4] )
      wire#w4
      Coil( "DB_STATUS_IJCORE".ALL_TRC_OK )
   END_RUNG
   RUNG wire#powerrail
      Contact( "M_TRC1_OK" )
   END_RUNG wire#w1
   RUNG wire#w1
      Contact( "M_TRC2_OK" )
   END_RUNG wire#w2
   RUNG wire#w2
      Contact( "M_TRC3_OK" )
   END_RUNG wire#w3
   RUNG wire#w2
      I_Contact( "READER_MODEL_ACTUAL".PRODUCTO.NUM_TUBE )
   END_RUNG wire#w3
   RUNG wire#w3
      Contact( "M_TRC4_OK" )
   END_RUNG wire#w4
   // the same network as SCL:
   "DB_STATUS_IJCORE".ALL_TRC_OK := ("DB_STATUS_IJCORE".DN_TRC_COMP[1] OR "M_TRC1_OK") AND ("DB_STATUS_IJCORE".DN_TRC_COMP[2] OR "M_TRC2_OK") AND ("DB_STATUS_IJCORE".DN_TRC_COMP[3] OR "M_TRC3_OK" OR NOT "READER_MODEL_ACTUAL".PRODUCTO.NUM_TUBE) AND ("DB_STATUS_IJCORE".DN_TRC_COMP[4] OR "M_TRC4_OK");
END_REGION
END_FUNCTION

FUNCTION_BLOCK "AWAKE_SIGNAL"   // FB1002, LAD
TITLE = Awake signal
{ S7_Optimized_Access := 'TRUE' }
VERSION : 0.1
// This function supervise Awake signal, 
// - Awake signal is to test communication between PLC and IJCORE. 
// - Awake signal is set to 1 by PLC and set to -1 by IJCORE alternatively.
// - first PLC check if awake signal is different of 1, if it is, PLC launch timer T1 
//  (1s<T1<10s). at the end of this temporisation, PLC set awake signal to 1 and 
//  launch Timer 2. 
// - if IJCORE don't set awake signal to -1 before the end of timer 2,PLC generate  
//   Time out fault for awake signal.
// stored: AutoNumber false, IsIECCheckEnabled false, IsRetainMemResEnabled false, MemoryReserve 100, SetENOAutomatically false, UDAEnableTagReadback false
   VAR_INPUT
      ack_error : Bool;   // Acknowledge button
   END_VAR
   VAR_OUTPUT
      State_com : SInt;   // State of communication : 0 no communication 1: communication lost 2 : good communication
   END_VAR
   VAR RETAIN
      T1PresetValue : Time := T#1S;   // Bit of life Timer 1 preset value
      T2PresetValue : Time := T#60S;   // Bit of Life Timer 2 preset value
   END_VAR
   VAR
      AwSignalTimeOutFault : Bool := 0;   // Awake signal time out fault
      Reset_Counters : Bool;   // Signal to reset counter
      Restart_Counter_bit_of_life : USInt := 0;   // Number of restart bit of life
      NB_Bit_of_Life : Bool;   // Number bit of life
      number_restart : DInt;   // Number restart communication
      check_restart : Bool;   // Memo to check restart communication
      t13 : TON_TIME;
      t16 { S7_SetPoint := 'True'} : TON_TIME;
      t5 { S7_SetPoint := 'True'} : TON_TIME;
      t4 { S7_SetPoint := 'True'} : TON_TIME;
   END_VAR
   VAR CONSTANT
      Trestart : Time := T#200ms;   // Timer when IJCore replies normally
      T3 : Time := T#2s;   // Timer when IJCore blocks a short period of time
   END_VAR
   VAR_TEMP   // added for the SCL form of the ladder/FBD networks
      _w1 : Bool;
   END_VAR
BEGIN

REGION Network 1: - if awake signal is -1 then launch timer 1
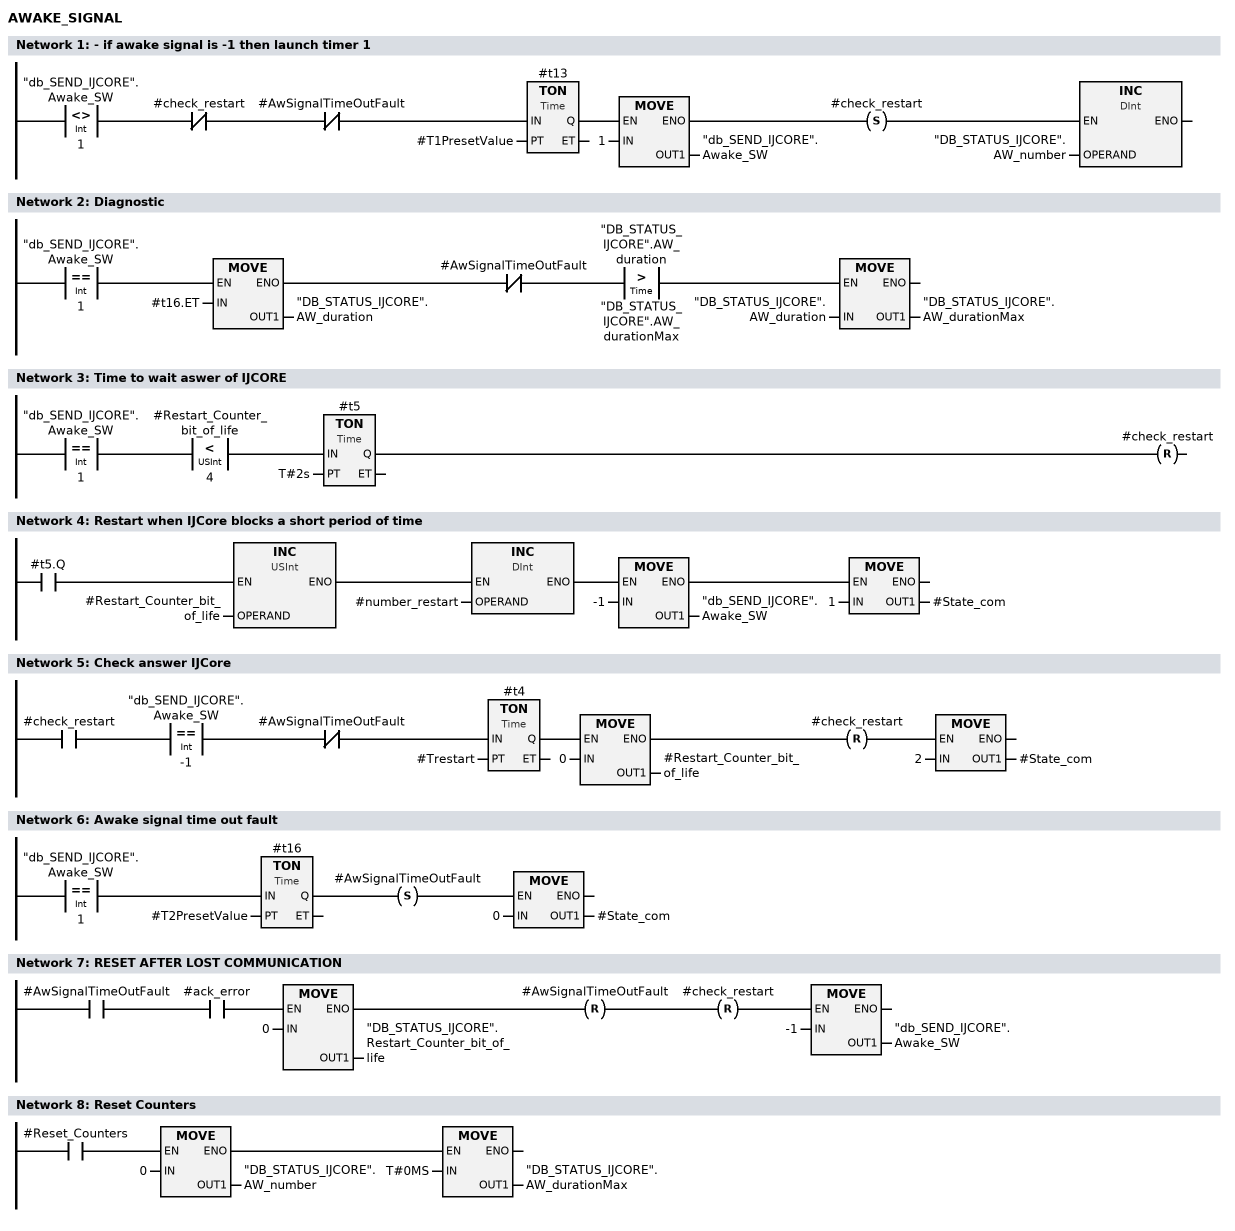
   RUNG wire#powerrail
      { S7_Templates := "SrcType := Int" } NE_Contact(in1 := "db_SEND_IJCORE".Awake_SW, in2 := 1)
      I_Contact( #check_restart )
      I_Contact( #AwSignalTimeOutFault )
      { S7_Templates := "time_type := Time" } #t13.TON(pt := #T1PresetValue, et =>)
      Move(in := 1, out1 => "db_SEND_IJCORE".Awake_SW)
      S_Coil( #check_restart )
      { S7_Templates := "DestType := DInt" } Inc( "DB_STATUS_IJCORE".AW_number )
   END_RUNG
   // the same network as SCL:
   #t13(IN := ("db_SEND_IJCORE".Awake_SW <> 1) AND NOT #check_restart AND NOT #AwSignalTimeOutFault,   // TON
        PT := #T1PresetValue);
   IF #t13.Q THEN
       "db_SEND_IJCORE".Awake_SW := 1;
       #check_restart := TRUE;
       "DB_STATUS_IJCORE".AW_number := "DB_STATUS_IJCORE".AW_number + 1;
   END_IF;
END_REGION

REGION Network 2: Diagnostic
   RUNG wire#powerrail
      { S7_Templates := "SrcType := Int" } EQ_Contact(in1 := "db_SEND_IJCORE".Awake_SW, in2 := 1)
      Move(in := #t16.ET, out1 => "DB_STATUS_IJCORE".AW_duration)
      I_Contact( #AwSignalTimeOutFault )
      { S7_Templates := "SrcType := Time" } GT_Contact(in1 := "DB_STATUS_IJCORE".AW_duration, in2 := "DB_STATUS_IJCORE".AW_durationMax)
      Move(in := "DB_STATUS_IJCORE".AW_duration, out1 => "DB_STATUS_IJCORE".AW_durationMax)
   END_RUNG
   // the same network as SCL:
   #_w1 := "db_SEND_IJCORE".Awake_SW = 1;
   IF #_w1 THEN "DB_STATUS_IJCORE".AW_duration := #t16.ET; END_IF;
   IF #_w1 AND NOT #AwSignalTimeOutFault AND ("DB_STATUS_IJCORE".AW_duration > "DB_STATUS_IJCORE".AW_durationMax) THEN
       "DB_STATUS_IJCORE".AW_durationMax := "DB_STATUS_IJCORE".AW_duration;
   END_IF;
END_REGION

REGION Network 3: Time to wait aswer of IJCORE
   RUNG wire#powerrail
      { S7_Templates := "SrcType := Int" } EQ_Contact(in1 := "db_SEND_IJCORE".Awake_SW, in2 := 1)
      { S7_Templates := "SrcType := USInt" } LT_Contact(in1 := #Restart_Counter_bit_of_life, in2 := 4)
      { S7_Templates := "time_type := Time" } #t5.TON(pt := T#2s, et =>)
      R_Coil( #check_restart )
   END_RUNG
   // the same network as SCL:
   #t5(IN := ("db_SEND_IJCORE".Awake_SW = 1) AND (#Restart_Counter_bit_of_life < 4), PT := T#2s);   // TON
   IF #t5.Q THEN #check_restart := FALSE; END_IF;
END_REGION

REGION Network 4: Restart when IJCore blocks a short period of time
   RUNG wire#powerrail
      Contact( #t5.Q )
      { S7_Templates := "DestType := USInt" } Inc( #Restart_Counter_bit_of_life )
      { S7_Templates := "DestType := DInt" } Inc( #number_restart )
      Move(in := -1, out1 => "db_SEND_IJCORE".Awake_SW)
      Move(in := 1, out1 => #State_com)
   END_RUNG
   // the same network as SCL:
   IF #t5.Q THEN
       #Restart_Counter_bit_of_life := #Restart_Counter_bit_of_life + 1;
       #number_restart := #number_restart + 1;
       "db_SEND_IJCORE".Awake_SW := -1;
       #State_com := 1;
   END_IF;
END_REGION

REGION Network 5: Check answer IJCore
   RUNG wire#powerrail
      Contact( #check_restart )
      { S7_Templates := "SrcType := Int" } EQ_Contact(in1 := "db_SEND_IJCORE".Awake_SW, in2 := -1)
      I_Contact( #AwSignalTimeOutFault )
      { S7_Templates := "time_type := Time" } #t4.TON(pt := #Trestart, et =>)
      Move(in := 0, out1 => #Restart_Counter_bit_of_life)
      R_Coil( #check_restart )
      Move(in := 2, out1 => #State_com)
   END_RUNG
   // the same network as SCL:
   #t4(IN := #check_restart AND ("db_SEND_IJCORE".Awake_SW = (-1)) AND NOT #AwSignalTimeOutFault,   // TON
       PT := #Trestart);
   IF #t4.Q THEN
       #Restart_Counter_bit_of_life := 0;
       #check_restart := FALSE;
       #State_com := 2;
   END_IF;
END_REGION

REGION Network 6: Awake signal time out fault
   RUNG wire#powerrail
      { S7_Templates := "SrcType := Int" } EQ_Contact(in1 := "db_SEND_IJCORE".Awake_SW, in2 := 1)
      { S7_Templates := "time_type := Time" } #t16.TON(pt := #T2PresetValue, et =>)
      S_Coil( #AwSignalTimeOutFault )
      Move(in := 0, out1 => #State_com)
   END_RUNG
   // the same network as SCL:
   #t16(IN := "db_SEND_IJCORE".Awake_SW = 1, PT := #T2PresetValue);   // TON
   IF #t16.Q THEN
       #AwSignalTimeOutFault := TRUE;
       #State_com := 0;
   END_IF;
END_REGION

REGION Network 7: RESET AFTER LOST COMMUNICATION
   RUNG wire#powerrail
      Contact( #AwSignalTimeOutFault )
      Contact( #ack_error )
      Move(in := 0, out1 => "DB_STATUS_IJCORE".Restart_Counter_bit_of_life)
      R_Coil( #AwSignalTimeOutFault )
      R_Coil( #check_restart )
      Move(in := -1, out1 => "db_SEND_IJCORE".Awake_SW)
   END_RUNG
   // the same network as SCL:
   IF #AwSignalTimeOutFault AND #ack_error THEN "DB_STATUS_IJCORE".Restart_Counter_bit_of_life := 0; END_IF;
   #_w1 := #AwSignalTimeOutFault AND #ack_error;
   IF #_w1 THEN
       #AwSignalTimeOutFault := FALSE;
       #check_restart := FALSE;
       "db_SEND_IJCORE".Awake_SW := -1;
   END_IF;
END_REGION

